T1313 BOOL  ; B机架#3门磁（公共）感应延时[0019.09]
T1314 BOOL  ; B机架#4门磁（公共）感应延时[0019.10]
T1315 BOOL  ; B机架#5门磁（公共）感应延时[0019.11]
T1316 BOOL  ; B机架#6门磁（公共）感应延时[0019.12]
T1317 BOOL  ; RK_07 #3托盘下料下降到位感应感应延时[0019.13]
T1318 BOOL  ; $?St$Bk?_#[5054] / RK_07 #3托盘下料位物料车到位感应#2感应延时[0019.14] / $?St$Bk?_#[5054]
T1319 BOOL  ; $?St$Bk?_#[5055] / RK_07 铝壳上料移载托盘到位保护感应感应延时[0019.15] / $?St$Bk?_#[5055]
T1322 BOOL  ; RK_02 电芯进料机械手#1压紧气缸压紧位感应延时
T1323 BOOL  ; RK_02 电芯进料机械手#2压紧气缸压紧位感应延时
T1326 BOOL  ; RK_03 电芯上料机械手#1压紧气缸压紧位感应延时
T1327 BOOL  ; RK_03 电芯上料机械手#2压紧气缸压紧位感应延时
T1373 BOOL  ; RK_05 #1入壳吸盘上#1伸缩气缸伸出位感应延时
T1374 BOOL  ; RK_05 #1入壳吸盘上#2伸缩气缸伸出位感应延时
T1375 BOOL  ; RK_05 #1入壳吸盘上#3伸缩气缸伸出位感应延时
T1376 BOOL  ; RK_05 #1入壳吸盘下#1伸缩气缸伸出位感应延时
T1377 BOOL  ; RK_05 #1入壳吸盘下#2伸缩气缸伸出位感应延时
T1378 BOOL  ; RK_05 #1入壳吸盘下#3伸缩气缸伸出位感应延时
T1391 BOOL  ; RK_05 #2入壳吸盘上#1伸缩气缸伸出位感应延时
T1392 BOOL  ; RK_05 #2入壳吸盘上#2伸缩气缸伸出位感应延时
T1393 BOOL  ; RK_05 #2入壳吸盘上#3伸缩气缸伸出位感应延时
T1394 BOOL  ; RK_05 #2入壳吸盘下#1伸缩气缸伸出位感应延时
T1395 BOOL  ; RK_05 #2入壳吸盘下#2伸缩气缸伸出位感应延时
T1396 BOOL  ; RK_05 #2入壳吸盘下#3伸缩气缸伸出位感应延时
T1500 BOOL  ; RK_02 电芯进料机械手夹爪气缸夹紧位报警延时
T1501 BOOL  ; RK_02 电芯进料机械手夹爪气缸张开位报警延时
T1502 BOOL  ; RK_02 电芯进料机械手#1压紧气缸松开位报警延时
T1503 BOOL  ; RK_02 电芯进料机械手#2压紧气缸松开位报警延时
T1504 BOOL  ; RK_03 电芯上料机械手夹爪气缸夹紧位报警延时
T1505 BOOL  ; RK_03 电芯上料机械手夹爪气缸张开位报警延时
T1506 BOOL  ; RK_03 电芯上料机械手#1压紧气缸松开位报警延时
T1507 BOOL  ; RK_03 电芯上料机械手#2压紧气缸松开位报警延时
T1508 BOOL  ; RK_03 电芯上料升降气缸下降位报警延时
T1509 BOOL  ; RK_03 电芯上料升降气缸上升位报警延时
T1510 BOOL  ; RK_04 电芯除尘伸缩气缸缩回位报警延时
T1511 BOOL  ; RK_04 电芯除尘伸缩气缸伸出位报警延时
T1512 BOOL  ; RK_05 #1入壳滚轮夹紧气缸夹紧位报警延时
T1513 BOOL  ; RK_05 #1入壳滚轮夹紧气缸松开位报警延时
T1514 BOOL  ; RK_05 #1入壳铝壳定位平台伸缩气缸缩回位报警延时
T1515 BOOL  ; RK_05 #1入壳铝壳定位平台伸缩气缸伸出位报警延时
T1516 BOOL  ; RK_05 #1入壳铝壳定位平台升降气缸上升位报警延时
T1517 BOOL  ; RK_05 #1入壳铝壳定位平台升降气缸下降位报警延时
T1518 BOOL  ; RK_05 #1入壳铝壳定位伸缩气缸缩回位报警延时
T1519 BOOL  ; RK_05 #1入壳铝壳定位伸缩气缸伸出位报警延时
T1520 BOOL  ; RK_05 #1入壳铝壳定位夹爪气缸夹紧位报警延时
T1521 BOOL  ; RK_05 #1入壳铝壳定位夹爪气缸张开位报警延时
T1522 BOOL  ; RK_05 #2入壳滚轮夹紧气缸夹紧位报警延时
T1523 BOOL  ; RK_05 #2入壳滚轮夹紧气缸松开位报警延时
T1524 BOOL  ; RK_05 #2入壳铝壳定位平台伸缩气缸缩回位报警延时
T1525 BOOL  ; RK_05 #2入壳铝壳定位平台伸缩气缸伸出位报警延时
T1526 BOOL  ; RK_05 #2入壳铝壳定位平台升降气缸上升位报警延时
T1527 BOOL  ; RK_05 #2入壳铝壳定位平台升降气缸下降位报警延时
T1528 BOOL  ; RK_05 #2入壳铝壳定位伸缩气缸缩回位报警延时
T1529 BOOL  ; RK_05 #2入壳铝壳定位伸缩气缸伸出位报警延时
T1530 BOOL  ; RK_05 #2入壳铝壳定位夹爪气缸夹紧位报警延时
T1531 BOOL  ; RK_05 #2入壳铝壳定位夹爪气缸张开位报警延时
T1532 BOOL  ; RK_01 U0_X 电芯来料Y轴报警信号报警延时
T1533 BOOL  ; RK_01 U0_X 电芯来料Y轴准备好了信号报警延时
T1534 BOOL  ; RK_02 U0_Y 电芯进料X轴报警信号报警延时
T1535 BOOL  ; RK_02 U0_Y 电芯进料X轴准备好了信号报警延时
T1536 BOOL  ; RK_02 U0_Z 电芯进料Z轴报警信号报警延时
T1537 BOOL  ; RK_02 U0_Z 电芯进料Z轴准备好了信号报警延时
T1538 BOOL  ; RK_03 U0_U 电芯上料X轴报警信号报警延时
T1539 BOOL  ; RK_03 U0_U 电芯上料X轴准备好了信号报警延时
T1540 BOOL  ; RK_05 U2_X #1入壳Y轴报警信号报警延时
T1541 BOOL  ; RK_05 U2_X #1入壳Y轴准备好了信号报警延时
T1542 BOOL  ; RK_05 U2_Y #2入壳Y轴报警信号报警延时
T1543 BOOL  ; RK_05 U2_Y #2入壳Y轴准备好了信号报警延时
T1544 BOOL  ; 0报警延时
T1545 BOOL  ; RK_05 #1入壳定位陶瓷棒上#1夹紧气缸伸出位报警延时
T1546 BOOL  ; RK_05 #1入壳定位陶瓷棒上#2夹紧气缸伸出位报警延时
T1547 BOOL  ; RK_05 #1入壳定位陶瓷棒下#1夹紧气缸伸出位报警延时
T1548 BOOL  ; RK_05 #1入壳定位陶瓷棒下#2夹紧气缸伸出位报警延时
T1549 BOOL  ; RK_05 #1入壳定位陶瓷棒上#1夹紧气缸缩回位报警延时
T1550 BOOL  ; RK_05 #1入壳定位陶瓷棒上#2夹紧气缸缩回位报警延时
T1551 BOOL  ; RK_05 #1入壳定位陶瓷棒下#1夹紧气缸缩回位报警延时
T1552 BOOL  ; RK_05 #1入壳定位陶瓷棒下#2夹紧气缸缩回位报警延时
T1553 BOOL  ; RK_05 #1入壳吸盘上#1伸缩气缸缩回位报警延时
T1554 BOOL  ; RK_05 #1入壳吸盘上#2伸缩气缸缩回位报警延时
T1555 BOOL  ; RK_05 #1入壳吸盘上#3伸缩气缸缩回位报警延时
T1556 BOOL  ; RK_05 #1入壳吸盘下#1伸缩气缸缩回位报警延时
T1557 BOOL  ; RK_05 #1入壳吸盘下#2伸缩气缸缩回位报警延时
T1558 BOOL  ; RK_05 #1入壳吸盘下#3伸缩气缸缩回位报警延时
T1559 BOOL  ; RK_05 #1入壳电芯#1定位夹爪气缸松开位报警延时
T1560 BOOL  ; RK_05 #1入壳电芯#2定位夹爪气缸松开位报警延时
T1561 BOOL  ; RK_05 #1入壳电芯#1定位夹爪气缸夹紧位报警延时
T1562 BOOL  ; RK_05 #1入壳电芯#2定位夹爪气缸夹紧位报警延时
T1563 BOOL  ; RK_05 #2入壳定位陶瓷棒上#1夹紧气缸伸出位报警延时
T1564 BOOL  ; RK_05 #2入壳定位陶瓷棒上#2夹紧气缸伸出位报警延时
T1565 BOOL  ; RK_05 #2入壳定位陶瓷棒下#1夹紧气缸伸出位报警延时
T1566 BOOL  ; RK_05 #2入壳定位陶瓷棒下#2夹紧气缸伸出位报警延时
T1567 BOOL  ; RK_05 #2入壳定位陶瓷棒上#1夹紧气缸缩回位报警延时
T1568 BOOL  ; RK_05 #2入壳定位陶瓷棒上#2夹紧气缸缩回位报警延时
T1569 BOOL  ; RK_05 #2入壳定位陶瓷棒下#1夹紧气缸缩回位报警延时
T1570 BOOL  ; RK_05 #2入壳定位陶瓷棒下#2夹紧气缸缩回位报警延时
T1571 BOOL  ; RK_05 #2入壳吸盘上#1伸缩气缸缩回位报警延时
T1572 BOOL  ; RK_05 #2入壳吸盘上#2伸缩气缸缩回位报警延时
T1573 BOOL  ; RK_05 #2入壳吸盘上#3伸缩气缸缩回位报警延时
T1574 BOOL  ; RK_05 #2入壳吸盘下#1伸缩气缸缩回位报警延时
T1575 BOOL  ; RK_05 #2入壳吸盘下#2伸缩气缸缩回位报警延时
T1576 BOOL  ; RK_05 #2入壳吸盘下#3伸缩气缸缩回位报警延时
T1577 BOOL  ; RK_05 #2入壳电芯#1定位夹爪气缸松开位报警延时
T1578 BOOL  ; RK_05 #2入壳电芯#2定位夹爪气缸松开位报警延时
T1579 BOOL  ; RK_05 #2入壳电芯#1定位夹爪气缸夹紧位报警延时
T1580 BOOL  ; RK_05 #2入壳电芯#2定位夹爪气缸夹紧位报警延时
T1581 BOOL  ; RK_01 电芯来料有料感应报警延时
T1582 BOOL  ; RK_02 电芯进料机械手夹爪柔性报警报警延时
T1583 BOOL  ; RK_03 电芯上料机械手夹爪柔性报警报警延时
T1584 BOOL  ; RK_04 电芯除尘有料感应报警延时
T1585 BOOL  ; RK_02 扫码NG拉带有料感应#1报警延时
T1586 BOOL  ; RK_02 扫码NG拉带有料感应#2报警延时
T1587 BOOL  ; RK_02 扫码NG拉带料满感应报警延时
T1588 BOOL  ; RK_05 #1入壳电芯有料感应报警延时
T1589 BOOL  ; RK_05 #1入壳铝壳有料感应报警延时
T1590 BOOL  ; RK_05 #2入壳电芯有料感应报警延时
T1591 BOOL  ; RK_05 #2入壳铝壳有料感应报警延时
T1592 BOOL  ; RK_05 #1入壳吸盘立真空报警延时
T1593 BOOL  ; RK_05 #2入壳吸盘立真空报警延时
T1594 BOOL  ; 前端设备对接输入信号（公共）报警延时
T1595 BOOL  ; 后端设备对接输入信号（公共）报警延时
T1597 BOOL  ; NC433模块DC5V电源信号（公共）报警延时
T1598 BOOL  ; DC24V伺服刹车电源信号（公共）报警延时
T1610 BOOL  ; 0报警延时
T1611 BOOL  ; 0报警延时
T1612 BOOL  ; 0报警延时
T1613 BOOL  ; 0报警延时
T1614 BOOL  ; 0报警延时
T1615 BOOL  ; 0报警延时
T1616 BOOL  ; 0报警延时
T1617 BOOL  ; 0报警延时
T1618 BOOL  ; 0报警延时
T1619 BOOL  ; 0报警延时
T1620 BOOL  ; 0报警延时
T1621 BOOL  ; 0报警延时
T1622 BOOL  ; 0报警延时
T1623 BOOL  ; 0报警延时
T1624 BOOL  ; 0报警延时
T1625 BOOL  ; 0报警延时
T1626 BOOL  ; 0报警延时
T1627 BOOL  ; 0报警延时
T1628 BOOL  ; RK_11 电池除尘旋转伸缩气缸到位报警延时
T1629 BOOL  ; RK_11 电池除尘旋转伸缩气缸原位报警延时
T1630 BOOL  ; RK_11 电池除尘伸缩气缸伸出位报警延时
T1631 BOOL  ; RK_11 电池除尘伸缩气缸缩回位报警延时
T1632 BOOL  ; RK_11 电池除尘夹爪气缸夹紧位报警延时
T1633 BOOL  ; RK_11 电池除尘夹爪气缸张开位报警延时
T1634 BOOL  ; RK_12 预焊上料机械手夹爪气缸夹紧位报警延时
T1635 BOOL  ; RK_12 预焊上料机械手夹爪气缸张开位报警延时
T1636 BOOL  ; RK_12 预焊下料机械手夹爪气缸夹紧位报警延时
T1637 BOOL  ; RK_12 预焊下料机械手夹爪气缸张开位报警延时
T1638 BOOL  ; RK_13 #1移载升降气缸上升位报警延时
T1639 BOOL  ; RK_13 #1移载升降气缸下降位报警延时
T1640 BOOL  ; RK_13 #1移载定位#1伸缩气缸缩回位报警延时
T1641 BOOL  ; RK_13 #1移载定位#1伸缩气缸伸出位报警延时
T1642 BOOL  ; RK_13 #1移载定位#2伸缩气缸缩回位报警延时
T1643 BOOL  ; RK_13 #1移载定位#2伸缩气缸伸出位报警延时
T1644 BOOL  ; RK_13 #1移载导向#1伸缩气缸伸出位报警延时
T1645 BOOL  ; RK_13 #1移载导向#1伸缩气缸缩回位报警延时
T1646 BOOL  ; RK_13 #1移载导向#2伸缩气缸伸出位报警延时
T1647 BOOL  ; RK_13 #1移载导向#2伸缩气缸缩回位报警延时
T1648 BOOL  ; RK_13 #1移载左右定位伸缩气缸伸出位报警延时
T1649 BOOL  ; RK_13 #1移载左右定位伸缩气缸缩回位报警延时
T1650 BOOL  ; RK_13 #2移载升降气缸上升位报警延时
T1651 BOOL  ; RK_13 #2移载升降气缸下降位报警延时
T1652 BOOL  ; RK_13 #2移载定位#1伸缩气缸缩回位报警延时
T1653 BOOL  ; RK_13 #2移载定位#1伸缩气缸伸出位报警延时
T1654 BOOL  ; RK_13 #2移载定位#2伸缩气缸缩回位报警延时
T1655 BOOL  ; RK_13 #2移载定位#2伸缩气缸伸出位报警延时
T1656 BOOL  ; RK_13 #2移载导向#1伸缩气缸伸出位报警延时
T1657 BOOL  ; RK_13 #2移载导向#1伸缩气缸缩回位报警延时
T1658 BOOL  ; RK_13 #2移载导向#2伸缩气缸伸出位报警延时
T1659 BOOL  ; RK_13 #2移载导向#2伸缩气缸缩回位报警延时
T1660 BOOL  ; RK_13 #2移载左右定位伸缩气缸伸出位报警延时
T1661 BOOL  ; RK_13 #2移载左右定位伸缩气缸缩回位报警延时
T1662 BOOL  ; RK_14 #1压装升降气缸下降位报警延时
T1663 BOOL  ; RK_14 #1压装升降气缸上升位报警延时
T1664 BOOL  ; RK_14 #1压装#1吸盘升降气缸下降位报警延时
T1665 BOOL  ; RK_14 #1压装#1吸盘升降气缸上升位报警延时
T1666 BOOL  ; RK_14 #1压装#2吸盘升降气缸下降位报警延时
T1667 BOOL  ; RK_14 #1压装#2吸盘升降气缸上升位报警延时
T1668 BOOL  ; RK_14 #2压装升降气缸下降位报警延时
T1669 BOOL  ; RK_14 #2压装升降气缸上升位报警延时
T1670 BOOL  ; RK_14 #2压装#1吸盘升降气缸下降位报警延时
T1671 BOOL  ; RK_14 #2压装#1吸盘升降气缸上升位报警延时
T1672 BOOL  ; RK_14 #2压装#2吸盘升降气缸下降位报警延时
T1673 BOOL  ; RK_14 #2压装#2吸盘升降气缸上升位报警延时
T1674 BOOL  ; RK_15 轮廓检测#1伸缩气缸伸出位报警延时
T1675 BOOL  ; RK_15 轮廓检测#1伸缩气缸缩回位报警延时
T1676 BOOL  ; RK_15 轮廓检测#2伸缩气缸伸出位报警延时
T1677 BOOL  ; RK_15 轮廓检测#2伸缩气缸缩回位报警延时
T1678 BOOL  ; RK_12 轮廓检测NG拨料气缸伸出位报警延时
T1679 BOOL  ; RK_12 轮廓检测NG拨料气缸缩回位报警延时
T1680 BOOL  ; RK_11 电池除尘有料感应报警延时
T1681 BOOL  ; RK_12 预焊上料机械手夹爪柔性报警报警延时
T1682 BOOL  ; RK_12 预焊下料机械手夹爪柔性报警报警延时
T1683 BOOL  ; RK_16 激光焊接完成信号报警延时
T1684 BOOL  ; RK_16 激光焊机故障信号报警延时
T1685 BOOL  ; RK_13 #1移载电池顶盖超高检测报警延时
T1686 BOOL  ; RK_16 激光焊机急停信号报警延时
T1687 BOOL  ; RK_13 #2移载电池顶盖超高检测报警延时
T1688 BOOL  ; RK_13 #1移载有料感应报警延时
T1689 BOOL  ; RK_13 #2移载有料感应报警延时
T1690 BOOL  ; RK_14 #1压装吸盘立真空报警延时
T1691 BOOL  ; RK_14 #2压装吸盘立真空报警延时
T1692 BOOL  ; RK_12 U4_X 预焊上下料X轴报警信号报警延时
T1693 BOOL  ; RK_12 U4_X 预焊上下料X轴准备好了信号报警延时
T1694 BOOL  ; RK_12 U4_Y 预焊上料Z轴报警信号报警延时
T1695 BOOL  ; RK_12 U4_Y 预焊上料Z轴准备好了信号报警延时
T1696 BOOL  ; RK_12 U4_Z 预焊下料Z轴报警信号报警延时
T1697 BOOL  ; RK_12 U4_Z 预焊下料Z轴准备好了信号报警延时
T1698 BOOL  ; RK_13 U4_U #1移载Y轴报警信号报警延时
T1699 BOOL  ; RK_13 U4_U #1移载Y轴准备好了信号报警延时
T1700 BOOL  ; RK_13 U6_X #2移载Y轴报警信号报警延时
T1701 BOOL  ; RK_13 U6_X #2移载Y轴准备好了信号报警延时
T1702 BOOL  ; RK_16 U6_Y 激光焊接X轴报警信号报警延时
T1703 BOOL  ; RK_16 U6_Y 激光焊接X轴准备好了信号报警延时
T1704 BOOL  ; RK_16 U6_Z 激光焊接Z轴报警信号报警延时
T1705 BOOL  ; RK_16 U6_Z 激光焊接Z轴准备好了信号报警延时
T1706 BOOL  ; 0报警延时
T1707 BOOL  ; 0报警延时
T1708 BOOL  ; 0报警延时
T1709 BOOL  ; RK_12 轮廓检测NG料槽#1有料感应报警延时
T1710 BOOL  ; RK_12 轮廓检测NG料槽#1料满感应报警延时
T1711 BOOL  ; RK_12 轮廓检测NG料槽#2有料感应报警延时
T1712 BOOL  ; RK_12 轮廓检测NG料槽#2料满感应报警延时
T1713 BOOL  ; RK_12 OK出料拉带放料位有料感应#1报警延时
T1714 BOOL  ; RK_12 OK出料拉带放料位有料感应#2报警延时
T1715 BOOL  ; RK_12 OK出料拉带出料位有料感应报警延时
T1716 BOOL  ; 0报警延时
T1717 BOOL  ; 0报警延时
T1718 BOOL  ; 0报警延时
T1719 BOOL  ; 0报警延时
T1720 BOOL  ; 0报警延时
T1721 BOOL  ; 0报警延时
T1722 BOOL  ; 0报警延时
T1723 BOOL  ; 0报警延时
T1724 BOOL  ; RK_06 铝壳上料升降气缸下降位报警延时
T1725 BOOL  ; RK_06 铝壳上料升降气缸上升位报警延时
T1726 BOOL  ; RK_06 电池下料升降气缸下降位报警延时
T1727 BOOL  ; RK_06 电池下料升降气缸上升位报警延时
T1728 BOOL  ; RK_06 铝壳上料夹爪气缸夹紧位报警延时
T1729 BOOL  ; RK_06 铝壳上料夹爪气缸张开位报警延时
T1730 BOOL  ; RK_06 电池下料夹爪气缸夹紧位报警延时
T1731 BOOL  ; RK_06 电池下料夹爪气缸张开位报警延时
T1732 BOOL  ; RK_07 #1铝壳上料车定位升降气缸上升位报警延时
T1733 BOOL  ; RK_07 #1铝壳上料车定位升降气缸下降位报警延时
T1734 BOOL  ; RK_07 #2铝壳上料车定位升降气缸上升位报警延时
T1735 BOOL  ; RK_07 #2铝壳上料车定位升降气缸下降位报警延时
T1736 BOOL  ; RK_07 #3托盘下料车定位升降气缸上升位报警延时
T1737 BOOL  ; RK_07 #3托盘下料车定位升降气缸下降位报警延时
T1738 BOOL  ; RK_07 铝壳进料机械手升降气缸下降位报警延时
T1739 BOOL  ; RK_07 铝壳进料机械手升降气缸上升位报警延时
T1740 BOOL  ; RK_08 铝壳除尘旋转伸缩气缸原位报警延时
T1741 BOOL  ; RK_08 铝壳除尘旋转伸缩气缸到位报警延时
T1742 BOOL  ; RK_08 铝壳除尘伸缩气缸伸出位报警延时
T1743 BOOL  ; RK_08 铝壳除尘伸缩气缸缩回位报警延时
T1744 BOOL  ; RK_08 铝壳除尘夹爪气缸夹紧位报警延时
T1745 BOOL  ; RK_08 铝壳除尘夹爪气缸张开位报警延时
T1746 BOOL  ; RK_09 #1Hipot测试旋转伸缩气缸到位报警延时
T1747 BOOL  ; RK_09 #1Hipot测试旋转伸缩气缸原位报警延时
T1748 BOOL  ; RK_09 #1Hipot测试平台伸缩气缸缩回位报警延时
T1749 BOOL  ; RK_09 #1Hipot测试平台伸缩气缸伸出位报警延时
T1750 BOOL  ; RK_09 #1Hipot测试伸缩气缸伸出位报警延时
T1751 BOOL  ; RK_09 #1Hipot测试伸缩气缸缩回位报警延时
T1752 BOOL  ; RK_09 #2Hipot测试旋转伸缩气缸到位报警延时
T1753 BOOL  ; RK_09 #2Hipot测试旋转伸缩气缸原位报警延时
T1754 BOOL  ; RK_09 #2Hipot测试平台伸缩气缸缩回位报警延时
T1755 BOOL  ; RK_09 #2Hipot测试平台伸缩气缸伸出位报警延时
T1756 BOOL  ; RK_09 #2Hipot测试伸缩气缸伸出位报警延时
T1757 BOOL  ; RK_09 #2Hipot测试伸缩气缸缩回位报警延时
T1758 BOOL  ; RK_10 电池除尘上料机械手升降气缸下降位报警延时
T1759 BOOL  ; RK_10 电池除尘上料机械手升降气缸上升位报警延时
T1760 BOOL  ; RK_10 电池除尘上料机械手夹爪气缸夹紧位报警延时
T1761 BOOL  ; RK_10 电池除尘上料机械手夹爪气缸张开位报警延时
T1762 BOOL  ; RK_06 U8_X 电池上下料X轴报警信号报警延时
T1763 BOOL  ; RK_06 U8_X 电池上下料X轴准备好了信号报警延时
T1764 BOOL  ; RK_07 U8_Y 铝壳进料X轴报警信号报警延时
T1765 BOOL  ; RK_07 U8_Y 铝壳进料X轴准备好了信号报警延时
T1766 BOOL  ; RK_07 U8_Z 铝壳上料移载Y轴报警信号报警延时
T1767 BOOL  ; RK_07 U8_Z 铝壳上料移载Y轴准备好了信号报警延时
T1768 BOOL  ; RK_10 U8_U 电池除尘上料X轴报警信号报警延时
T1769 BOOL  ; RK_10 U8_U 电池除尘上料X轴准备好了信号报警延时
T1770 BOOL  ; RK_09 Hipot测试完成信号报警延时
T1771 BOOL  ; RK_07 #1铝壳上料启动按钮报警延时
T1772 BOOL  ; RK_07 #2铝壳上料启动按钮报警延时
T1773 BOOL  ; RK_07 #3托盘下料启动按钮报警延时
T1774 BOOL  ; RK_07 铝壳上料移载吸盘立真空报警延时
T1775 BOOL  ; RK_07 铝壳进料吸盘立真空报警延时
T1776 BOOL  ; RK_07 #1铝壳上料托盘到位感应报警延时
T1777 BOOL  ; RK_07 #1铝壳上料位物料车到位感应报警延时
T1778 BOOL  ; RK_07 #1铝壳上料初始位（#1）报警延时
T1779 BOOL  ; RK_07 #1铝壳上料一个托盘位（#2）报警延时
T1780 BOOL  ; RK_07 #1铝壳上料高限位（#3）报警延时
T1781 BOOL  ; RK_07 #2铝壳上料托盘到位感应报警延时
T1782 BOOL  ; RK_07 #2铝壳上料位物料车到位感应报警延时
T1783 BOOL  ; RK_07 #2铝壳上料初始位（#1）报警延时
T1784 BOOL  ; RK_07 #2铝壳上料一个托盘位（#2）报警延时
T1785 BOOL  ; RK_07 #2铝壳上料高限位（#3）报警延时
T1786 BOOL  ; RK_07 #3托盘下料上升到位感应报警延时
T1787 BOOL  ; RK_07 #3托盘下料位物料车到位感应报警延时
T1788 BOOL  ; RK_07 #3托盘下料初始位（#1）报警延时
T1789 BOOL  ; RK_07 #3托盘下料一个托盘位（#2）报警延时
T1790 BOOL  ; RK_07 #3托盘下料高限位（#3）报警延时
T1791 BOOL  ; RK_07 铝壳上料移载托盘到位感应报警延时
T1792 BOOL  ; RK_08 铝壳除尘有料感应报警延时
T1793 BOOL  ; RK_09 #1Hipot测试有料感应报警延时
T1794 BOOL  ; RK_09 #2Hipot测试有料感应报警延时
T1795 BOOL  ; RK_10 Hipot检测NG拉带有料感应#1报警延时
T1796 BOOL  ; RK_10 Hipot检测NG拉带有料感应#2报警延时
T1797 BOOL  ; RK_10 Hipot检测NG拉带料满感应报警延时
T1798 BOOL  ; RK_06 铝壳上料夹爪柔性报警报警延时
T1799 BOOL  ; RK_06 电池下料夹爪柔性报警报警延时
T1800 BOOL  ; RK_07 铝壳进料机械手柔性报警报警延时
T1801 BOOL  ; RK_10 电池除尘上料机械手夹爪柔性报警报警延时
T1806 BOOL  ; 机台进气压力（正压）（公共）报警延时
T1807 BOOL  ; 机台进气压力（负压）（公共）报警延时
T1817 BOOL  ; RK_07 #3托盘下料下降到位感应报警延时
T1819 BOOL  ; $?St$Bk?_#[5056] / RK_07 铝壳上料移载托盘到位保护感应报警延时 / $?St$Bk?_#[5056]
T1822 BOOL  ; RK_02 电芯进料机械手#1压紧气缸压紧位报警延时
T1823 BOOL  ; RK_02 电芯进料机械手#2压紧气缸压紧位报警延时
T1826 BOOL  ; RK_03 电芯上料机械手#1压紧气缸压紧位报警延时
T1827 BOOL  ; RK_03 电芯上料机械手#2压紧气缸压紧位报警延时
T1836 BOOL  ; RK_05 #1入壳压力高报警延时
T1837 BOOL  ; RK_05 #2入壳压力高报警延时
T1852 BOOL  ; RK_01 U0_X 电芯来料Y轴无原点信号报警延时
T1853 BOOL  ; RK_02 U0_Y 电芯进料X轴无原点信号报警延时
T1854 BOOL  ; RK_02 U0_Z 电芯进料Z轴无原点信号报警延时
T1855 BOOL  ; RK_03 U0_U 电芯上料X轴无原点信号报警延时
T1856 BOOL  ; RK_05 U2_X #1入壳Y轴无原点信号报警延时
T1857 BOOL  ; RK_05 U2_Y #2入壳Y轴无原点信号报警延时
T1858 BOOL  ; RK_12 U4_X 预焊上下料X轴无原点信号报警延时
T1859 BOOL  ; RK_12 U4_Y 预焊上料Z轴无原点信号报警延时
T1860 BOOL  ; RK_12 U4_Z 预焊下料Z轴无原点信号报警延时
T1861 BOOL  ; RK_13 U4_U #1移载Y轴无原点信号报警延时
T1862 BOOL  ; RK_13 U6_X #2移载Y轴无原点信号报警延时
T1863 BOOL  ; RK_16 U6_Y 激光焊接X轴无原点信号报警延时
T1864 BOOL  ; RK_16 U6_Z 激光焊接Z轴无原点信号报警延时
T1865 BOOL  ; RK_06 U8_X 电池上下料X轴无原点信号报警延时
T1866 BOOL  ; RK_07 U8_Y 铝壳进料X轴无原点信号报警延时
T1867 BOOL  ; RK_07 U8_Z 铝壳上料移载Y轴无原点信号报警延时
T1868 BOOL  ; RK_10 U8_U 电池除尘上料X轴无原点信号报警延时
T1869 BOOL  ; 扫码阻挡#1伸出输出报警
T1870 BOOL  ; 扫码阻挡#1缩回输出报警
T1871 BOOL  ; 扫码阻挡#2伸出输出报警
T1872 BOOL  ; 扫码阻挡#2缩回输出报警
T1873 BOOL  ; RK_05 #1入壳吸盘上#1伸缩气缸伸出位报警延时
T1874 BOOL  ; RK_05 #1入壳吸盘上#2伸缩气缸伸出位报警延时
T1875 BOOL  ; RK_05 #1入壳吸盘上#3伸缩气缸伸出位报警延时
T1876 BOOL  ; RK_05 #1入壳吸盘下#1伸缩气缸伸出位报警延时
T1877 BOOL  ; RK_05 #1入壳吸盘下#2伸缩气缸伸出位报警延时
T1878 BOOL  ; RK_05 #1入壳吸盘下#3伸缩气缸伸出位报警延时
T1891 BOOL  ; RK_05 #2入壳吸盘上#1伸缩气缸伸出位报警延时
T1892 BOOL  ; RK_05 #2入壳吸盘上#2伸缩气缸伸出位报警延时
T1893 BOOL  ; RK_05 #2入壳吸盘上#3伸缩气缸伸出位报警延时
T1894 BOOL  ; RK_05 #2入壳吸盘下#1伸缩气缸伸出位报警延时
T1895 BOOL  ; RK_05 #2入壳吸盘下#2伸缩气缸伸出位报警延时
T1896 BOOL  ; RK_05 #2入壳吸盘下#3伸缩气缸伸出位报警延时
T1902 BOOL  ; RK_07 铝壳上料移载吸盘破真空报警延时
T1903 BOOL  ; RK_07 铝壳进料吸盘破真空报警延时
T1912 BOOL  ; RK_05 #1入壳吸盘破真空报警延时
T1913 BOOL  ; RK_05 #2入壳吸盘破真空报警延时
T1914 BOOL  ; RK_14 #1压装吸盘破真空报警延时
T1915 BOOL  ; RK_14 #2压装吸盘破真空报警延时
T1932 BOOL  ; RK_01 电芯来料机构复位超时报警延时
T1933 BOOL  ; RK_02 电芯进料机构复位超时报警延时
T1934 BOOL  ; RK_03 电芯上料机构复位超时报警延时
T1935 BOOL  ; RK_04 电芯除尘机构复位超时报警延时
T1936 BOOL  ; RK_05 #1入壳机构复位超时报警延时
T1937 BOOL  ; RK_05 #2入壳机构复位超时报警延时
T1938 BOOL  ; RK_06 电池上下料机构复位超时报警延时
T1939 BOOL  ; RK_07 铝壳进料机构复位超时报警延时
T1940 BOOL  ; RK_07 铝壳上料移载机构复位超时报警延时
T1941 BOOL  ; RK_07 #1铝壳上料升降机构复位超时报警延时
T1942 BOOL  ; RK_07 #2铝壳上料升降机构复位超时报警延时
T1943 BOOL  ; RK_07 铝壳托盘下料升降机构复位超时报警延时
T1944 BOOL  ; RK_08 铝壳除尘机构复位超时报警延时
T1945 BOOL  ; RK_09 #1Hipot检测机构复位超时报警延时
T1946 BOOL  ; RK_09 #2Hipot检测机构复位超时报警延时
T1947 BOOL  ; RK_10 电池除尘上料机构复位超时报警延时
T1948 BOOL  ; RK_11 电池除尘机构复位超时报警延时
T1949 BOOL  ; RK_12 预焊上下料机构复位超时报警延时
T1950 BOOL  ; RK_13 #1移载机构复位超时报警延时
T1951 BOOL  ; RK_13 #2移载机构复位超时报警延时
T1952 BOOL  ; RK_14 #1压装机构复位超时报警延时
T1953 BOOL  ; RK_14 #2压装机构复位超时报警延时
T1954 BOOL  ; RK_15 轮廓检测机构复位超时报警延时
T1955 BOOL  ; RK_16 焊接机构复位超时报警延时
T1962 BOOL  ; 整机复位超时报警延时
T1963 BOOL  ; 激光焊接超时报警延时
T1964 BOOL  ; RK_01 电芯来料机构有料记忆报警延时
T1965 BOOL  ; RK_02 扫码NG拉带放料位有料记忆报警延时
T1966 BOOL  ; RK_04 电芯除尘机构有料记忆报警延时
T1967 BOOL  ; RK_05 #1入壳机构有电池记忆报警延时
T1968 BOOL  ; RK_05 #1入壳机构有电芯记忆报警延时
T1969 BOOL  ; RK_05 #1入壳机构有铝壳记忆报警延时
T1970 BOOL  ; RK_05 #2入壳机构有电池记忆报警延时
T1971 BOOL  ; RK_05 #2入壳机构有电芯记忆报警延时
T1972 BOOL  ; RK_05 #2入壳机构有铝壳记忆报警延时
T1973 BOOL  ; RK_11 电池除尘机构有料记忆报警延时
T1974 BOOL  ; RK_08 铝壳除尘机构有料记忆报警延时
T1975 BOOL  ; RK_09 #1Hipot检测机构有料记忆报警延时
T1976 BOOL  ; RK_09 #2Hipot检测机构有料记忆报警延时
T1977 BOOL  ; RK_10 Hipot检测NG拉带放料位有料记忆报警延时
T1978 BOOL  ; RK_12 轮廓检测NG槽#1有料记忆报警延时
T1979 BOOL  ; RK_12 轮廓检测NG槽#2有料记忆报警延时
T1980 BOOL  ; RK_13 #1移载有料记忆报警延时
T1981 BOOL  ; RK_13 #2移载有料记忆报警延时
T1982 BOOL  ; RK_12 出料拉带放料位有料记忆报警延时
T1983 BOOL  ; RK_07 铝壳上料移载机构有托盘记忆报警延时
T1984 BOOL  ; RK_07 铝壳上料移载机构托盘有料记忆报警延时
T1992 BOOL  ; $?St$Bk?_#[5057] / 电芯进料X轴允许去放料位安全设定值过小 / 报警延时$?St$Bk?_#[5057]
T1993 BOOL  ; $?St$Bk?_#[5058] / 电芯上料X轴允许去取料位安全设定值过小 / 报警延时$?St$Bk?_#[5058]
T1994 BOOL  ; 电池除尘上料X轴允许去电池除尘放料位安全设定值过小报警延时
T1995 BOOL  ; $?St$Bk?_#[5059] / 预焊上下料X轴允许去电池除尘取料位安全设定值过小 / 报警延时$?St$Bk?_#[5059]
T1996 BOOL  ; RK_02 电芯进料机构MES入站就绪通知&确认超时报警延时
T1997 BOOL  ; RK_11 电池除尘上料机构MES出站就绪通知&确认超时报警延时
T1998 BOOL  ; RK_12 电池上下料机构MES出站就绪通知&确认超时报警延时
T1999 BOOL  ; 整机工艺参数变更通知&确认超时报警延时
T2500 BOOL  ; RK_01 电芯来料机构开始运行条件延时
T2509 BOOL  ; RK_01 电芯来料机构复位完成延时
T2510 BOOL  ; RK_02 电芯进料机构开始运行条件延时
T2519 BOOL  ; RK_02 电芯进料机构复位完成延时
T2520 BOOL  ; RK_03 电芯上料机构开始运行条件延时
T2529 BOOL  ; RK_03 电芯上料机构复位完成延时
T2530 BOOL  ; RK_04 电芯除尘机构开始运行条件延时
T2538 BOOL  ; 电芯除尘机构吹气延时
T2539 BOOL  ; RK_04 电芯除尘机构复位完成延时
T2540 BOOL  ; RK_05 #1入壳机构开始运行条件1延时（铝壳定位）
T2541 BOOL  ; RK_05 #1入壳机构开始运行条件2延时（电芯定位&入壳）
T2549 BOOL  ; RK_05 #1入壳机构复位完成延时
T2550 BOOL  ; RK_05 #2入壳机构开始运行条件1延时（铝壳定位）
T2551 BOOL  ; RK_05 #2入壳机构开始运行条件2延时（电芯定位&入壳）
T2559 BOOL  ; RK_05 #2入壳机构复位完成延时
T2560 BOOL  ; RK_06 电池上下料机构开始运行条件1延时（铝壳取料）
T2561 BOOL  ; RK_06 电池上下料机构开始运行条件2延时（铝壳下料）
T2562 BOOL  ; RK_06 电池上下料机构开始运行条件3延时（电池取料）
T2563 BOOL  ; RK_06 电池上下料机构开始运行条件4延时（电池下料）
T2569 BOOL  ; RK_06 电池上下料机构复位完成延时
T2570 BOOL  ; RK_07 铝壳进料机构开始运行条件延时
T2579 BOOL  ; RK_07 铝壳进料机构复位完成延时
T2580 BOOL  ; RK_07 铝壳上料移载机构开始运行条件1延时（铝壳上料）
T2581 BOOL  ; RK_07 铝壳上料移载机构开始运行条件2延时（铝壳取料）
T2582 BOOL  ; RK_07 铝壳上料移载机构开始运行条件3延时（铝壳托盘卸载）
T2589 BOOL  ; RK_07 铝壳上料移载机构复位完成延时
T2595 BOOL  ; #1铝壳上料电机初次上料反转到安全位延时
T2596 BOOL  ; #1铝壳上料车定位升降气缸下降延时
T2605 BOOL  ; #2铝壳上料电机初次上料反转到安全位延时
T2606 BOOL  ; #2铝壳上料车定位升降气缸下降延时
T2615 BOOL  ; #3铝壳下料电机初次下料反转到安全位延时
T2620 BOOL  ; RK_08 铝壳除尘机构开始运行条件延时
T2628 BOOL  ; 铝壳除尘机构吹气延时
T2629 BOOL  ; RK_08 铝壳除尘机构复位完成延时
T2630 BOOL  ; RK_09 #1Hipot检测机构开始运行条件延时
T2635 BOOL  ; RK_09 #1Hipot检测机构测试触发延时
T2636 BOOL  ; RK_09 #1Hipot检测机构测试完成放电延时
T2637 BOOL  ; RK_09 Hipot测试完成读结果延时
T2639 BOOL  ; RK_09 #1Hipot检测机构复位完成延时
T2640 BOOL  ; RK_09 #2Hipot检测机构开始运行条件延时
T2645 BOOL  ; RK_09 #2Hipot检测机构测试触发延时
T2646 BOOL  ; RK_09 #2Hipot检测机构测试完成放电延时
T2649 BOOL  ; RK_09 #2Hipot检测机构复位完成延时
T2650 BOOL  ; RK_10 电池除尘上料机构开始运行条件延时
T2659 BOOL  ; RK_10 电池除尘上料机构复位完成延时
T2660 BOOL  ; RK_11 电池除尘机构开始运行条件延时
T2668 BOOL  ; 电池除尘机构吹气延时
T2669 BOOL  ; RK_11 电池除尘机构复位完成延时
T2670 BOOL  ; RK_12 预焊上下料机构开始运行条件1延时（预焊电池取料）
T2671 BOOL  ; RK_12 预焊上下料机构开始运行条件2延时（预焊电池放料）
T2672 BOOL  ; RK_12 预焊上下料机构开始运行条件3延时（OK/NG电池取料）
T2673 BOOL  ; RK_12 预焊上下料机构开始运行条件4延时（OK/NG电池放料）
T2679 BOOL  ; RK_12 预焊上下料机构复位完成延时
T2680 BOOL  ; RK_13 #1移载机构开始运行条件延时
T2689 BOOL  ; RK_13 #1移载机构复位完成延时
T2690 BOOL  ; RK_13 #2移载机构开始运行条件延时
T2699 BOOL  ; RK_13 #2移载机构复位完成延时
T2700 BOOL  ; RK_14 #1压装机构开始运行条件延时
T2709 BOOL  ; RK_14 #1压装机构复位完成延时
T2710 BOOL  ; RK_14 #2压装机构开始运行条件延时
T2719 BOOL  ; RK_14 #2压装机构复位完成延时
T2720 BOOL  ; RK_15 轮廓检测机构开始运行条件延时
T2724 BOOL  ; RK_15 轮廓检测机构测量数据初始化延时
T2725 BOOL  ; RK_15 轮廓检测机构#1点测量读数据延时
T2726 BOOL  ; RK_15 轮廓检测机构#2点测量读数据延时
T2727 BOOL  ; RK_15 轮廓检测机构#3点测量读数据延时
T2728 BOOL  ; RK_15 轮廓检测机构#4点测量读数据延时
T2729 BOOL  ; RK_15 轮廓检测机构复位完成延时
T2730 BOOL  ; RK_16 焊接机构开始运行条件延时
T2735 BOOL  ; RK_16 焊接机构激光焊接延时触发
T2736 BOOL  ; RK_16 焊接机构激光焊接触发延时
T2739 BOOL  ; RK_16 焊接机构复位完成延时
T2800 BOOL  ; 电芯进料扫码数据初始化延时
T2801 BOOL  ; 进料扫码延时
T2802 BOOL  ; 接收数据清零延时发送无协议通讯TXD
T2803 BOOL  ; 扫码结果判定延时
T2804 BOOL  ; 扫码发送超时
T2822 BOOL  ; Hipot检测仪参数写入标志延时
T2840 BOOL  ; RK_15 轮廓检测机构测量程序切换解析延时
T2841 BOOL  ; RK_15 轮廓检测机构测量数据读取解析延时
T2843 BOOL  ; RK_15 轮廓检测机构测量数据读取触发延时
T2860 BOOL  ; RK_07 U8_Y 铝壳进料X轴#1取料位感应延时
T2861 BOOL  ; RK_07 U8_Y 铝壳进料X轴#2取料位感应延时
T2862 BOOL  ; RK_07 U8_Y 铝壳进料X轴#3取料位感应延时
T2863 BOOL  ; RK_07 U8_Y 铝壳进料X轴#4取料位感应延时
T2864 BOOL  ; RK_07 U8_Y 铝壳进料X轴#5取料位感应延时
T2880 BOOL  ; RK_07 U8_Z 铝壳上料移载Y轴#1铝壳取料位感应延时
T2881 BOOL  ; RK_07 U8_Z 铝壳上料移载Y轴#2铝壳取料位感应延时
T2882 BOOL  ; RK_07 U8_Z 铝壳上料移载Y轴#3铝壳取料位感应延时
T2900 BOOL  ; RK_13 #1移载左右定位伸缩气缸缩回[A]延迟
T2901 BOOL  ; RK_13 #2移载左右定位伸缩气缸缩回[A]延迟
T3000 BOOL  ; #1铝壳上料机构手动上料超时
T3001 BOOL  ; #2铝壳上料机构手动上料超时
T3002 BOOL  ; #3铝壳托盘下料机构手动下料超时
W0.00 BOOL  ; 启动按钮（SW）
W0.01 BOOL  ; 停止按钮(SW)
W0.02 BOOL  ; 复位按钮（SW）
W0.04 BOOL  ; 整机复位按钮（SW）
W0.05 BOOL  ; 清料停止按钮（SW）
W0.06 BOOL  ; 整机记忆清除（SW）
W0.07 BOOL  ; 门磁屏蔽（SW）
W0.08 BOOL  ; 蜂鸣器屏蔽（SW）
W0.14 BOOL  ; 铝壳进料X轴自动生成位置按钮（SW）
W0.15 BOOL  ; 铝壳上料移载Y轴自动生成位置按钮（SW）
W150.00 BOOL  ; 数据保存按钮（SW）
W150.01 BOOL  ; 数据调出按钮（SW）
W151.00 BOOL  ; 参数保存成功
W151.01 BOOL  ; 参数调出成功
W152.01 BOOL  ; #1配方使用标志
W152.02 BOOL  ; #2配方使用标志
W152.03 BOOL  ; #3配方使用标志
W152.04 BOOL  ; #4配方使用标志
W152.05 BOOL  ; #5配方使用标志
W152.06 BOOL  ; #6配方使用标志
W152.07 BOOL  ; #7配方使用标志
W152.08 BOOL  ; #8配方使用标志
W152.09 BOOL  ; #9配方使用标志
W1.00 BOOL  ; 手动模式
W1.01 BOOL  ; 自动模式
W200.00 BOOL  ; RK_01 U0_X 电芯来料Y轴回原点完成标志
W200.01 BOOL  ; RK_01 U0_X 电芯来料Y轴回原点忙标志
W200.02 BOOL  ; RK_01 U0_X 电芯来料Y轴上料位完成标志
W200.03 BOOL  ; RK_01 U0_X 电芯来料Y轴上料位忙标志
W200.04 BOOL  ; RK_01 U0_X 电芯来料Y轴下料位完成标志
W200.05 BOOL  ; RK_01 U0_X 电芯来料Y轴下料位忙标志
W201.15 BOOL  ; RK_01 U0_X 电芯来料Y轴轴忙标志
W204.00 BOOL  ; RK_01 电芯来料机构单步标志
W205.00 BOOL  ; RK_02 U0_Y 电芯进料X轴回原点完成标志
W205.01 BOOL  ; RK_02 U0_Y 电芯进料X轴回原点忙标志
W205.02 BOOL  ; RK_02 U0_Y 电芯进料X轴取料位完成标志
W205.03 BOOL  ; $?St$Bk?_#[5060] / RK_02 U0_Y 电芯进料X轴取料位忙标志 / $?St$Bk?_#[5060]
W205.04 BOOL  ; RK_02 U0_Y 电芯进料X轴扫码OK放料位完成标志
W205.05 BOOL  ; RK_02 U0_Y 电芯进料X轴扫码OK放料位忙标志
W205.06 BOOL  ; RK_02 U0_Y 电芯进料X轴扫码NG放料位完成标志
W205.07 BOOL  ; $?St$Bk?_#[5061] / RK_02 U0_Y 电芯进料X轴扫码NG放料位忙标志 / $?St$Bk?_#[5061]
W205.08 BOOL  ; RK_02 U0_Z 电芯进料Z轴回原点完成标志
W205.09 BOOL  ; RK_02 U0_Z 电芯进料Z轴回原点忙标志
W205.10 BOOL  ; RK_02 U0_Z 电芯进料Z轴待料位（扫码）完成标志
W205.11 BOOL  ; RK_02 U0_Z 电芯进料Z轴待料位（扫码）忙标志
W205.12 BOOL  ; RK_02 U0_Z 电芯进料Z轴取料位完成标志
W205.13 BOOL  ; RK_02 U0_Z 电芯进料Z轴取料位忙标志
W205.14 BOOL  ; RK_02 U0_Z 电芯进料Z轴扫码OK放料位完成标志
W205.15 BOOL  ; RK_02 U0_Z 电芯进料Z轴扫码OK放料位忙标志
W206.00 BOOL  ; RK_02 U0_Z 电芯进料Z轴扫码NG放料位完成标志
W206.01 BOOL  ; RK_02 U0_Z 电芯进料Z轴扫码NG放料位忙标志
W206.02 BOOL  ; RK_02 U0_Z 电芯进料Z轴扫码位完成标志
W206.03 BOOL  ; RK_02 U0_Z 电芯进料Z轴扫码位忙标志
W206.10 BOOL  ; RK_02 U0_Y 电芯进料X轴运行中电芯进料Z轴不在待料位（扫码）停轴标志
W206.11 BOOL  ; RK_02 U0_Z 电芯进料Z轴柔性报警后轴回初始位标志
W206.14 BOOL  ; RK_02 U0_Z 电芯进料Z轴轴忙标志
W206.15 BOOL  ; RK_02 U0_Y 电芯进料X轴轴忙标志
W209.00 BOOL  ; RK_02  电芯进料机构单步标志
W209.01 BOOL  ; 电芯进料X轴允许去放料位安全标志
W209.02 BOOL  ; 电芯进料X轴有放OK料需求标志
W209.03 BOOL  ; 电芯进料X轴有放NG料需求标志
W209.13 BOOL  ; 电芯上料X轴允许运行标志
W209.14 BOOL  ; 电芯进料X轴允许运行标志
W209.15 BOOL  ; 电芯进/上料伺服距离过小标志
W20.00 BOOL  ; RK_02 电芯进料机构夹爪有料标志
W20.01 BOOL  ; RK_04 电芯除尘机构有料标志
W20.02 BOOL  ; RK_03 电芯上料机构夹爪有料标志
W20.03 BOOL  ; RK_05 #1入壳机构有电芯标志
W20.04 BOOL  ; RK_05 #2入壳机构有电芯标志
W210.00 BOOL  ; RK_03 U0_U 电芯上料X轴回原点完成标志
W210.01 BOOL  ; RK_03 U0_U 电芯上料X轴回原点忙标志
W210.02 BOOL  ; RK_03 U0_U 电芯上料X轴待料位完成标志
W210.03 BOOL  ; RK_03 U0_U 电芯上料X轴待料位忙标志
W210.04 BOOL  ; RK_03 U0_U 电芯上料X轴取料位完成标志
W210.05 BOOL  ; RK_03 U0_U 电芯上料X轴取料位忙标志
W210.06 BOOL  ; RK_03 U0_U 电芯上料X轴#1入壳放料位完成标志
W210.07 BOOL  ; RK_03 U0_U 电芯上料X轴#1入壳放料位忙标志
W210.08 BOOL  ; RK_03 U0_U 电芯上料X轴#2入壳放料位完成标志
W210.09 BOOL  ; RK_03 U0_U 电芯上料X轴#2入壳放料位忙标志
W211.10 BOOL  ; RK_03 U0_U 电芯上料X轴运行中电芯上料升降气缸不在上升位停止伺服标志
W211.15 BOOL  ; RK_03 U0_U 电芯上料X轴轴忙标志
W214.00 BOOL  ; RK_03  电芯上料机构单步标志
W214.01 BOOL  ; 电芯上料X轴允许去取料位安全标志
W214.02 BOOL  ; 电芯上料X轴有取料需求标志
W214.03 BOOL  ; 电芯上料X轴去#1入壳放料位条件
W214.04 BOOL  ; 电芯上料X轴去#2入壳放料位条件
W219.00 BOOL  ; RK_04  电芯除尘机构单步标志
W21.00 BOOL  ; RK_07 铝壳进料机构夹爪有料标志
W21.01 BOOL  ; RK_08 铝壳除尘机构有料标志
W21.02 BOOL  ; RK_06 电池上下料机构上料夹爪有料标志
W21.03 BOOL  ; RK_05 #1入壳机构有铝壳标志
W21.04 BOOL  ; RK_05 #2入壳机构有铝壳标志
W220.00 BOOL  ; RK_05 U2_X #1入壳Y轴回原点完成标志
W220.01 BOOL  ; RK_05 U2_X #1入壳Y轴回原点忙标志
W220.02 BOOL  ; RK_05 U2_X #1入壳Y轴待料位完成标志
W220.03 BOOL  ; RK_05 U2_X #1入壳Y轴待料位忙标志
W220.04 BOOL  ; RK_05 U2_X #1入壳Y轴滚轮压紧位完成标志
W220.05 BOOL  ; RK_05 U2_X #1入壳Y轴滚轮压紧位忙标志
W220.06 BOOL  ; RK_05 U2_X #1入壳Y轴滚轮松开位完成标志
W220.07 BOOL  ; RK_05 U2_X #1入壳Y轴滚轮松开位忙标志
W220.08 BOOL  ; RK_05 U2_X #1入壳Y轴入壳位完成标志
W220.09 BOOL  ; RK_05 U2_X #1入壳Y轴入壳位忙标志
W220.10 BOOL  ; RK_05 U2_X #1入壳Y轴电芯定位夹爪松开位完成标志
W220.11 BOOL  ; RK_05 U2_X #1入壳Y轴电芯定位夹爪松开位忙标志
W221.10 BOOL  ; RK_05 #1入壳压力高报警标志
W221.15 BOOL  ; RK_05 U2_X #1入壳Y轴轴忙标志
W222.00 BOOL  ; RK_05 #1入壳机构入壳条件
W222.01 BOOL  ; RK_05 #1入壳机构入壳位到待料位条件
W224.00 BOOL  ; RK_05 #1入壳机构单步标志
W225.00 BOOL  ; RK_05 U2_Y #2入壳Y轴回原点完成标志
W225.01 BOOL  ; RK_05 U2_Y #2入壳Y轴回原点忙标志
W225.02 BOOL  ; RK_05 U2_Y #2入壳Y轴待料位完成标志
W225.03 BOOL  ; RK_05 U2_Y #2入壳Y轴待料位忙标志
W225.04 BOOL  ; RK_05 U2_Y #2入壳Y轴滚轮压紧位完成标志
W225.05 BOOL  ; RK_05 U2_Y #2入壳Y轴滚轮压紧位忙标志
W225.06 BOOL  ; RK_05 U2_Y #2入壳Y轴滚轮松开位完成标志
W225.07 BOOL  ; RK_05 U2_Y #2入壳Y轴滚轮松开位忙标志
W225.08 BOOL  ; RK_05 U2_Y #2入壳Y轴入壳位完成标志
W225.09 BOOL  ; RK_05 U2_Y #2入壳Y轴入壳位忙标志
W225.10 BOOL  ; RK_05 U2_Y #2入壳Y轴电芯定位夹爪松开位完成标志
W225.11 BOOL  ; RK_05 U2_Y #2入壳Y轴电芯定位夹爪松开位忙标志
W226.10 BOOL  ; RK_05 #2入壳压力高报警标志
W226.15 BOOL  ; RK_05 U2_Y #2入壳Y轴轴忙标志
W227.00 BOOL  ; RK_05 #2入壳机构入壳条件
W227.01 BOOL  ; RK_05 #2入壳机构入壳位到待料位条件
W229.00 BOOL  ; RK_05 #2入壳机构单步标志
W22.00 BOOL  ; 清料中铝壳进料机构运行允许标志
W230.00 BOOL  ; RK_06 U8_X 电池上下料X轴回原点完成标志
W230.01 BOOL  ; RK_06 U8_X 电池上下料X轴回原点忙标志
W230.02 BOOL  ; RK_06 U8_X 电池上下料X轴铝壳除尘取料位完成标志
W230.03 BOOL  ; RK_06 U8_X 电池上下料X轴铝壳除尘取料位忙标志
W230.04 BOOL  ; RK_06 U8_X 电池上下料X轴#1入壳放料位完成标志
W230.05 BOOL  ; RK_06 U8_X 电池上下料X轴#1入壳放料位忙标志
W230.06 BOOL  ; RK_06 U8_X 电池上下料X轴#2入壳放料位完成标志
W230.07 BOOL  ; RK_06 U8_X 电池上下料X轴#2入壳放料位忙标志
W230.08 BOOL  ; RK_06 U8_X 电池上下料X轴#1入壳取料位完成标志
W230.09 BOOL  ; RK_06 U8_X 电池上下料X轴#1入壳取料位忙标志
W230.10 BOOL  ; RK_06 U8_X 电池上下料X轴#2入壳取料位完成标志
W230.11 BOOL  ; RK_06 U8_X 电池上下料X轴#2入壳取料位忙标志
W230.12 BOOL  ; RK_06 U8_X 电池上下料X轴#1Hipot检测放料位完成标志
W230.13 BOOL  ; RK_06 U8_X 电池上下料X轴#1Hipot检测放料位忙标志
W230.14 BOOL  ; RK_06 U8_X 电池上下料X轴#2Hipot检测放料位完成标志
W230.15 BOOL  ; RK_06 U8_X 电池上下料X轴#2Hipot检测放料位忙标志
W231.10 BOOL  ; RK_06 U8_X 电池上下料X轴运行中上料升降气缸不在上升位停止伺服标志
W231.11 BOOL  ; RK_06 U8_X 电池上下料X轴运行中下料升降气缸不在上升位停止伺服标志
W231.15 BOOL  ; RK_06 U8_X 电池上下料X轴轴忙标志
W233.00 BOOL  ; RK_06 #1入壳位有上铝壳需求标志
W233.01 BOOL  ; RK_06 #2入壳位有上铝壳需求标志
W233.02 BOOL  ; RK_06 #1入壳位有下电池需求标志
W233.03 BOOL  ; RK_06 #2入壳位有下电池需求标志
W233.04 BOOL  ; RK_09 #1Hipot检测位有放电池需求
W233.05 BOOL  ; RK_09 #2Hipot检测位有放电池需求
W233.06 BOOL  ; RK_09 #1入壳位有上铝壳需求优先标志
W233.07 BOOL  ; RK_09 #2入壳位有上铝壳需求优先标志
W234.00 BOOL  ; RK_06 电池上下料机构单步标志
W235.00 BOOL  ; RK_07 U8_Y 铝壳进料X轴回原点完成标志
W235.01 BOOL  ; RK_07 U8_Y 铝壳进料X轴回原点忙标志
W235.02 BOOL  ; RK_07 U8_Y 铝壳进料X轴等待位完成标志
W235.03 BOOL  ; RK_07 U8_Y 铝壳进料X轴等待位忙标志
W235.04 BOOL  ; RK_07 U8_Y 铝壳进料X轴取料位完成标志
W235.05 BOOL  ; RK_07 U8_Y 铝壳进料X轴取料位忙标志
W235.06 BOOL  ; RK_07 U8_Y 铝壳进料X轴放料位完成标志
W235.07 BOOL  ; RK_07 U8_Y 铝壳进料X轴放料位忙标志
W236.10 BOOL  ; RK_07 U8_Y 铝壳进料X轴运行中上料升降气缸不在上升位停止伺服标志
W236.15 BOOL  ; RK_07 U8_Y 铝壳进料X轴轴忙标志
W238.00 BOOL  ; RK_07 铝壳进料机构取料位序号递增标志
W239.00 BOOL  ; RK_07 铝壳进料机构单步标志
W240.00 BOOL  ; RK_07 U8_Z 铝壳上料移载Y轴回原点完成标志
W240.01 BOOL  ; RK_07 U8_Z 铝壳上料移载Y轴回原点忙标志
W240.02 BOOL  ; RK_07 U8_Z 铝壳上料移载Y轴#1铝壳上料位完成标志
W240.03 BOOL  ; RK_07 U8_Z 铝壳上料移载Y轴#1铝壳上料位忙标志
W240.04 BOOL  ; RK_07 U8_Z 铝壳上料移载Y轴#2铝壳上料位完成标志
W240.05 BOOL  ; RK_07 U8_Z 铝壳上料移载Y轴#2铝壳上料位忙标志
W240.06 BOOL  ; RK_07 U8_Z 铝壳上料移载Y轴#3铝壳托盘下料位完成标志
W240.07 BOOL  ; RK_07 U8_Z 铝壳上料移载Y轴#3铝壳托盘下料位忙标志
W240.08 BOOL  ; RK_07 U8_Z 铝壳上料移载Y轴铝壳取料位完成标志
W240.09 BOOL  ; RK_07 U8_Z 铝壳上料移载Y轴铝壳取料位忙标志
W241.10 BOOL  ; RK_07 U8_Z 铝壳上料移载Y轴运行中铝壳进料升降气缸&铝壳上下料工位异常停止伺服标志
W241.15 BOOL  ; RK_07 U8_Z 铝壳上料移载Y轴轴忙标志
W242.00 BOOL  ; 铝壳上料移载机构Y轴#1铝壳上料位优先标志
W242.01 BOOL  ; 铝壳上料移载机构Y轴#2铝壳上料位优先标志
W242.10 BOOL  ; RK_07 #1铝壳上料电机启动标志
W242.11 BOOL  ; RK_07 #2铝壳上料电机启动标志
W242.12 BOOL  ; RK_07 #3铝壳下料电机启动标志
W243.00 BOOL  ; RK_07 铝壳上料移载机构取料位序号递增标志
W244.00 BOOL  ; RK_07 铝壳上料移载机构单步标志
W264.00 BOOL  ; RK_08 铝壳除尘机构单步标志
W265.00 BOOL  ; RK_09 Hipot测试完成信号标志
W267.02 BOOL  ; Hipot检测仪参数写入标志
W268.00 BOOL  ; #1Hipot检测机构平台伸缩气缸允许伸出优先条件
W268.01 BOOL  ; #2Hipot检测机构平台伸缩气缸允许伸出优先条件
W269.00 BOOL  ; RK_09 #1Hipot检测机构单步标志
W274.00 BOOL  ; RK_09 #2Hipot检测机构单步标志
W275.00 BOOL  ; RK_10 U8_U 电池除尘上料X轴回原点完成标志
W275.01 BOOL  ; RK_10 U8_U 电池除尘上料X轴回原点忙标志
W275.02 BOOL  ; RK_10 U8_U 电池除尘上料X轴#1Hipot检测取料位完成标志
W275.03 BOOL  ; RK_10 U8_U 电池除尘上料X轴#1Hipot检测取料位忙标志
W275.04 BOOL  ; RK_10 U8_U 电池除尘上料X轴#2Hipot检测取料位完成标志
W275.05 BOOL  ; RK_10 U8_U 电池除尘上料X轴#2Hipot检测取料位忙标志
W275.06 BOOL  ; RK_10 U8_U 电池除尘上料X轴Hipot OK放料位完成标志
W275.07 BOOL  ; RK_10 U8_U 电池除尘上料X轴Hipot OK放料位忙标志
W275.08 BOOL  ; RK_10 U8_U 电池除尘上料X轴Hipot NG放料位完成标志
W275.09 BOOL  ; RK_10 U8_U 电池除尘上料X轴Hipot NG放料位忙标志
W276.10 BOOL  ; RK_10 U8_U 电池除尘上料X轴运行中上料升降气缸不在上升位停止伺服标志
W276.15 BOOL  ; RK_10 U8_U 电池除尘上料X轴轴忙标志
W279.00 BOOL  ; RK_10 电池除尘上料机构单步标志
W279.01 BOOL  ; 电池除尘上料X轴允许去电池除尘放料位安全标志
W279.02 BOOL  ; 电池除尘上料X轴有放OK料需求标志
W279.03 BOOL  ; 电池除尘上料X轴有放NG料需求标志
W279.04 BOOL  ; #1Hipot检测取料位有取电池需求
W279.05 BOOL  ; #2Hipot检测取料位有取电池需求
W279.13 BOOL  ; 预焊上下料X轴允许运行标志
W279.14 BOOL  ; 电池除尘上料X轴允许运行标志
W279.15 BOOL  ; 电池除尘上料/预焊上下料伺服距离过小标志
W284.00 BOOL  ; RK_11 电池除尘机构单步标志
W285.00 BOOL  ; RK_12 U4_X 预焊上下料X轴回原点完成标志
W285.01 BOOL  ; RK_12 U4_X 预焊上下料X轴回原点忙标志
W285.02 BOOL  ; RK_12 U4_X 预焊上下料X轴除尘取料位完成标志
W285.03 BOOL  ; RK_12 U4_X 预焊上下料X轴除尘取料位忙标志
W285.04 BOOL  ; RK_12 U4_X 预焊上下料X轴#1移载放料位完成标志
W285.05 BOOL  ; RK_12 U4_X 预焊上下料X轴#1移载放料位忙标志
W285.06 BOOL  ; RK_12 U4_X 预焊上下料X轴#2移载放料位完成标志
W285.07 BOOL  ; RK_12 U4_X 预焊上下料X轴#2移载放料位忙标志
W285.08 BOOL  ; RK_12 U4_X 预焊上下料X轴#1移载取料位完成标志
W285.09 BOOL  ; RK_12 U4_X 预焊上下料X轴#1移载取料位忙标志
W285.10 BOOL  ; RK_12 U4_X 预焊上下料X轴#2移载取料位完成标志
W285.11 BOOL  ; RK_12 U4_X 预焊上下料X轴#2移载取料位忙标志
W285.12 BOOL  ; RK_12 U4_X 预焊上下料X轴OK放料位完成标志
W285.13 BOOL  ; RK_12 U4_X 预焊上下料X轴OK放料位忙标志
W285.14 BOOL  ; RK_12 U4_X 预焊上下料X轴#1NG放料位完成标志
W285.15 BOOL  ; RK_12 U4_X 预焊上下料X轴#1NG放料位忙标志
W286.00 BOOL  ; RK_12 U4_X 预焊上下料X轴#2NG放料位完成标志
W286.01 BOOL  ; RK_12 U4_X 预焊上下料X轴#2NG放料位忙标志
W286.02 BOOL  ; RK_12 U4_Y 预焊上料Z轴回原点完成标志
W286.03 BOOL  ; RK_12 U4_Y 预焊上料Z轴回原点忙标志
W286.04 BOOL  ; RK_12 U4_Y 预焊上料Z轴待料位完成标志
W286.05 BOOL  ; RK_12 U4_Y 预焊上料Z轴待料位忙标志
W286.06 BOOL  ; RK_12 U4_Y 预焊上料Z轴除尘取料位完成标志
W286.07 BOOL  ; RK_12 U4_Y 预焊上料Z轴除尘取料位忙标志
W286.08 BOOL  ; RK_12 U4_Y 预焊上料Z轴#1移载放料位完成标志
W286.09 BOOL  ; RK_12 U4_Y 预焊上料Z轴#1移载放料位忙标志
W286.10 BOOL  ; RK_12 U4_Y 预焊上料Z轴#2移载放料位完成标志
W286.11 BOOL  ; RK_12 U4_Y 预焊上料Z轴#2移载放料位忙标志
W286.13 BOOL  ; RK_12 U4_Z 预焊下料Z轴轴忙标志
W286.14 BOOL  ; RK_12 U4_Y 预焊上料Z轴轴忙标志
W286.15 BOOL  ; RK_12 U4_X 预焊上下料X轴轴忙标志
W287.00 BOOL  ; RK_12 U4_Z 预焊下料Z轴回原点完成标志
W287.01 BOOL  ; RK_12 U4_Z 预焊下料Z轴回原点忙标志
W287.02 BOOL  ; RK_12 U4_Z 预焊下料Z轴待料位完成标志
W287.03 BOOL  ; RK_12 U4_Z 预焊下料Z轴待料位忙标志
W287.04 BOOL  ; RK_12 U4_Z 预焊下料Z轴#1移载取料位完成标志
W287.05 BOOL  ; RK_12 U4_Z 预焊下料Z轴#1移载取料位忙标志
W287.06 BOOL  ; RK_12 U4_Z 预焊下料Z轴#2移载取料位完成标志
W287.07 BOOL  ; RK_12 U4_Z 预焊下料Z轴#2移载取料位忙标志
W287.08 BOOL  ; RK_12 U4_Z 预焊下料Z轴OK放料位完成标志
W287.09 BOOL  ; RK_12 U4_Z 预焊下料Z轴OK放料位忙标志
W287.10 BOOL  ; RK_12 U4_Z 预焊下料Z轴#1NG放料位完成标志
W287.11 BOOL  ; RK_12 U4_Z 预焊下料Z轴#1NG放料位忙标志
W287.12 BOOL  ; RK_12 U4_Z 预焊下料Z轴#2NG放料位完成标志
W287.13 BOOL  ; RK_12 U4_Z 预焊下料Z轴#2NG放料位忙标志
W287.14 BOOL  ; RK_12 U4_X 预焊上下料X轴待料位完成标志
W287.15 BOOL  ; RK_12 U4_X 预焊上下料X轴待料位忙标志
W288.08 BOOL  ; RK_12 U4_Z 预焊上料Z轴柔性报警后轴回初始位标志
W288.09 BOOL  ; RK_12 U4_Z 预焊下料Z轴柔性报警后轴回初始位标志
W288.10 BOOL  ; RK_12 U4_X 预焊上下料X轴运行中预焊上料Z轴不在待料位停轴标志
W288.11 BOOL  ; RK_12 U4_X 预焊上下料X轴运行中预焊下料Z轴不在待料位停轴标志
W288.13 BOOL  ; RK_12 U4_Z 预焊下料Z轴轴忙标志
W288.14 BOOL  ; RK_12 U4_Z 预焊上料Z轴轴忙标志
W288.15 BOOL  ; RK_12 U4_X 预焊上下料X轴轴忙标志
W289.00 BOOL  ; RK_12 预焊上下料机构单步标志
W289.01 BOOL  ; 预焊上下料X轴允许去电池除尘取料位安全标志
W289.02 BOOL  ; 预焊上下料X轴有取料需求标志
W289.03 BOOL  ; #1移载有放电池需求标志
W289.04 BOOL  ; #2移载有放电池需求标志
W289.05 BOOL  ; #1移载有取电池需求标志
W289.06 BOOL  ; #2移载有取电池需求标志
W289.07 BOOL  ; #1轮廓NG槽有放NG电池需求标志
W289.08 BOOL  ; #2轮廓NG槽有放NG电池需求标志
W289.09 BOOL  ; 出料拉带有放OK电池需求标志
W289.10 BOOL  ; #1移载放电池需求优先标志
W289.11 BOOL  ; #2移载放电池需求优先标志
W289.12 BOOL  ; 轮廓NG槽放料前拨料气缸伸缩一次标志
W289.13 BOOL  ; #1移载有取电池标志
W289.14 BOOL  ; #2移载有取电池标志（预焊电池放料工况未运行）
W289.15 BOOL  ; #2移载有取电池标志
W290.00 BOOL  ; RK_13 U4_U #1移载Y轴回原点完成标志
W290.01 BOOL  ; RK_13 U4_U #1移载Y轴回原点忙标志
W290.02 BOOL  ; RK_13 U4_U #1移载Y轴取放料位完成标志
W290.03 BOOL  ; RK_13 U4_U #1移载Y轴取放料位忙标志
W290.04 BOOL  ; RK_13 U4_U #1移载Y轴压装位完成标志
W290.05 BOOL  ; RK_13 U4_U #1移载Y轴压装位忙标志
W290.06 BOOL  ; RK_13 U4_U #1移载Y轴#1轮廓检测位完成标志
W290.07 BOOL  ; RK_13 U4_U #1移载Y轴#1轮廓检测位忙标志
W290.08 BOOL  ; RK_13 U4_U #1移载Y轴#2轮廓检测位完成标志
W290.09 BOOL  ; RK_13 U4_U #1移载Y轴#2轮廓检测位忙标志
W290.10 BOOL  ; RK_13 U4_U #1移载Y轴激光焊接位完成标志
W290.11 BOOL  ; RK_13 U4_U #1移载Y轴激光焊接位忙标志
W291.15 BOOL  ; RK_13 U4_U #1移载Y轴轴忙标志
W294.00 BOOL  ; RK_13 #1移载机构单步标志
W295.00 BOOL  ; RK_13 U6_X #2移载Y轴回原点完成标志
W295.01 BOOL  ; RK_13 U6_X #2移载Y轴回原点忙标志
W295.02 BOOL  ; RK_13 U6_X #2移载Y轴取放料位完成标志
W295.03 BOOL  ; RK_13 U6_X #2移载Y轴取放料位忙标志
W295.04 BOOL  ; RK_13 U6_X #2移载Y轴压装位完成标志
W295.05 BOOL  ; RK_13 U6_X #2移载Y轴压装位忙标志
W295.06 BOOL  ; RK_13 U6_X #2移载Y轴#1轮廓检测位完成标志
W295.07 BOOL  ; RK_13 U6_X #2移载Y轴#1轮廓检测位忙标志
W295.08 BOOL  ; RK_13 U6_X #2移载Y轴#2轮廓检测位完成标志
W295.09 BOOL  ; RK_13 U6_X #2移载Y轴#2轮廓检测位忙标志
W295.10 BOOL  ; RK_13 U6_X #2移载Y轴激光焊接位完成标志
W295.11 BOOL  ; RK_13 U6_X #2移载Y轴激光焊接位忙标志
W296.15 BOOL  ; RK_13 U6_X #2移载Y轴轴忙标志
W299.00 BOOL  ; RK_13 #2移载机构单步标志
W2.00 BOOL  ; 良品数清零按钮（SW）
W2.01 BOOL  ; 不良品数清零按钮（SW）
W304.00 BOOL  ; RK_14 #1压装机构单步标志
W309.00 BOOL  ; RK_14 #2压装机构单步标志
W310.00 BOOL  ; #1移载轮廓检测位有轮廓检测需求
W310.01 BOOL  ; #2移载轮廓检测位有轮廓检测需求
W310.08 BOOL  ; RK_15 轮廓检测机构#1移载#1轮廓测量值读取标志
W310.09 BOOL  ; RK_15 轮廓检测机构#1移载#2轮廓测量值读取标志
W310.10 BOOL  ; RK_15 轮廓检测机构#1移载#3轮廓测量值读取标志
W310.11 BOOL  ; RK_15 轮廓检测机构#1移载#4轮廓测量值读取标志
W310.12 BOOL  ; RK_15 轮廓检测机构#2移载#1轮廓测量值读取标志
W310.13 BOOL  ; RK_15 轮廓检测机构#2移载#2轮廓测量值读取标志
W310.14 BOOL  ; RK_15 轮廓检测机构#2移载#3轮廓测量值读取标志
W310.15 BOOL  ; RK_15 轮廓检测机构#2移载#4轮廓测量值读取标志
W311.00 BOOL  ; RK_15 轮廓检测机构#1移载#1/4点测量程序触发
W311.01 BOOL  ; RK_15 轮廓检测机构#1移载#2/3点测量程序触发
W311.02 BOOL  ; RK_15 轮廓检测机构#2移载#1/4点测量程序触发
W311.03 BOOL  ; RK_15 轮廓检测机构#2移载#2/3点测量程序触发
W311.04 BOOL  ; RK_15 轮廓检测机构#1点测量数据读取触发
W311.05 BOOL  ; RK_15 轮廓检测机构#2点测量数据读取触发
W311.06 BOOL  ; RK_15 轮廓检测机构#3点测量数据读取触发
W311.07 BOOL  ; RK_15 轮廓检测机构#4点测量数据读取触发
W311.08 BOOL  ; RK_15 轮廓检测机构#1移载#1轮廓测量数据浮点数|字符显示标志（浮点数显示=0）
W311.09 BOOL  ; RK_15 轮廓检测机构#1移载#2轮廓测量数据浮点数|字符显示标志（浮点数显示=0）
W311.10 BOOL  ; RK_15 轮廓检测机构#1移载#3轮廓测量数据浮点数|字符显示标志（浮点数显示=0）
W311.11 BOOL  ; RK_15 轮廓检测机构#1移载#4轮廓测量数据浮点数|字符显示标志（浮点数显示=0）
W311.12 BOOL  ; RK_15 轮廓检测机构#2移载#1轮廓测量数据浮点数|字符显示标志（浮点数显示=0）
W311.13 BOOL  ; RK_15 轮廓检测机构#2移载#2轮廓测量数据浮点数|字符显示标志（浮点数显示=0）
W311.14 BOOL  ; RK_15 轮廓检测机构#2移载#3轮廓测量数据浮点数|字符显示标志（浮点数显示=0）
W311.15 BOOL  ; RK_15 轮廓检测机构#2移载#4轮廓测量数据浮点数|字符显示标志（浮点数显示=0）
W312.00 BOOL  ; RK_15 轮廓检测机构测量程序切换触发标志
W312.01 BOOL  ; RK_15 轮廓检测机构测量数据读取触发标志
W312.08 BOOL  ; RK_15 轮廓检测机构#1移载#1点测量OK标志
W312.09 BOOL  ; RK_15 轮廓检测机构#1移载#1点测量NG标志
W312.10 BOOL  ; RK_15 轮廓检测机构#1移载#2点测量OK标志
W312.11 BOOL  ; RK_15 轮廓检测机构#1移载#2点测量NG标志
W312.12 BOOL  ; RK_15 轮廓检测机构#1移载#3点测量OK标志
W312.13 BOOL  ; RK_15 轮廓检测机构#1移载#3点测量NG标志
W312.14 BOOL  ; RK_15 轮廓检测机构#1移载#4点测量OK标志
W312.15 BOOL  ; RK_15 轮廓检测机构#1移载#4点测量NG标志
W313.00 BOOL  ; RK_15 轮廓检测机构程序切换解析完成标志
W313.01 BOOL  ; RK_15 轮廓检测机构测量数据读取解析完成标志
W313.08 BOOL  ; RK_15 轮廓检测机构#2移载#1点测量OK标志
W313.09 BOOL  ; RK_15 轮廓检测机构#2移载#1点测量NG标志
W313.10 BOOL  ; RK_15 轮廓检测机构#2移载#2点测量OK标志
W313.11 BOOL  ; RK_15 轮廓检测机构#2移载#2点测量NG标志
W313.12 BOOL  ; RK_15 轮廓检测机构#2移载#3点测量OK标志
W313.13 BOOL  ; RK_15 轮廓检测机构#2移载#3点测量NG标志
W313.14 BOOL  ; RK_15 轮廓检测机构#2移载#4点测量OK标志
W313.15 BOOL  ; RK_15 轮廓检测机构#2移载#4点测量NG标志
W314.00 BOOL  ; RK_15 轮廓检测机构单步标志
W314.02 BOOL  ; RK_15 轮廓检测机构#1移载#1轮廓测量选择（手动）
W314.03 BOOL  ; RK_15 轮廓检测机构#1移载#2轮廓测量选择（手动）
W314.04 BOOL  ; RK_15 轮廓检测机构#1移载#3轮廓测量选择（手动）
W314.05 BOOL  ; RK_15 轮廓检测机构#1移载#4轮廓测量选择（手动）
W314.06 BOOL  ; RK_15 轮廓检测机构#2移载#1轮廓测量选择（手动）
W314.07 BOOL  ; RK_15 轮廓检测机构#2移载#2轮廓测量选择（手动）
W314.08 BOOL  ; RK_15 轮廓检测机构#2移载#3轮廓测量选择（手动）
W314.09 BOOL  ; RK_15 轮廓检测机构#2移载#4轮廓测量选择（手动）
W314.10 BOOL  ; RK_15 轮廓检测机构程序切换解析异常标志
W314.11 BOOL  ; RK_15 轮廓检测机构测量数据读取解析异常标志
W315.00 BOOL  ; RK_16 U6_Y 激光焊接X轴回原点完成标志
W315.01 BOOL  ; RK_16 U6_Y 激光焊接X轴回原点忙标志
W315.02 BOOL  ; RK_16 U6_Y 激光焊接X轴#1移载焊接位完成标志
W315.03 BOOL  ; RK_16 U6_Y 激光焊接X轴#1移载焊接位忙标志
W315.04 BOOL  ; RK_16 U6_Y 激光焊接X轴#2移载焊接位完成标志
W315.05 BOOL  ; RK_16 U6_Y 激光焊接X轴#2移载焊接位忙标志
W316.00 BOOL  ; RK_16 U6_Z 激光焊接Z轴回原点完成标志
W316.01 BOOL  ; RK_16 U6_Z 激光焊接Z轴回原点忙标志
W316.02 BOOL  ; RK_16 U6_Z 激光焊接Z轴待机位完成标志
W316.03 BOOL  ; RK_16 U6_Z 激光焊接Z轴待机位忙标志
W316.04 BOOL  ; RK_16 U6_Z 激光焊接Z轴#1移载焊接位完成标志
W316.05 BOOL  ; RK_16 U6_Z 激光焊接Z轴#1移载焊接位忙标志
W316.06 BOOL  ; RK_16 U6_Z 激光焊接Z轴#2移载焊接位完成标志
W316.07 BOOL  ; RK_16 U6_Z 激光焊接Z轴#2移载焊接位忙标志
W316.10 BOOL  ; RK_16 U6_Y 激光焊接X轴运行中激光焊接Z轴不在待料位停止伺服标志
W316.14 BOOL  ; RK_16 U6_Z 激光焊接Z轴轴忙标志
W316.15 BOOL  ; RK_16 U6_Y 激光焊接X轴轴忙标志
W318.00 BOOL  ; #1移载焊接位有焊接需求
W318.01 BOOL  ; #2移载焊接位有焊接需求
W319.00 BOOL  ; RK_16 焊接机构单步标志
W320.02 BOOL  ; RK_15 轮廓检测机构#1移载#1轮廓测量允许（手动）
W320.03 BOOL  ; RK_15 轮廓检测机构#1移载#2轮廓测量允许（手动）
W320.04 BOOL  ; RK_15 轮廓检测机构#1移载#3轮廓测量允许（手动）
W320.05 BOOL  ; RK_15 轮廓检测机构#1移载#4轮廓测量允许（手动）
W320.06 BOOL  ; RK_15 轮廓检测机构#2移载#1轮廓测量允许（手动）
W320.07 BOOL  ; RK_15 轮廓检测机构#2移载#2轮廓测量允许（手动）
W320.08 BOOL  ; RK_15 轮廓检测机构#2移载#3轮廓测量允许（手动）
W320.09 BOOL  ; RK_15 轮廓检测机构#2移载#4轮廓测量允许（手动）
W3.00 BOOL  ; 上游设备运行允许（SW）（屏蔽=1）
W3.01 BOOL  ; 下游设备放料允许（SW）（屏蔽=1）
W400.00 BOOL  ; RK_02 电芯进料机械手夹爪气缸夹紧位[alm]
W400.01 BOOL  ; RK_02 电芯进料机械手夹爪气缸张开位[alm]
W400.02 BOOL  ; RK_02 电芯进料机械手#1压紧气缸松开位[alm]
W400.03 BOOL  ; RK_02 电芯进料机械手#2压紧气缸松开位[alm]
W400.04 BOOL  ; RK_03 电芯上料机械手夹爪气缸夹紧位[alm]
W400.05 BOOL  ; RK_03 电芯上料机械手夹爪气缸张开位[alm]
W400.06 BOOL  ; RK_03 电芯上料机械手#1压紧气缸松开位[alm]
W400.07 BOOL  ; RK_03 电芯上料机械手#2压紧气缸松开位[alm]
W400.08 BOOL  ; RK_03 电芯上料升降气缸下降位[alm]
W400.09 BOOL  ; RK_03 电芯上料升降气缸上升位[alm]
W400.10 BOOL  ; RK_04 电芯除尘伸缩气缸缩回位[alm]
W400.11 BOOL  ; RK_04 电芯除尘伸缩气缸伸出位[alm]
W400.12 BOOL  ; RK_05 #1入壳滚轮夹紧气缸夹紧位[alm]
W400.13 BOOL  ; RK_05 #1入壳滚轮夹紧气缸松开位[alm]
W400.14 BOOL  ; RK_05 #1入壳铝壳定位平台伸缩气缸缩回位[alm]
W400.15 BOOL  ; RK_05 #1入壳铝壳定位平台伸缩气缸伸出位[alm]
W401.00 BOOL  ; RK_05 #1入壳铝壳定位平台升降气缸上升位[alm]
W401.01 BOOL  ; RK_05 #1入壳铝壳定位平台升降气缸下降位[alm]
W401.02 BOOL  ; RK_05 #1入壳铝壳定位伸缩气缸缩回位[alm]
W401.03 BOOL  ; RK_05 #1入壳铝壳定位伸缩气缸伸出位[alm]
W401.04 BOOL  ; RK_05 #1入壳铝壳定位夹爪气缸夹紧位[alm]
W401.05 BOOL  ; RK_05 #1入壳铝壳定位夹爪气缸张开位[alm]
W401.06 BOOL  ; RK_05 #2入壳滚轮夹紧气缸夹紧位[alm]
W401.07 BOOL  ; RK_05 #2入壳滚轮夹紧气缸松开位[alm]
W401.08 BOOL  ; RK_05 #2入壳铝壳定位平台伸缩气缸缩回位[alm]
W401.09 BOOL  ; RK_05 #2入壳铝壳定位平台伸缩气缸伸出位[alm]
W401.10 BOOL  ; RK_05 #2入壳铝壳定位平台升降气缸上升位[alm]
W401.11 BOOL  ; RK_05 #2入壳铝壳定位平台升降气缸下降位[alm]
W401.12 BOOL  ; RK_05 #2入壳铝壳定位伸缩气缸缩回位[alm]
W401.13 BOOL  ; RK_05 #2入壳铝壳定位伸缩气缸伸出位[alm]
W401.14 BOOL  ; RK_05 #2入壳铝壳定位夹爪气缸夹紧位[alm]
W401.15 BOOL  ; RK_05 #2入壳铝壳定位夹爪气缸张开位[alm]
W402.00 BOOL  ; RK_01 U0_X 电芯来料Y轴报警信号[alm]
W402.01 BOOL  ; RK_01 U0_X 电芯来料Y轴准备好了信号[alm]
W402.02 BOOL  ; RK_02 U0_Y 电芯进料X轴报警信号[alm]
W402.03 BOOL  ; RK_02 U0_Y 电芯进料X轴准备好了信号[alm]
W402.04 BOOL  ; RK_02 U0_Z 电芯进料Z轴报警信号[alm]
W402.05 BOOL  ; RK_02 U0_Z 电芯进料Z轴准备好了信号[alm]
W402.06 BOOL  ; RK_03 U0_U 电芯上料X轴报警信号[alm]
W402.07 BOOL  ; RK_03 U0_U 电芯上料X轴准备好了信号[alm]
W402.08 BOOL  ; RK_05 U2_X #1入壳Y轴报警信号[alm]
W402.09 BOOL  ; RK_05 U2_X #1入壳Y轴准备好了信号[alm]
W402.10 BOOL  ; RK_05 U2_Y #2入壳Y轴报警信号[alm]
W402.11 BOOL  ; RK_05 U2_Y #2入壳Y轴准备好了信号[alm]
W402.12 BOOL  ; 0[alm]
W402.13 BOOL  ; RK_05 #1入壳定位陶瓷棒上#1夹紧气缸伸出位[alm]
W402.14 BOOL  ; RK_05 #1入壳定位陶瓷棒上#2夹紧气缸伸出位[alm]
W402.15 BOOL  ; RK_05 #1入壳定位陶瓷棒下#1夹紧气缸伸出位[alm]
W403.00 BOOL  ; RK_05 #1入壳定位陶瓷棒下#2夹紧气缸伸出位[alm]
W403.01 BOOL  ; RK_05 #1入壳定位陶瓷棒上#1夹紧气缸缩回位[alm]
W403.02 BOOL  ; RK_05 #1入壳定位陶瓷棒上#2夹紧气缸缩回位[alm]
W403.03 BOOL  ; RK_05 #1入壳定位陶瓷棒下#1夹紧气缸缩回位[alm]
W403.04 BOOL  ; RK_05 #1入壳定位陶瓷棒下#2夹紧气缸缩回位[alm]
W403.05 BOOL  ; RK_05 #1入壳吸盘上#1伸缩气缸缩回位[alm]
W403.06 BOOL  ; RK_05 #1入壳吸盘上#2伸缩气缸缩回位[alm]
W403.07 BOOL  ; RK_05 #1入壳吸盘上#3伸缩气缸缩回位[alm]
W403.08 BOOL  ; RK_05 #1入壳吸盘下#1伸缩气缸缩回位[alm]
W403.09 BOOL  ; RK_05 #1入壳吸盘下#2伸缩气缸缩回位[alm]
W403.10 BOOL  ; RK_05 #1入壳吸盘下#3伸缩气缸缩回位[alm]
W403.11 BOOL  ; RK_05 #1入壳电芯#1定位夹爪气缸松开位[alm]
W403.12 BOOL  ; RK_05 #1入壳电芯#2定位夹爪气缸松开位[alm]
W403.13 BOOL  ; RK_05 #1入壳电芯#1定位夹爪气缸夹紧位[alm]
W403.14 BOOL  ; RK_05 #1入壳电芯#2定位夹爪气缸夹紧位[alm]
W403.15 BOOL  ; RK_05 #2入壳定位陶瓷棒上#1夹紧气缸伸出位[alm]
W404.00 BOOL  ; RK_05 #2入壳定位陶瓷棒上#2夹紧气缸伸出位[alm]
W404.01 BOOL  ; RK_05 #2入壳定位陶瓷棒下#1夹紧气缸伸出位[alm]
W404.02 BOOL  ; RK_05 #2入壳定位陶瓷棒下#2夹紧气缸伸出位[alm]
W404.03 BOOL  ; RK_05 #2入壳定位陶瓷棒上#1夹紧气缸缩回位[alm]
W404.04 BOOL  ; RK_05 #2入壳定位陶瓷棒上#2夹紧气缸缩回位[alm]
W404.05 BOOL  ; RK_05 #2入壳定位陶瓷棒下#1夹紧气缸缩回位[alm]
W404.06 BOOL  ; RK_05 #2入壳定位陶瓷棒下#2夹紧气缸缩回位[alm]
W404.07 BOOL  ; RK_05 #2入壳吸盘上#1伸缩气缸缩回位[alm]
W404.08 BOOL  ; RK_05 #2入壳吸盘上#2伸缩气缸缩回位[alm]
W404.09 BOOL  ; RK_05 #2入壳吸盘上#3伸缩气缸缩回位[alm]
W404.10 BOOL  ; RK_05 #2入壳吸盘下#1伸缩气缸缩回位[alm]
W404.11 BOOL  ; RK_05 #2入壳吸盘下#2伸缩气缸缩回位[alm]
W404.12 BOOL  ; RK_05 #2入壳吸盘下#3伸缩气缸缩回位[alm]
W404.13 BOOL  ; RK_05 #2入壳电芯#1定位夹爪气缸松开位[alm]
W404.14 BOOL  ; RK_05 #2入壳电芯#2定位夹爪气缸松开位[alm]
W404.15 BOOL  ; RK_05 #2入壳电芯#1定位夹爪气缸夹紧位[alm]
W405.00 BOOL  ; RK_05 #2入壳电芯#2定位夹爪气缸夹紧位[alm]
W405.01 BOOL  ; RK_01 电芯来料有料感应[alm]
W405.02 BOOL  ; RK_02 电芯进料机械手夹爪柔性报警[alm]
W405.03 BOOL  ; RK_03 电芯上料机械手夹爪柔性报警[alm]
W405.04 BOOL  ; RK_04 电芯除尘有料感应[alm]
W405.05 BOOL  ; RK_02 扫码NG拉带有料感应#1[alm]
W405.06 BOOL  ; RK_02 扫码NG拉带有料感应#2[alm]
W405.07 BOOL  ; RK_02 扫码NG拉带料满感应[alm]
W405.08 BOOL  ; RK_05 #1入壳电芯有料感应[alm]
W405.09 BOOL  ; RK_05 #1入壳铝壳有料感应[alm]
W405.10 BOOL  ; RK_05 #2入壳电芯有料感应[alm]
W405.11 BOOL  ; RK_05 #2入壳铝壳有料感应[alm]
W405.12 BOOL  ; RK_05 #1入壳吸盘立真空[alm]
W405.13 BOOL  ; RK_05 #2入壳吸盘立真空[alm]
W405.14 BOOL  ; 前端设备对接输入信号（公共）[alm]
W405.15 BOOL  ; 后端设备对接输入信号（公共）[alm]
W406.00 BOOL  ; 小屏插入信号（公共）[alm]
W406.01 BOOL  ; NC433模块DC5V电源信号（公共）[alm]
W406.02 BOOL  ; DC24V伺服刹车电源信号（公共）[alm]
W406.03 BOOL  ; 出料端急停（公共）[alm]
W406.04 BOOL  ; 小移动屏急停（公共）[alm]
W406.05 BOOL  ; A机架#1门磁（公共）[alm]
W406.06 BOOL  ; A机架#2门磁（公共）[alm]
W406.07 BOOL  ; A机架#3门磁（公共）[alm]
W406.08 BOOL  ; A机架#4门磁（公共）[alm]
W406.09 BOOL  ; A机架#5门磁（公共）[alm]
W406.10 BOOL  ; A机架#6门磁（公共）[alm]
W406.11 BOOL  ; A机架#7门磁（公共）[alm]
W406.12 BOOL  ; A机架#8门磁（公共）[alm]
W406.13 BOOL  ; A机架#9门磁（公共）[alm]
W406.14 BOOL  ; 0[alm]
W406.15 BOOL  ; 0[alm]
W407.00 BOOL  ; 0[alm]
W407.01 BOOL  ; 0[alm]
W407.02 BOOL  ; 0[alm]
W407.03 BOOL  ; 0[alm]
W407.04 BOOL  ; 0[alm]
W407.05 BOOL  ; 0[alm]
W407.06 BOOL  ; 0[alm]
W407.07 BOOL  ; 0[alm]
W407.08 BOOL  ; 0[alm]
W407.09 BOOL  ; 0[alm]
W407.10 BOOL  ; 0[alm]
W407.11 BOOL  ; 0[alm]
W407.12 BOOL  ; 0[alm]
W407.13 BOOL  ; 0[alm]
W407.14 BOOL  ; 0[alm]
W407.15 BOOL  ; 0[alm]
W408.00 BOOL  ; RK_11 电池除尘旋转伸缩气缸到位[alm]
W408.01 BOOL  ; RK_11 电池除尘旋转伸缩气缸原位[alm]
W408.02 BOOL  ; RK_11 电池除尘伸缩气缸伸出位[alm]
W408.03 BOOL  ; RK_11 电池除尘伸缩气缸缩回位[alm]
W408.04 BOOL  ; RK_11 电池除尘夹爪气缸夹紧位[alm]
W408.05 BOOL  ; RK_11 电池除尘夹爪气缸张开位[alm]
W408.06 BOOL  ; RK_12 预焊上料机械手夹爪气缸夹紧位[alm]
W408.07 BOOL  ; RK_12 预焊上料机械手夹爪气缸张开位[alm]
W408.08 BOOL  ; RK_12 预焊下料机械手夹爪气缸夹紧位[alm]
W408.09 BOOL  ; RK_12 预焊下料机械手夹爪气缸张开位[alm]
W408.10 BOOL  ; RK_13 #1移载升降气缸上升位[alm]
W408.11 BOOL  ; RK_13 #1移载升降气缸下降位[alm]
W408.12 BOOL  ; RK_13 #1移载定位#1伸缩气缸缩回位[alm]
W408.13 BOOL  ; RK_13 #1移载定位#1伸缩气缸伸出位[alm]
W408.14 BOOL  ; $?St$Bk?_#[5062] / RK_13 #1移载定位#2伸缩气缸缩回位[alm] / RK_13 #1移载定位#2伸缩气缸缩回位[alm] / $?St$Bk?_#[5062]
W408.15 BOOL  ; RK_13 #1移载定位#2伸缩气缸伸出位[alm]
W409.00 BOOL  ; RK_13 #1移载导向#1伸缩气缸伸出位[alm]
W409.01 BOOL  ; RK_13 #1移载导向#1伸缩气缸缩回位[alm]
W409.02 BOOL  ; RK_13 #1移载导向#2伸缩气缸伸出位[alm]
W409.03 BOOL  ; RK_13 #1移载导向#2伸缩气缸缩回位[alm]
W409.04 BOOL  ; RK_13 #1移载左右定位伸缩气缸伸出位[alm]
W409.05 BOOL  ; RK_13 #1移载左右定位伸缩气缸缩回位[alm]
W409.06 BOOL  ; RK_13 #2移载升降气缸上升位[alm]
W409.07 BOOL  ; RK_13 #2移载升降气缸下降位[alm]
W409.08 BOOL  ; RK_13 #2移载定位#1伸缩气缸缩回位[alm]
W409.09 BOOL  ; RK_13 #2移载定位#1伸缩气缸伸出位[alm]
W409.10 BOOL  ; RK_13 #2移载定位#2伸缩气缸缩回位[alm]
W409.11 BOOL  ; RK_13 #2移载定位#2伸缩气缸伸出位[alm]
W409.12 BOOL  ; RK_13 #2移载导向#1伸缩气缸伸出位[alm]
W409.13 BOOL  ; RK_13 #2移载导向#1伸缩气缸缩回位[alm]
W409.14 BOOL  ; RK_13 #2移载导向#2伸缩气缸伸出位[alm]
W409.15 BOOL  ; RK_13 #2移载导向#2伸缩气缸缩回位[alm]
W410.00 BOOL  ; RK_13 #2移载左右定位伸缩气缸伸出位[alm]
W410.01 BOOL  ; RK_13 #2移载左右定位伸缩气缸缩回位[alm]
W410.02 BOOL  ; RK_14 #1压装升降气缸下降位[alm]
W410.03 BOOL  ; RK_14 #1压装升降气缸上升位[alm]
W410.04 BOOL  ; RK_14 #1压装#1吸盘升降气缸下降位[alm]
W410.05 BOOL  ; RK_14 #1压装#1吸盘升降气缸上升位[alm]
W410.06 BOOL  ; RK_14 #1压装#2吸盘升降气缸下降位[alm]
W410.07 BOOL  ; RK_14 #1压装#2吸盘升降气缸上升位[alm]
W410.08 BOOL  ; RK_14 #2压装升降气缸下降位[alm]
W410.09 BOOL  ; RK_14 #2压装升降气缸上升位[alm]
W410.10 BOOL  ; RK_14 #2压装#1吸盘升降气缸下降位[alm]
W410.11 BOOL  ; RK_14 #2压装#1吸盘升降气缸上升位[alm]
W410.12 BOOL  ; RK_14 #2压装#2吸盘升降气缸下降位[alm]
W410.13 BOOL  ; RK_14 #2压装#2吸盘升降气缸上升位[alm]
W410.14 BOOL  ; RK_15 轮廓检测#1伸缩气缸伸出位[alm]
W410.15 BOOL  ; RK_15 轮廓检测#1伸缩气缸缩回位[alm]
W411.00 BOOL  ; RK_15 轮廓检测#2伸缩气缸伸出位[alm]
W411.01 BOOL  ; RK_15 轮廓检测#2伸缩气缸缩回位[alm]
W411.02 BOOL  ; RK_12 轮廓检测NG拨料气缸伸出位[alm]
W411.03 BOOL  ; RK_12 轮廓检测NG拨料气缸缩回位[alm]
W411.04 BOOL  ; RK_11 电池除尘有料感应[alm]
W411.05 BOOL  ; RK_12 预焊上料机械手夹爪柔性报警[alm]
W411.06 BOOL  ; RK_12 预焊下料机械手夹爪柔性报警[alm]
W411.07 BOOL  ; RK_16 激光焊接完成信号[alm]
W411.08 BOOL  ; RK_16 激光焊机故障信号[alm]
W411.09 BOOL  ; RK_13 #1移载电池顶盖超高检测[alm]
W411.10 BOOL  ; RK_16 激光焊机急停信号[alm]
W411.11 BOOL  ; RK_13 #2移载电池顶盖超高检测[alm]
W411.12 BOOL  ; RK_13 #1移载有料感应[alm]
W411.13 BOOL  ; RK_13 #2移载有料感应[alm]
W411.14 BOOL  ; RK_14 #1压装吸盘立真空[alm]
W411.15 BOOL  ; RK_14 #2压装吸盘立真空[alm]
W412.00 BOOL  ; RK_12 U4_X 预焊上下料X轴报警信号[alm]
W412.01 BOOL  ; RK_12 U4_X 预焊上下料X轴准备好了信号[alm]
W412.02 BOOL  ; RK_12 U4_Y 预焊上料Z轴报警信号[alm]
W412.03 BOOL  ; RK_12 U4_Y 预焊上料Z轴准备好了信号[alm]
W412.04 BOOL  ; RK_12 U4_Z 预焊下料Z轴报警信号[alm]
W412.05 BOOL  ; RK_12 U4_Z 预焊下料Z轴准备好了信号[alm]
W412.06 BOOL  ; RK_13 U4_U #1移载Y轴报警信号[alm]
W412.07 BOOL  ; RK_13 U4_U #1移载Y轴准备好了信号[alm]
W412.08 BOOL  ; RK_13 U6_X #2移载Y轴报警信号[alm]
W412.09 BOOL  ; RK_13 U6_X #2移载Y轴准备好了信号[alm]
W412.10 BOOL  ; RK_16 U6_Y 激光焊接X轴报警信号[alm]
W412.11 BOOL  ; RK_16 U6_Y 激光焊接X轴准备好了信号[alm]
W412.12 BOOL  ; RK_16 U6_Z 激光焊接Z轴报警信号[alm]
W412.13 BOOL  ; RK_16 U6_Z 激光焊接Z轴准备好了信号[alm]
W412.14 BOOL  ; 0[alm]
W412.15 BOOL  ; 0[alm]
W413.00 BOOL  ; 0[alm]
W413.01 BOOL  ; RK_12 轮廓检测NG料槽#1有料感应[alm]
W413.02 BOOL  ; RK_12 轮廓检测NG料槽#1料满感应[alm]
W413.03 BOOL  ; RK_12 轮廓检测NG料槽#2有料感应[alm]
W413.04 BOOL  ; RK_12 轮廓检测NG料槽#2料满感应[alm]
W413.05 BOOL  ; RK_12 OK出料拉带放料位有料感应#1[alm]
W413.06 BOOL  ; RK_12 OK出料拉带放料位有料感应#2[alm]
W413.07 BOOL  ; RK_12 OK出料拉带出料位有料感应[alm]
W413.08 BOOL  ; 0[alm]
W413.09 BOOL  ; 0[alm]
W413.10 BOOL  ; 0[alm]
W413.11 BOOL  ; 0[alm]
W413.12 BOOL  ; 0[alm]
W413.13 BOOL  ; 0[alm]
W413.14 BOOL  ; 0[alm]
W413.15 BOOL  ; 0[alm]
W414.00 BOOL  ; RK_06 铝壳上料升降气缸下降位[alm]
W414.01 BOOL  ; RK_06 铝壳上料升降气缸上升位[alm]
W414.02 BOOL  ; RK_06 电池下料升降气缸下降位[alm]
W414.03 BOOL  ; RK_06 电池下料升降气缸上升位[alm]
W414.04 BOOL  ; RK_06 铝壳上料夹爪气缸夹紧位[alm]
W414.05 BOOL  ; RK_06 铝壳上料夹爪气缸张开位[alm]
W414.06 BOOL  ; RK_06 电池下料夹爪气缸夹紧位[alm]
W414.07 BOOL  ; RK_06 电池下料夹爪气缸张开位[alm]
W414.08 BOOL  ; RK_07 #1铝壳上料车定位升降气缸上升位[alm]
W414.09 BOOL  ; RK_07 #1铝壳上料车定位升降气缸下降位[alm]
W414.10 BOOL  ; RK_07 #2铝壳上料车定位升降气缸上升位[alm]
W414.11 BOOL  ; RK_07 #2铝壳上料车定位升降气缸下降位[alm]
W414.12 BOOL  ; RK_07 #3托盘下料车定位升降气缸上升位[alm]
W414.13 BOOL  ; RK_07 #3托盘下料车定位升降气缸下降位[alm]
W414.14 BOOL  ; RK_07 铝壳进料机械手升降气缸下降位[alm]
W414.15 BOOL  ; RK_07 铝壳进料机械手升降气缸上升位[alm]
W415.00 BOOL  ; RK_08 铝壳除尘旋转伸缩气缸原位[alm]
W415.01 BOOL  ; RK_08 铝壳除尘旋转伸缩气缸到位[alm]
W415.02 BOOL  ; RK_08 铝壳除尘伸缩气缸伸出位[alm]
W415.03 BOOL  ; RK_08 铝壳除尘伸缩气缸缩回位[alm]
W415.04 BOOL  ; RK_08 铝壳除尘夹爪气缸夹紧位[alm]
W415.05 BOOL  ; RK_08 铝壳除尘夹爪气缸张开位[alm]
W415.06 BOOL  ; RK_09 #1Hipot测试旋转伸缩气缸到位[alm]
W415.07 BOOL  ; RK_09 #1Hipot测试旋转伸缩气缸原位[alm]
W415.08 BOOL  ; RK_09 #1Hipot测试平台伸缩气缸缩回位[alm]
W415.09 BOOL  ; RK_09 #1Hipot测试平台伸缩气缸伸出位[alm]
W415.10 BOOL  ; RK_09 #1Hipot测试伸缩气缸伸出位[alm]
W415.11 BOOL  ; RK_09 #1Hipot测试伸缩气缸缩回位[alm]
W415.12 BOOL  ; RK_09 #2Hipot测试旋转伸缩气缸到位[alm]
W415.13 BOOL  ; RK_09 #2Hipot测试旋转伸缩气缸原位[alm]
W415.14 BOOL  ; RK_09 #2Hipot测试平台伸缩气缸缩回位[alm]
W415.15 BOOL  ; RK_09 #2Hipot测试平台伸缩气缸伸出位[alm]
W416.00 BOOL  ; RK_09 #2Hipot测试伸缩气缸伸出位[alm]
W416.01 BOOL  ; RK_09 #2Hipot测试伸缩气缸缩回位[alm]
W416.02 BOOL  ; RK_10 电池除尘上料机械手升降气缸下降位[alm]
W416.03 BOOL  ; RK_10 电池除尘上料机械手升降气缸上升位[alm]
W416.04 BOOL  ; RK_10 电池除尘上料机械手夹爪气缸夹紧位[alm]
W416.05 BOOL  ; RK_10 电池除尘上料机械手夹爪气缸张开位[alm]
W416.06 BOOL  ; RK_06 U8_X 电池上下料X轴报警信号[alm]
W416.07 BOOL  ; RK_06 U8_X 电池上下料X轴准备好了信号[alm]
W416.08 BOOL  ; RK_07 U8_Y 铝壳进料X轴报警信号[alm]
W416.09 BOOL  ; RK_07 U8_Y 铝壳进料X轴准备好了信号[alm]
W416.10 BOOL  ; RK_07 U8_Z 铝壳上料移载Y轴报警信号[alm]
W416.11 BOOL  ; RK_07 U8_Z 铝壳上料移载Y轴准备好了信号[alm]
W416.12 BOOL  ; RK_10 U8_U 电池除尘上料X轴报警信号[alm]
W416.13 BOOL  ; RK_10 U8_U 电池除尘上料X轴准备好了信号[alm]
W416.14 BOOL  ; RK_09 Hipot测试完成信号[alm]
W416.15 BOOL  ; RK_07 #1铝壳上料启动按钮[alm]
W417.00 BOOL  ; RK_07 #2铝壳上料启动按钮[alm]
W417.01 BOOL  ; RK_07 #3托盘下料启动按钮[alm]
W417.02 BOOL  ; RK_07 铝壳上料移载吸盘立真空[alm]
W417.03 BOOL  ; RK_07 铝壳进料吸盘立真空[alm]
W417.04 BOOL  ; RK_07 #1铝壳上料托盘到位感应[alm]
W417.05 BOOL  ; RK_07 #1铝壳上料位物料车到位感应[alm]
W417.06 BOOL  ; RK_07 #1铝壳上料初始位（#1）[alm]
W417.07 BOOL  ; RK_07 #1铝壳上料一个托盘位（#2）[alm]
W417.08 BOOL  ; RK_07 #1铝壳上料高限位（#3）[alm]
W417.09 BOOL  ; RK_07 #2铝壳上料托盘到位感应[alm]
W417.10 BOOL  ; RK_07 #2铝壳上料位物料车到位感应[alm]
W417.11 BOOL  ; RK_07 #2铝壳上料初始位（#1）[alm]
W417.12 BOOL  ; RK_07 #2铝壳上料一个托盘位（#2）[alm]
W417.13 BOOL  ; RK_07 #2铝壳上料高限位（#3）[alm]
W417.14 BOOL  ; RK_07 #3托盘下料上升到位感应[alm]
W417.15 BOOL  ; RK_07 #3托盘下料位物料车到位感应[alm]
W418.00 BOOL  ; RK_07 #3托盘下料初始位（#1）[alm]
W418.01 BOOL  ; RK_07 #3托盘下料一个托盘位（#2）[alm]
W418.02 BOOL  ; RK_07 #3托盘下料高限位（#3）[alm]
W418.03 BOOL  ; RK_07 铝壳上料移载托盘到位感应[alm]
W418.04 BOOL  ; RK_08 铝壳除尘有料感应[alm]
W418.05 BOOL  ; RK_09 #1Hipot测试有料感应[alm]
W418.06 BOOL  ; RK_09 #2Hipot测试有料感应[alm]
W418.07 BOOL  ; RK_10 Hipot检测NG拉带有料感应#1[alm]
W418.08 BOOL  ; RK_10 Hipot检测NG拉带有料感应#2[alm]
W418.09 BOOL  ; RK_10 Hipot检测NG拉带料满感应[alm]
W418.10 BOOL  ; RK_06 铝壳上料夹爪柔性报警[alm]
W418.11 BOOL  ; RK_06 电池下料夹爪柔性报警[alm]
W418.12 BOOL  ; RK_07 铝壳进料机械手柔性报警[alm]
W418.13 BOOL  ; RK_10 电池除尘上料机械手夹爪柔性报警[alm]
W418.14 BOOL  ; 手/自动选择（公共）[alm]
W418.15 BOOL  ; 启动按钮_绿（公共）[alm]
W419.00 BOOL  ; 停止按钮_红（公共）[alm]
W419.01 BOOL  ; 复位按钮_黄（公共）[alm]
W419.02 BOOL  ; 机台进气压力（正压）（公共）[alm]
W419.03 BOOL  ; 机台进气压力（负压）（公共）[alm]
W419.04 BOOL  ; 主屏急停（公共）[alm]
W419.05 BOOL  ; 铝壳上料端急停（公共）[alm]
W419.06 BOOL  ; HipotNG端急停（公共）[alm]
W419.07 BOOL  ; B机架#1门磁（公共）[alm]
W419.08 BOOL  ; B机架#2门磁（公共）[alm]
W419.09 BOOL  ; B机架#3门磁（公共）[alm]
W419.10 BOOL  ; B机架#4门磁（公共）[alm]
W419.11 BOOL  ; B机架#5门磁（公共）[alm]
W419.12 BOOL  ; B机架#6门磁（公共）[alm]
W419.13 BOOL  ; RK_07 #3托盘下料下降到位感应[alm]
W419.15 BOOL  ; $?St$Bk?_#[5063] / RK_07 铝壳上料移载托盘到位保护感应[alm] / $?St$Bk?_#[5063]
W420.02 BOOL  ; RK_02 电芯进料机械手#1压紧气缸压紧位[alm]
W420.03 BOOL  ; RK_02 电芯进料机械手#2压紧气缸压紧位[alm]
W420.06 BOOL  ; RK_03 电芯上料机械手#1压紧气缸压紧位[alm]
W420.07 BOOL  ; RK_03 电芯上料机械手#2压紧气缸压紧位[alm]
W421.00 BOOL  ; RK_05 #1入壳压力高[alm]
W421.01 BOOL  ; RK_05 #2入壳压力高[alm]
W422.00 BOOL  ; RK_01 U0_X 电芯来料Y轴无原点信号[alm]
W422.01 BOOL  ; RK_02 U0_Y 电芯进料X轴无原点信号[alm]
W422.02 BOOL  ; RK_02 U0_Z 电芯进料Z轴无原点信号[alm]
W422.03 BOOL  ; RK_03 U0_U 电芯上料X轴无原点信号[alm]
W422.04 BOOL  ; RK_05 U2_X #1入壳Y轴无原点信号[alm]
W422.05 BOOL  ; RK_05 U2_Y #2入壳Y轴无原点信号[alm]
W422.06 BOOL  ; RK_12 U4_X 预焊上下料X轴无原点信号[alm]
W422.07 BOOL  ; RK_12 U4_Y 预焊上料Z轴无原点信号[alm]
W422.08 BOOL  ; RK_12 U4_Z 预焊下料Z轴无原点信号[alm]
W422.09 BOOL  ; RK_13 U4_U #1移载Y轴无原点信号[alm]
W422.10 BOOL  ; RK_13 U6_X #2移载Y轴无原点信号[alm]
W422.11 BOOL  ; RK_16 U6_Y 激光焊接X轴无原点信号[alm]
W422.12 BOOL  ; RK_16 U6_Z 激光焊接Z轴无原点信号[alm]
W422.13 BOOL  ; RK_06 U8_X 电池上下料X轴无原点信号[alm]
W422.14 BOOL  ; RK_07 U8_Y 铝壳进料X轴无原点信号[alm]
W422.15 BOOL  ; RK_07 U8_Z 铝壳上料移载Y轴无原点信号[alm]
W423.00 BOOL  ; RK_10 U8_U 电池除尘上料X轴无原点信号[alm]
W423.01 BOOL  ; 扫码阻挡#1伸出输出报警
W423.02 BOOL  ; 扫码阻挡#1缩回输出报警
W423.03 BOOL  ; 扫码阻挡#2伸出输出报警
W423.04 BOOL  ; 扫码阻挡#2缩回输出报警
W423.05 BOOL  ; RK_05 #1入壳吸盘上#1伸缩气缸伸出位[alm]
W423.06 BOOL  ; RK_05 #1入壳吸盘上#2伸缩气缸伸出位[alm]
W423.07 BOOL  ; RK_05 #1入壳吸盘上#3伸缩气缸伸出位[alm]
W423.08 BOOL  ; RK_05 #1入壳吸盘下#1伸缩气缸伸出位[alm]
W423.09 BOOL  ; RK_05 #1入壳吸盘下#2伸缩气缸伸出位[alm]
W423.10 BOOL  ; RK_05 #1入壳吸盘下#3伸缩气缸伸出位[alm]
W424.07 BOOL  ; RK_05 #2入壳吸盘上#1伸缩气缸伸出位[alm]
W424.08 BOOL  ; RK_05 #2入壳吸盘上#2伸缩气缸伸出位[alm]
W424.09 BOOL  ; RK_05 #2入壳吸盘上#3伸缩气缸伸出位[alm]
W424.10 BOOL  ; RK_05 #2入壳吸盘下#1伸缩气缸伸出位[alm]
W424.11 BOOL  ; RK_05 #2入壳吸盘下#2伸缩气缸伸出位[alm]
W424.12 BOOL  ; RK_05 #2入壳吸盘下#3伸缩气缸伸出位[alm]
W425.02 BOOL  ; RK_07 铝壳上料移载吸盘破真空[alm]
W425.03 BOOL  ; RK_07 铝壳进料吸盘破真空[alm]
W425.12 BOOL  ; RK_05 #1入壳吸盘破真空[alm]
W425.13 BOOL  ; RK_05 #2入壳吸盘破真空[alm]
W425.14 BOOL  ; RK_14 #1压装吸盘破真空[alm]
W425.15 BOOL  ; RK_14 #2压装吸盘破真空[alm]
W427.00 BOOL  ; RK_01 电芯来料机构复位超时[alm]
W427.01 BOOL  ; RK_02 电芯进料机构复位超时[alm]
W427.02 BOOL  ; RK_03 电芯上料机构复位超时复位超时[alm]
W427.03 BOOL  ; RK_04 电芯除尘机构复位超时复位超时[alm]
W427.04 BOOL  ; RK_05 #1入壳机构复位超时复位超时[alm]
W427.05 BOOL  ; RK_05 #2入壳机构复位超时复位超时[alm]
W427.06 BOOL  ; RK_06 电池上下料机构复位超时复位超时[alm]
W427.07 BOOL  ; RK_07 铝壳进料机构复位超时复位超时[alm]
W427.08 BOOL  ; RK_07 铝壳上料移载机构复位超时复位超时[alm]
W427.09 BOOL  ; RK_07 #1铝壳上料升降机构复位超时复位超时[alm]
W427.10 BOOL  ; RK_07 #2铝壳上料升降机构复位超时复位超时[alm]
W427.11 BOOL  ; RK_07 铝壳托盘下料升降机构复位超时复位超时[alm]
W427.12 BOOL  ; RK_08 铝壳除尘机构复位超时复位超时[alm]
W427.13 BOOL  ; RK_09 #1Hipot检测机构复位超时复位超时[alm]
W427.14 BOOL  ; RK_09 #2Hipot检测机构复位超时复位超时[alm]
W427.15 BOOL  ; RK_10 电池除尘上料机构复位超时复位超时[alm]
W428.00 BOOL  ; RK_11 电池除尘机构复位超时复位超时[alm]
W428.01 BOOL  ; RK_12 预焊上下料机构复位超时复位超时[alm]
W428.02 BOOL  ; RK_13 #1移载机构复位超时复位超时[alm]
W428.03 BOOL  ; RK_13 #2移载机构复位超时复位超时[alm]
W428.04 BOOL  ; RK_14 #1压装机构复位超时复位超时[alm]
W428.05 BOOL  ; RK_14 #2压装机构复位超时复位超时[alm]
W428.06 BOOL  ; RK_15 轮廓检测机构复位超时复位超时[alm]
W428.07 BOOL  ; RK_16 焊接机构复位超时复位超时[alm]
W428.14 BOOL  ; 整机复位超时[alm]
W428.15 BOOL  ; RK_16 激光焊接超时[alm]
W429.00 BOOL  ; RK_01 电芯来料机构有料记忆[alm]
W429.01 BOOL  ; RK_02 扫码NG拉带放料位有料记忆[alm]
W429.02 BOOL  ; RK_04 电芯除尘机构有料记忆[alm]
W429.03 BOOL  ; RK_05 #1入壳机构有电池记忆[alm]
W429.04 BOOL  ; RK_05 #1入壳机构有电芯记忆[alm]
W429.05 BOOL  ; RK_05 #1入壳机构有铝壳记忆[alm]
W429.06 BOOL  ; RK_05 #2入壳机构有电池记忆[alm]
W429.07 BOOL  ; RK_05 #2入壳机构有电芯记忆[alm]
W429.08 BOOL  ; RK_05 #2入壳机构有铝壳记忆[alm]
W429.09 BOOL  ; RK_11 电池除尘机构有料记忆[alm]
W429.10 BOOL  ; RK_08 铝壳除尘机构有料记忆[alm]
W429.11 BOOL  ; RK_09 #1Hipot检测机构有料记忆[alm]
W429.12 BOOL  ; RK_09 #2Hipot检测机构有料记忆[alm]
W429.13 BOOL  ; RK_10 Hipot检测NG拉带放料位有料记忆[alm]
W429.14 BOOL  ; RK_12 轮廓检测NG槽#1有料记忆异常,请检查[0013.01]
W429.15 BOOL  ; RK_12 轮廓检测NG槽#2有料记忆异常,请检查[0013.03]
W430.00 BOOL  ; RK_13 #1移载有料记忆异常,请检查[0011.12]
W430.01 BOOL  ; RK_13 #2移载有料记忆异常,请检查[0011.13]
W430.02 BOOL  ; RK_12 出料拉带放料位有料记忆[alm]
W430.03 BOOL  ; RK_07 铝壳上料移载机构有托盘记忆[alm]
W430.04 BOOL  ; RK_07 铝壳上料移载机构托盘有料记忆[alm]
W430.12 BOOL  ; $?St$Bk?_#[5064] / 电芯进料X轴允许去放料位安全设定值过小 / [alm]$?St$Bk?_#[5064]
W430.13 BOOL  ; $?St$Bk?_#[5065] / 电芯上料X轴允许去取料位安全设定值过小 / [alm]$?St$Bk?_#[5065]
W430.14 BOOL  ; 电池除尘上料X轴允许去电池除尘放料位安全设定值过小[alm]
W430.15 BOOL  ; $?St$Bk?_#[5066] / 预焊上下料X轴允许去电池除尘取料位安全设定值过小 / [alm]$?St$Bk?_#[5066]
W431.00 BOOL  ; RK_02 电芯进料机构MES入站就绪通知&确认超时[alm]
W431.01 BOOL  ; RK_11 电池除尘上料机构MES出站就绪通知&确认超时[alm]
W431.02 BOOL  ; RK_12 电池上下料机构MES出站就绪通知&确认超时[alm]
W431.03 BOOL  ; 整机工艺参数变更通知&确认超时[alm]
W432.00 BOOL  ; 电脑软件未启动[alm]
W432.01 BOOL  ; RK_01 扫码通讯异常[alm]
W432.02 BOOL  ; RK_09 Hipot检测通讯异常[alm]
W432.03 BOOL  ; RK_15 轮廓检测通讯异常[alm]
W432.04 BOOL  ; RK_05 #1入壳压力断线[alm]
W432.05 BOOL  ; RK_05 #2入壳压力断线[alm]
W438.00 BOOL  ; RK_02 U0_Y 电芯进料X轴运行中电芯进料Z轴不在待料位（扫码）[alm]
W438.02 BOOL  ; 电芯进/上料伺服距离过小[alm]
W438.03 BOOL  ; RK_03 U0_U 电芯上料X轴运行中电芯上料升降气缸不在上升位[alm]
W438.04 BOOL  ; RK_05 #1入壳压力高[alm]
W438.05 BOOL  ; RK_05 #2入壳压力高[alm]
W438.06 BOOL  ; RK_06 U8_X 电池上下料X轴运行中上料升降气缸不在上升位[alm]
W438.07 BOOL  ; RK_06 U8_X 电池上下料X轴运行中下料升降气缸不在上升位[alm]
W438.08 BOOL  ; RK_07 U8_Y 铝壳进料X轴运行中上料升降气缸不在上升位[alm]
W438.09 BOOL  ; RK_07 U8_Z 铝壳上料移载Y轴运行中铝壳进料升降气缸不在上升位&铝壳上下料电机不在安全位[alm]
W438.10 BOOL  ; RK_10 U8_U 电池除尘上料X轴运行中上料升降气缸不在上升位[alm]
W438.11 BOOL  ; 电池除尘上料/预焊上下料伺服距离过小[alm]
W438.14 BOOL  ; RK_12 U4_X 预焊上下料X轴运行中预焊上料Z轴不在待料位[alm]
W438.15 BOOL  ; RK_12 U4_X 预焊上下料X轴运行中预焊下料Z轴不在待料位[alm]
W439.00 BOOL  ; RK_16 U6_Y 激光焊接X轴运行中激光焊接Z轴不在待料位
W65.00 BOOL  ; RK_02 电芯进料机构扫码
W65.01 BOOL  ; RK_02 电芯进料机构扫码发送
W65.02 BOOL  ; RK_02 电芯进料机构扫码失败
W65.03 BOOL  ; RK_02 电芯进料机构扫码成功
W65.04 BOOL  ; RK_02 电芯进料机构扫码接收
W65.05 BOOL  ; RK_02 电芯进料机构重新扫码触发
W80.00 BOOL  ; #1铝壳上料机构手动上料超时
W80.01 BOOL  ; #2铝壳上料机构手动上料超时
W80.02 BOOL  ; #3铝壳托盘下料机构手动下料超时
W81.00 BOOL  ; RK_01 电芯来料机构不在初始位提示
W81.01 BOOL  ; RK_02 电芯进料机构不在初始位提示
W81.02 BOOL  ; RK_03 电芯上料机构不在初始位提示
W81.03 BOOL  ; RK_04 电芯除尘机构不在初始位提示
W81.04 BOOL  ; RK_05 #1入壳机构不在初始位提示
W81.05 BOOL  ; RK_05 #2入壳机构不在初始位提示
W81.06 BOOL  ; RK_06 电池上下料机构不在初始位提示
W81.07 BOOL  ; RK_07 铝壳进料机构不在初始位提示
W81.08 BOOL  ; RK_07 铝壳上料移载机构不在初始位提示
W81.09 BOOL  ; RK_08 铝壳除尘机构不在初始位提示
W81.10 BOOL  ; RK_09 #1Hipot检测机构不在初始位提示
W81.11 BOOL  ; RK_09 #2Hipot检测机构不在初始位提示
W81.12 BOOL  ; RK_10 电池除尘上料机构不在初始位提示
W81.13 BOOL  ; RK_11 电池除尘机构不在初始位提示
W81.14 BOOL  ; RK_12 预焊上下料机构不在初始位提示
W81.15 BOOL  ; RK_13 #1移载机构不在初始位提示
W82.00 BOOL  ; RK_13 #2移载机构不在初始位提示
W82.01 BOOL  ; RK_14 #1压装机构不在初始位提示
W82.02 BOOL  ; RK_14 #2压装机构不在初始位提示
W82.03 BOOL  ; RK_15 轮廓检测机构不在初始位提示
W82.04 BOOL  ; RK_16 焊接机构不在初始位提示
W83.00 BOOL  ; RK_07 #1铝壳上料托盘到位有感应异常提示[0017.04]
W83.01 BOOL  ; RK_07 #1铝壳上料托盘到位无感应异常提示[0017.04]
W84.00 BOOL  ; RK_07 #2铝壳上料托盘到位有感应异常提示[0017.09]
W84.01 BOOL  ; RK_07 #2铝壳上料托盘到位无感应异常提示[0017.09]
W85.00 BOOL  ; RK_07 #3托盘下料上升到位有感应异常提示[0017.14]
W85.01 BOOL  ; RK_07 #3托盘下料上升到位无感应异常提示[0017.14]
W85.02 BOOL  ; RK_07 #3托盘下料下降到位有感应异常提示[0019.13]
W85.03 BOOL  ; RK_07 #3托盘下料下降到位无感应异常提示[0019.13]
W86.00 BOOL  ; RK_07 铝壳上料移载托盘到位有感应异常提示[0018.03]
NC433_0_2000_Setting _NCx600_Setting
NC433_2_2020_Setting _NCx600_Setting
NC433_4_2040_Setting _NCx600_Setting
NC433_6_2060_Setting _NCx600_Setting
NC433_8_2080_Setting _NCx600_Setting
RK_01_U0_X_Home _NCx051A_Home_DINT
RK_01_U0_X_Pos1 _NCx011A_MoveAbsolute_DINT
RK_01_U0_X_Pos2 _NCx011A_MoveAbsolute_DINT
RK_02_U0_Y_Home _NCx051A_Home_DINT
RK_02_U0_Y_Pos1 _NCx011A_MoveAbsolute_DINT
RK_02_U0_Y_Pos2 _NCx011A_MoveAbsolute_DINT
RK_02_U0_Y_Pos3 _NCx011A_MoveAbsolute_DINT
RK_02_U0_Z_Home _NCx051A_Home_DINT
RK_02_U0_Z_Pos1 _NCx011A_MoveAbsolute_DINT
RK_02_U0_Z_Pos2 _NCx011A_MoveAbsolute_DINT
RK_02_U0_Z_Pos3 _NCx011A_MoveAbsolute_DINT
RK_02_U0_Z_Pos4 _NCx011A_MoveAbsolute_DINT
RK_02_U0_Z_Pos5 _NCx011A_MoveAbsolute_DINT
RK_03_U0_U_Home _NCx051A_Home_DINT
RK_03_U0_U_Pos1 _NCx011A_MoveAbsolute_DINT
RK_03_U0_U_Pos2 _NCx011A_MoveAbsolute_DINT
RK_03_U0_U_Pos3 _NCx011A_MoveAbsolute_DINT
RK_03_U0_U_Pos4 _NCx011A_MoveAbsolute_DINT
RK_05_U2_X_Home _NCx051A_Home_DINT
RK_05_U2_X_Pos1 _NCx011A_MoveAbsolute_DINT
RK_05_U2_X_Pos2 _NCx011A_MoveAbsolute_DINT
RK_05_U2_X_Pos3 _NCx011A_MoveAbsolute_DINT
RK_05_U2_X_Pos4 _NCx011A_MoveAbsolute_DINT
RK_05_U2_X_Pos5 _NCx011A_MoveAbsolute_DINT
RK_05_U2_Y_Home _NCx051A_Home_DINT
RK_05_U2_Y_Pos1 _NCx011A_MoveAbsolute_DINT
RK_05_U2_Y_Pos2 _NCx011A_MoveAbsolute_DINT
RK_05_U2_Y_Pos3 _NCx011A_MoveAbsolute_DINT
RK_05_U2_Y_Pos4 _NCx011A_MoveAbsolute_DINT
RK_05_U2_Y_Pos5 _NCx011A_MoveAbsolute_DINT
RK_06_U8_X_Home _NCx051A_Home_DINT
RK_06_U8_X_Pos1 _NCx011A_MoveAbsolute_DINT
RK_06_U8_X_Pos2 _NCx011A_MoveAbsolute_DINT
RK_06_U8_X_Pos3 _NCx011A_MoveAbsolute_DINT
RK_06_U8_X_Pos4 _NCx011A_MoveAbsolute_DINT
RK_06_U8_X_Pos5 _NCx011A_MoveAbsolute_DINT
RK_06_U8_X_Pos6 _NCx011A_MoveAbsolute_DINT
RK_06_U8_X_Pos7 _NCx011A_MoveAbsolute_DINT
RK_07_U8_Y_Home _NCx051A_Home_DINT
RK_07_U8_Y_Pos1 _NCx011A_MoveAbsolute_DINT
RK_07_U8_Y_Pos2 _NCx011A_MoveAbsolute_DINT
RK_07_U8_Y_Pos3 _NCx011A_MoveAbsolute_DINT
RK_07_U8_Z_Home _NCx051A_Home_DINT
RK_07_U8_Z_Pos1 _NCx011A_MoveAbsolute_DINT
RK_07_U8_Z_Pos2 _NCx011A_MoveAbsolute_DINT
RK_07_U8_Z_Pos3 _NCx011A_MoveAbsolute_DINT
RK_07_U8_Z_Pos4 _NCx011A_MoveAbsolute_DINT
RK_10_U8_U_Home _NCx051A_Home_DINT
RK_10_U8_U_Pos1 _NCx011A_MoveAbsolute_DINT
RK_10_U8_U_Pos2 _NCx011A_MoveAbsolute_DINT
RK_10_U8_U_Pos3 _NCx011A_MoveAbsolute_DINT
RK_10_U8_U_Pos4 _NCx011A_MoveAbsolute_DINT
RK_12_U4_X_Home _NCx051A_Home_DINT
RK_12_U4_X_Pos1 _NCx011A_MoveAbsolute_DINT
RK_12_U4_X_Pos2 _NCx011A_MoveAbsolute_DINT
RK_12_U4_X_Pos3 _NCx011A_MoveAbsolute_DINT
RK_12_U4_X_Pos4 _NCx011A_MoveAbsolute_DINT
RK_12_U4_X_Pos5 _NCx011A_MoveAbsolute_DINT
RK_12_U4_X_Pos6 _NCx011A_MoveAbsolute_DINT
RK_12_U4_X_Pos7 _NCx011A_MoveAbsolute_DINT
RK_12_U4_X_Pos8 _NCx011A_MoveAbsolute_DINT
RK_12_U4_X_Pos9 _NCx011A_MoveAbsolute_DINT
RK_12_U4_Y_Home _NCx051A_Home_DINT
RK_12_U4_Y_Pos1 _NCx011A_MoveAbsolute_DINT
RK_12_U4_Y_Pos2 _NCx011A_MoveAbsolute_DINT
RK_12_U4_Y_Pos3 _NCx011A_MoveAbsolute_DINT
RK_12_U4_Y_Pos4 _NCx011A_MoveAbsolute_DINT
RK_12_U4_Z_Home _NCx051A_Home_DINT
RK_12_U4_Z_Pos1 _NCx011A_MoveAbsolute_DINT
RK_12_U4_Z_Pos2 _NCx011A_MoveAbsolute_DINT
RK_12_U4_Z_Pos3 _NCx011A_MoveAbsolute_DINT
RK_12_U4_Z_Pos4 _NCx011A_MoveAbsolute_DINT
RK_12_U4_Z_Pos5 _NCx011A_MoveAbsolute_DINT
RK_12_U4_Z_Pos6 _NCx011A_MoveAbsolute_DINT
RK_13_U4_U_Home _NCx051A_Home_DINT
RK_13_U4_U_Pos1 _NCx011A_MoveAbsolute_DINT
RK_13_U4_U_Pos2 _NCx011A_MoveAbsolute_DINT
RK_13_U4_U_Pos3 _NCx011A_MoveAbsolute_DINT
RK_13_U4_U_Pos4 _NCx011A_MoveAbsolute_DINT
RK_13_U4_U_Pos5 _NCx011A_MoveAbsolute_DINT
RK_13_U6_X_Home _NCx051A_Home_DINT
RK_13_U6_X_Pos1 _NCx011A_MoveAbsolute_DINT
RK_13_U6_X_Pos2 _NCx011A_MoveAbsolute_DINT
RK_13_U6_X_Pos3 _NCx011A_MoveAbsolute_DINT
RK_13_U6_X_Pos4 _NCx011A_MoveAbsolute_DINT
RK_13_U6_X_Pos5 _NCx011A_MoveAbsolute_DINT
RK_16_U6_Y_Home _NCx051A_Home_DINT
RK_16_U6_Y_Pos1 _NCx011A_MoveAbsolute_DINT
RK_16_U6_Y_Pos2 _NCx011A_MoveAbsolute_DINT
RK_16_U6_Z_Home _NCx051A_Home_DINT
RK_16_U6_Z_Pos1 _NCx011A_MoveAbsolute_DINT
RK_16_U6_Z_Pos2 _NCx011A_MoveAbsolute_DINT
RK_16_U6_Z_Pos3 _NCx011A_MoveAbsolute_DINT
RK_Pressure_1 入壳压力量程转换
RK_Pressure_2 入壳压力量程转换

## Program MAIN (cyclic task 0)
Local symbols
P_0_015 BOOL

### Section Main

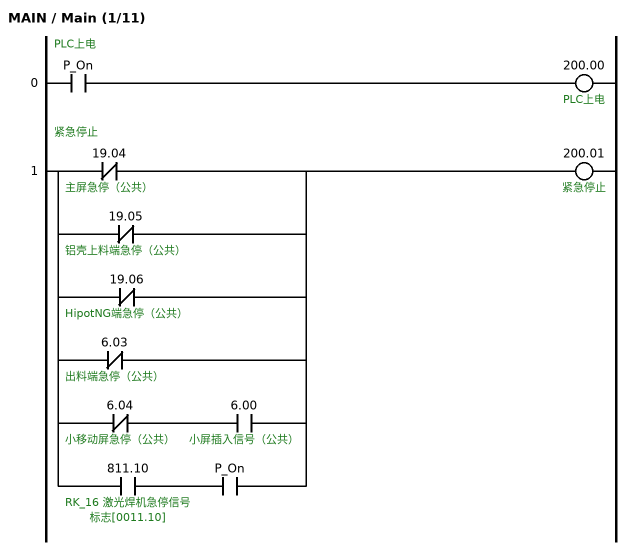
; rung 0: PLC上电
LD P_On
OUT 200.00  ; PLC上电
; rung 1: 紧急停止
LDNOT 19.04  ; 主屏急停（公共）
ORNOT 19.05  ; 铝壳上料端急停（公共）
ORNOT 19.06  ; HipotNG端急停（公共）
ORNOT 6.03  ; 出料端急停（公共）
LDNOT 6.04  ; 小移动屏急停（公共）
AND 6.00  ; 小屏插入信号（公共）
ORLD
LD 811.10  ; RK_16 激光焊机急停信号标志[0011.10]
AND P_On
ORLD
OUT 200.01  ; 紧急停止

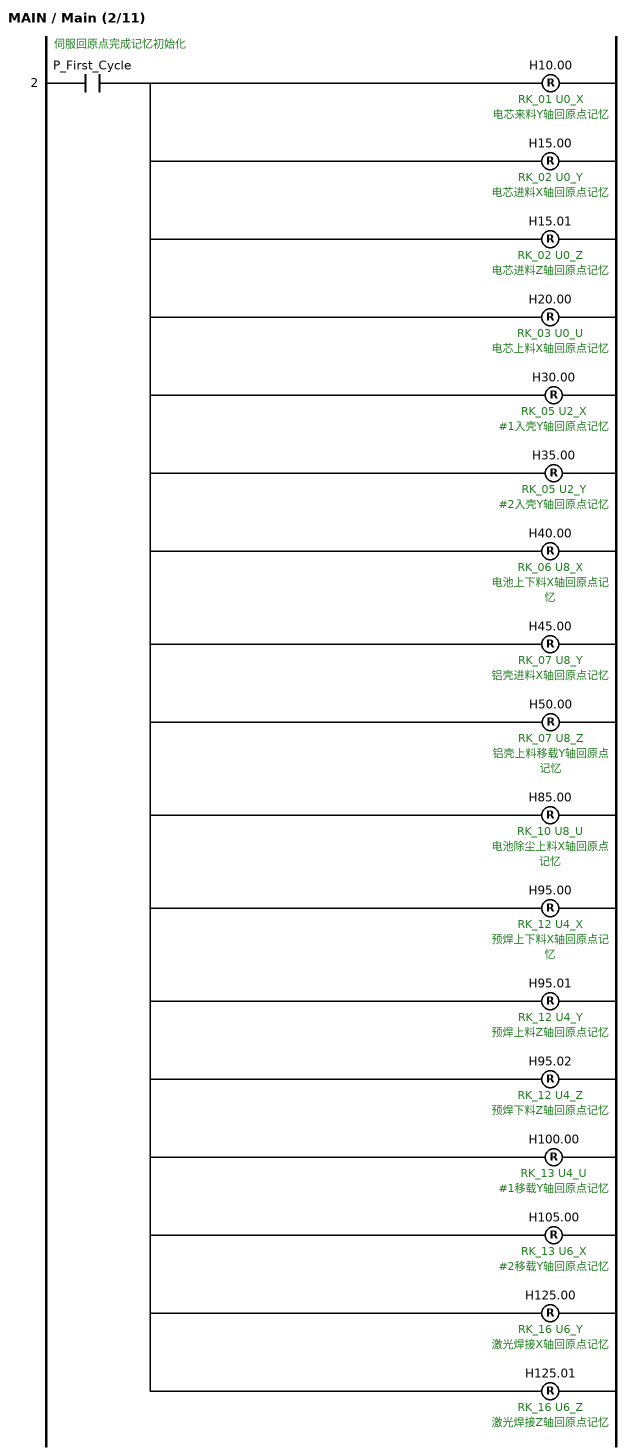
; rung 2: 伺服回原点完成记忆初始化
LD P_First_Cycle
RSET H10.00  ; RK_01 U0_X 电芯来料Y轴回原点记忆
RSET H15.00  ; RK_02 U0_Y 电芯进料X轴回原点记忆
RSET H15.01  ; RK_02 U0_Z 电芯进料Z轴回原点记忆
RSET H20.00  ; RK_03 U0_U 电芯上料X轴回原点记忆
RSET H30.00  ; RK_05 U2_X #1入壳Y轴回原点记忆
RSET H35.00  ; RK_05 U2_Y #2入壳Y轴回原点记忆
RSET H40.00  ; RK_06 U8_X 电池上下料X轴回原点记忆
RSET H45.00  ; RK_07 U8_Y 铝壳进料X轴回原点记忆
RSET H50.00  ; RK_07 U8_Z 铝壳上料移载Y轴回原点记忆
RSET H85.00  ; RK_10 U8_U 电池除尘上料X轴回原点记忆
RSET H95.00  ; RK_12 U4_X 预焊上下料X轴回原点记忆
RSET H95.01  ; RK_12 U4_Y 预焊上料Z轴回原点记忆
RSET H95.02  ; RK_12 U4_Z 预焊下料Z轴回原点记忆
RSET H100.00  ; RK_13 U4_U #1移载Y轴回原点记忆
RSET H105.00  ; RK_13 U6_X #2移载Y轴回原点记忆
RSET H125.00  ; RK_16 U6_Y 激光焊接X轴回原点记忆
RSET H125.01  ; RK_16 U6_Z 激光焊接Z轴回原点记忆

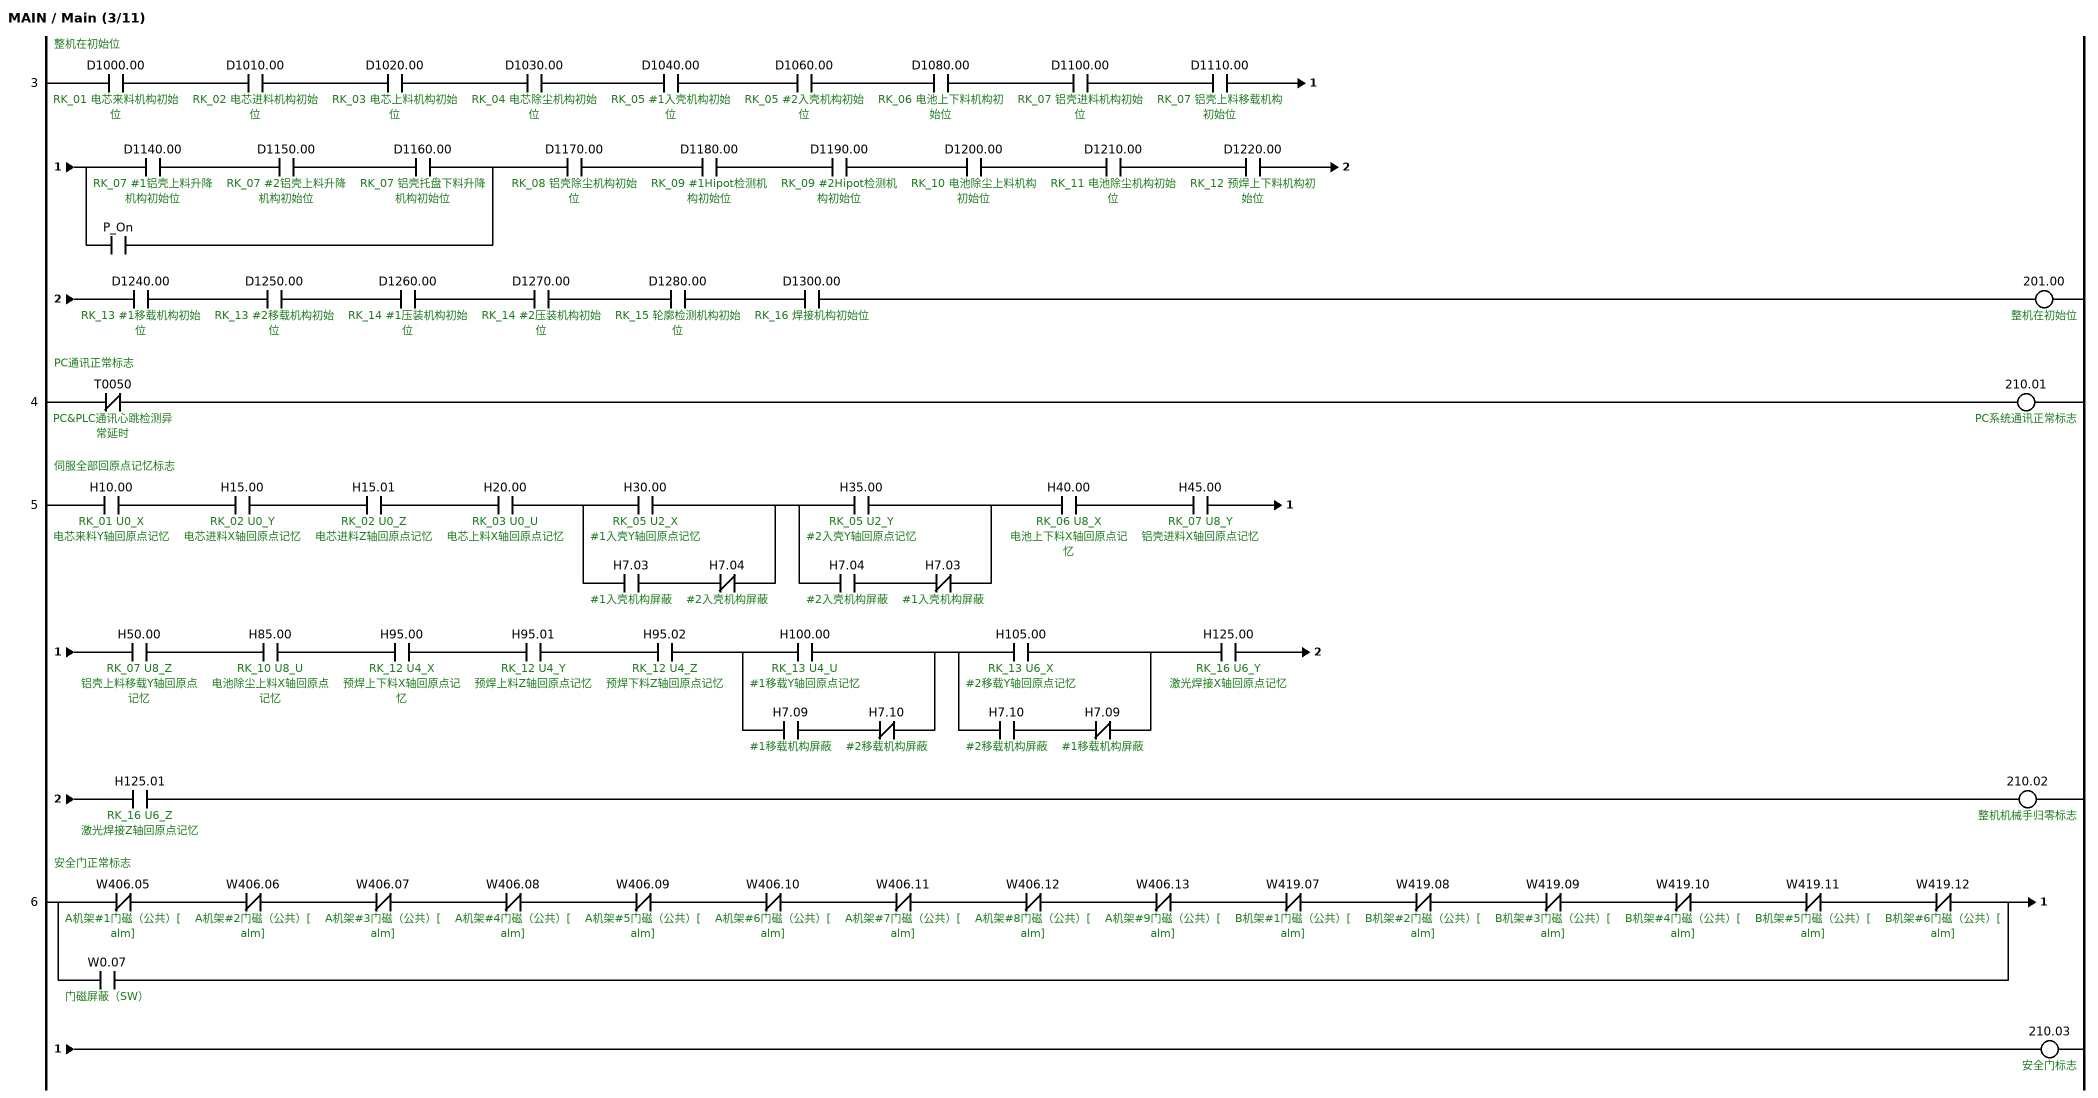
; rung 3: 整机在初始位
LD D1000.00  ; RK_01 电芯来料机构初始位
AND D1010.00  ; RK_02 电芯进料机构初始位
AND D1020.00  ; RK_03 电芯上料机构初始位
AND D1030.00  ; RK_04 电芯除尘机构初始位
AND D1040.00  ; RK_05 #1入壳机构初始位
AND D1060.00  ; RK_05 #2入壳机构初始位
AND D1080.00  ; RK_06 电池上下料机构初始位
AND D1100.00  ; RK_07 铝壳进料机构初始位
AND D1110.00  ; RK_07 铝壳上料移载机构初始位
LD D1140.00  ; RK_07 #1铝壳上料升降机构初始位
AND D1150.00  ; RK_07 #2铝壳上料升降机构初始位
AND D1160.00  ; RK_07 铝壳托盘下料升降机构初始位
OR P_On
ANDLD
AND D1170.00  ; RK_08 铝壳除尘机构初始位
AND D1180.00  ; RK_09 #1Hipot检测机构初始位
AND D1190.00  ; RK_09 #2Hipot检测机构初始位
AND D1200.00  ; RK_10 电池除尘上料机构初始位
AND D1210.00  ; RK_11 电池除尘机构初始位
AND D1220.00  ; RK_12 预焊上下料机构初始位
AND D1240.00  ; RK_13 #1移载机构初始位
AND D1250.00  ; RK_13 #2移载机构初始位
AND D1260.00  ; RK_14 #1压装机构初始位
AND D1270.00  ; RK_14 #2压装机构初始位
AND D1280.00  ; RK_15 轮廓检测机构初始位
AND D1300.00  ; RK_16 焊接机构初始位
OUT 201.00  ; 整机在初始位
; rung 4: PC通讯正常标志
LDNOT T0050  ; PC&PLC通讯心跳检测异常延时
OUT 210.01  ; PC系统通讯正常标志
; rung 5: 伺服全部回原点记忆标志
LD H10.00  ; RK_01 U0_X 电芯来料Y轴回原点记忆
AND H15.00  ; RK_02 U0_Y 电芯进料X轴回原点记忆
AND H15.01  ; RK_02 U0_Z 电芯进料Z轴回原点记忆
AND H20.00  ; RK_03 U0_U 电芯上料X轴回原点记忆
LD H30.00  ; RK_05 U2_X #1入壳Y轴回原点记忆
LD H7.03  ; #1入壳机构屏蔽
ANDNOT H7.04  ; #2入壳机构屏蔽
ORLD
ANDLD
LD H35.00  ; RK_05 U2_Y #2入壳Y轴回原点记忆
LD H7.04  ; #2入壳机构屏蔽
ANDNOT H7.03  ; #1入壳机构屏蔽
ORLD
ANDLD
AND H40.00  ; RK_06 U8_X 电池上下料X轴回原点记忆
AND H45.00  ; RK_07 U8_Y 铝壳进料X轴回原点记忆
AND H50.00  ; RK_07 U8_Z 铝壳上料移载Y轴回原点记忆
AND H85.00  ; RK_10 U8_U 电池除尘上料X轴回原点记忆
AND H95.00  ; RK_12 U4_X 预焊上下料X轴回原点记忆
AND H95.01  ; RK_12 U4_Y 预焊上料Z轴回原点记忆
AND H95.02  ; RK_12 U4_Z 预焊下料Z轴回原点记忆
LD H100.00  ; RK_13 U4_U #1移载Y轴回原点记忆
LD H7.09  ; #1移载机构屏蔽
ANDNOT H7.10  ; #2移载机构屏蔽
ORLD
ANDLD
LD H105.00  ; RK_13 U6_X #2移载Y轴回原点记忆
LD H7.10  ; #2移载机构屏蔽
ANDNOT H7.09  ; #1移载机构屏蔽
ORLD
ANDLD
AND H125.00  ; RK_16 U6_Y 激光焊接X轴回原点记忆
AND H125.01  ; RK_16 U6_Z 激光焊接Z轴回原点记忆
OUT 210.02  ; 整机机械手归零标志
; rung 6: 安全门正常标志
LDNOT W406.05  ; A机架#1门磁（公共）[alm]
ANDNOT W406.06  ; A机架#2门磁（公共）[alm]
ANDNOT W406.07  ; A机架#3门磁（公共）[alm]
ANDNOT W406.08  ; A机架#4门磁（公共）[alm]
ANDNOT W406.09  ; A机架#5门磁（公共）[alm]
ANDNOT W406.10  ; A机架#6门磁（公共）[alm]
ANDNOT W406.11  ; A机架#7门磁（公共）[alm]
ANDNOT W406.12  ; A机架#8门磁（公共）[alm]
ANDNOT W406.13  ; A机架#9门磁（公共）[alm]
ANDNOT W419.07  ; B机架#1门磁（公共）[alm]
ANDNOT W419.08  ; B机架#2门磁（公共）[alm]
ANDNOT W419.09  ; B机架#3门磁（公共）[alm]
ANDNOT W419.10  ; B机架#4门磁（公共）[alm]
ANDNOT W419.11  ; B机架#5门磁（公共）[alm]
ANDNOT W419.12  ; B机架#6门磁（公共）[alm]
OR W0.07  ; 门磁屏蔽（SW）
OUT 210.03  ; 安全门标志

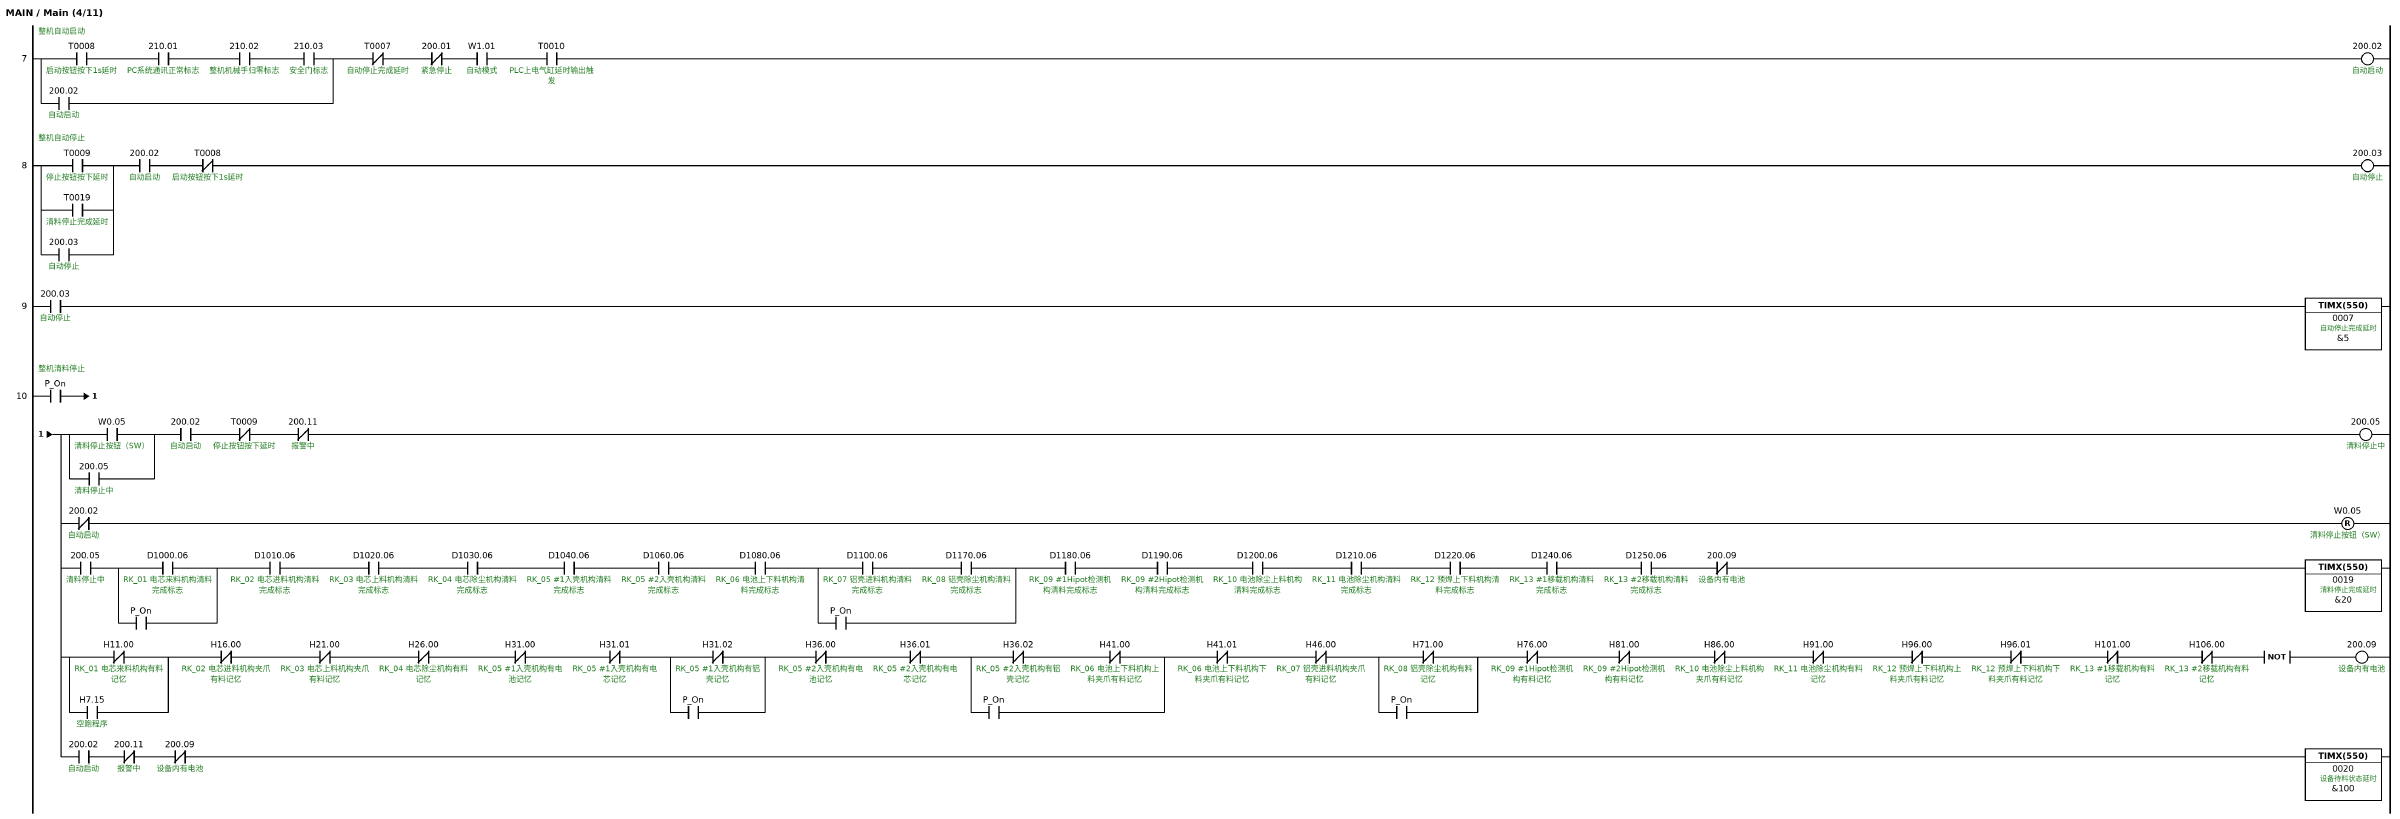
; rung 7: 整机自动启动
LD T0008  ; 启动按钮按下1s延时
AND 210.01  ; PC系统通讯正常标志
AND 210.02  ; 整机机械手归零标志
AND 210.03  ; 安全门标志
OR 200.02  ; 自动启动
ANDNOT T0007  ; 自动停止完成延时
ANDNOT 200.01  ; 紧急停止
AND W1.01  ; 自动模式
AND T0010  ; PLC上电气缸延时输出触发
OUT 200.02  ; 自动启动
; rung 8: 整机自动停止
LD T0009  ; 停止按钮按下延时
OR T0019  ; 清料停止完成延时
OR 200.03  ; 自动停止
AND 200.02  ; 自动启动
ANDNOT T0008  ; 启动按钮按下1s延时
OUT 200.03  ; 自动停止
; rung 9
LD 200.03  ; 自动停止
TIMX(550) 0007 &5  ; 自动停止完成延时
; rung 10: 整机清料停止
LD P_On
OUT TR0
LD W0.05  ; 清料停止按钮（SW）
OR 200.05  ; 清料停止中
ANDLD
AND 200.02  ; 自动启动
ANDNOT T0009  ; 停止按钮按下延时
ANDNOT 200.11  ; 报警中
OUT 200.05  ; 清料停止中
LD TR0
ANDNOT 200.02  ; 自动启动
RSET W0.05  ; 清料停止按钮（SW）
LD TR0
AND 200.05  ; 清料停止中
LD D1000.06  ; RK_01 电芯来料机构清料完成标志
OR P_On  // 待确认！！
ANDLD
AND D1010.06  ; RK_02 电芯进料机构清料完成标志
AND D1020.06  ; RK_03 电芯上料机构清料完成标志
AND D1030.06  ; RK_04 电芯除尘机构清料完成标志
AND D1040.06  ; RK_05 #1入壳机构清料完成标志
AND D1060.06  ; RK_05 #2入壳机构清料完成标志
AND D1080.06  ; RK_06 电池上下料机构清料完成标志
LD D1100.06  ; RK_07 铝壳进料机构清料完成标志
AND D1170.06  ; RK_08 铝壳除尘机构清料完成标志
OR P_On  // 待确认！！
ANDLD
AND D1180.06  ; RK_09 #1Hipot检测机构清料完成标志
AND D1190.06  ; RK_09 #2Hipot检测机构清料完成标志
AND D1200.06  ; RK_10 电池除尘上料机构清料完成标志
AND D1210.06  ; RK_11 电池除尘机构清料完成标志
AND D1220.06  ; RK_12 预焊上下料机构清料完成标志
AND D1240.06  ; RK_13 #1移载机构清料完成标志
AND D1250.06  ; RK_13 #2移载机构清料完成标志
ANDNOT 200.09  ; 设备内有电池
TIMX(550) 0019 &20  ; 清料停止完成延时
LD TR0
LDNOT H11.00  ; RK_01 电芯来料机构有料记忆
OR H7.15  ; 空跑程序
ANDLD
ANDNOT H16.00  ; RK_02 电芯进料机构夹爪有料记忆
ANDNOT H21.00  ; RK_03 电芯上料机构夹爪有料记忆
ANDNOT H26.00  ; RK_04 电芯除尘机构有料记忆
ANDNOT H31.00  ; RK_05 #1入壳机构有电池记忆
ANDNOT H31.01  ; RK_05 #1入壳机构有电芯记忆
LDNOT H31.02  ; RK_05 #1入壳机构有铝壳记忆
OR P_On  // 待确认！！
ANDLD
ANDNOT H36.00  ; RK_05 #2入壳机构有电池记忆
ANDNOT H36.01  ; RK_05 #2入壳机构有电芯记忆
LDNOT H36.02  ; RK_05 #2入壳机构有铝壳记忆
ANDNOT H41.00  ; RK_06 电池上下料机构上料夹爪有料记忆
OR P_On  // 待确认！！
ANDLD
ANDNOT H41.01  ; RK_06 电池上下料机构下料夹爪有料记忆
ANDNOT H46.00  ; RK_07 铝壳进料机构夹爪有料记忆
LDNOT H71.00  ; RK_08 铝壳除尘机构有料记忆
OR P_On  // 待确认！！
ANDLD
ANDNOT H76.00  ; RK_09 #1Hipot检测机构有料记忆
ANDNOT H81.00  ; RK_09 #2Hipot检测机构有料记忆
ANDNOT H86.00  ; RK_10 电池除尘上料机构夹爪有料记忆
ANDNOT H91.00  ; RK_11 电池除尘机构有料记忆
ANDNOT H96.00  ; RK_12 预焊上下料机构上料夹爪有料记忆
ANDNOT H96.01  ; RK_12 预焊上下料机构下料夹爪有料记忆
ANDNOT H101.00  ; RK_13 #1移载机构有料记忆
ANDNOT H106.00  ; RK_13 #2移载机构有料记忆
NOT(520)
OUT 200.09  ; 设备内有电池
LD TR0
AND 200.02  ; 自动启动
ANDNOT 200.11  ; 报警中
ANDNOT 200.09  ; 设备内有电池
TIMX(550) 0020 &100  ; 设备待料状态延时

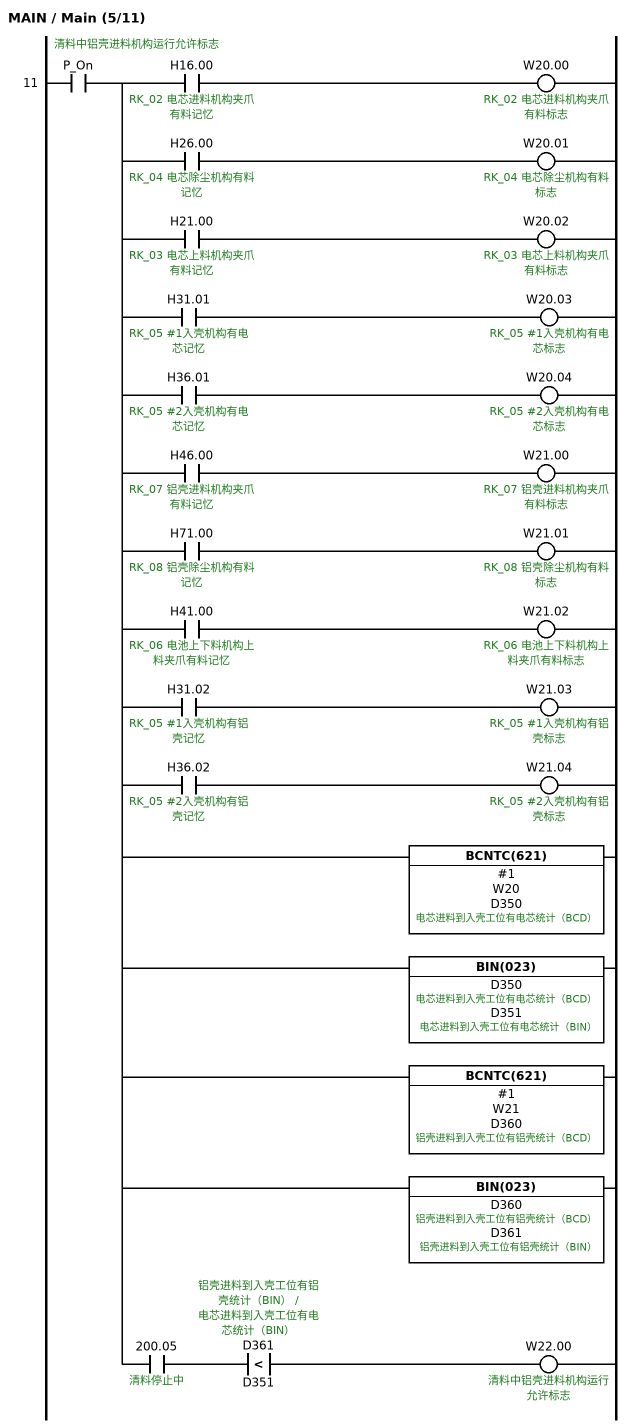
; rung 11: 清料中铝壳进料机构运行允许标志
LD P_On
OUT TR0
AND H16.00  ; RK_02 电芯进料机构夹爪有料记忆
OUT W20.00  ; RK_02 电芯进料机构夹爪有料标志
LD TR0
AND H26.00  ; RK_04 电芯除尘机构有料记忆
OUT W20.01  ; RK_04 电芯除尘机构有料标志
LD TR0
AND H21.00  ; RK_03 电芯上料机构夹爪有料记忆
OUT W20.02  ; RK_03 电芯上料机构夹爪有料标志
LD TR0
AND H31.01  ; RK_05 #1入壳机构有电芯记忆
OUT W20.03  ; RK_05 #1入壳机构有电芯标志
LD TR0
AND H36.01  ; RK_05 #2入壳机构有电芯记忆
OUT W20.04  ; RK_05 #2入壳机构有电芯标志
LD TR0
AND H46.00  ; RK_07 铝壳进料机构夹爪有料记忆
OUT W21.00  ; RK_07 铝壳进料机构夹爪有料标志
LD TR0
AND H71.00  ; RK_08 铝壳除尘机构有料记忆
OUT W21.01  ; RK_08 铝壳除尘机构有料标志
LD TR0
AND H41.00  ; RK_06 电池上下料机构上料夹爪有料记忆
OUT W21.02  ; RK_06 电池上下料机构上料夹爪有料标志
LD TR0
AND H31.02  ; RK_05 #1入壳机构有铝壳记忆
OUT W21.03  ; RK_05 #1入壳机构有铝壳标志
LD TR0
AND H36.02  ; RK_05 #2入壳机构有铝壳记忆
OUT W21.04  ; RK_05 #2入壳机构有铝壳标志
LD TR0
BCNTC(621) #1 W20 D350  ; 电芯进料到入壳工位有电芯统计（BCD）  // W20.05-20.15被占用，不能另作其它用途！！
BIN(023) D350 D351  ; 电芯进料到入壳工位有电芯统计（BCD）, 电芯进料到入壳工位有电芯统计（BIN）
BCNTC(621) #1 W21 D360  ; 铝壳进料到入壳工位有铝壳统计（BCD）  // W21.05-21.15被占用，不能另作其它用途！！
BIN(023) D360 D361  ; 铝壳进料到入壳工位有铝壳统计（BCD）, 铝壳进料到入壳工位有铝壳统计（BIN）
AND 200.05  ; 清料停止中
AND<(310) D361 D351  ; 铝壳进料到入壳工位有铝壳统计（BIN）, 电芯进料到入壳工位有电芯统计（BIN）
OUT W22.00  ; 清料中铝壳进料机构运行允许标志

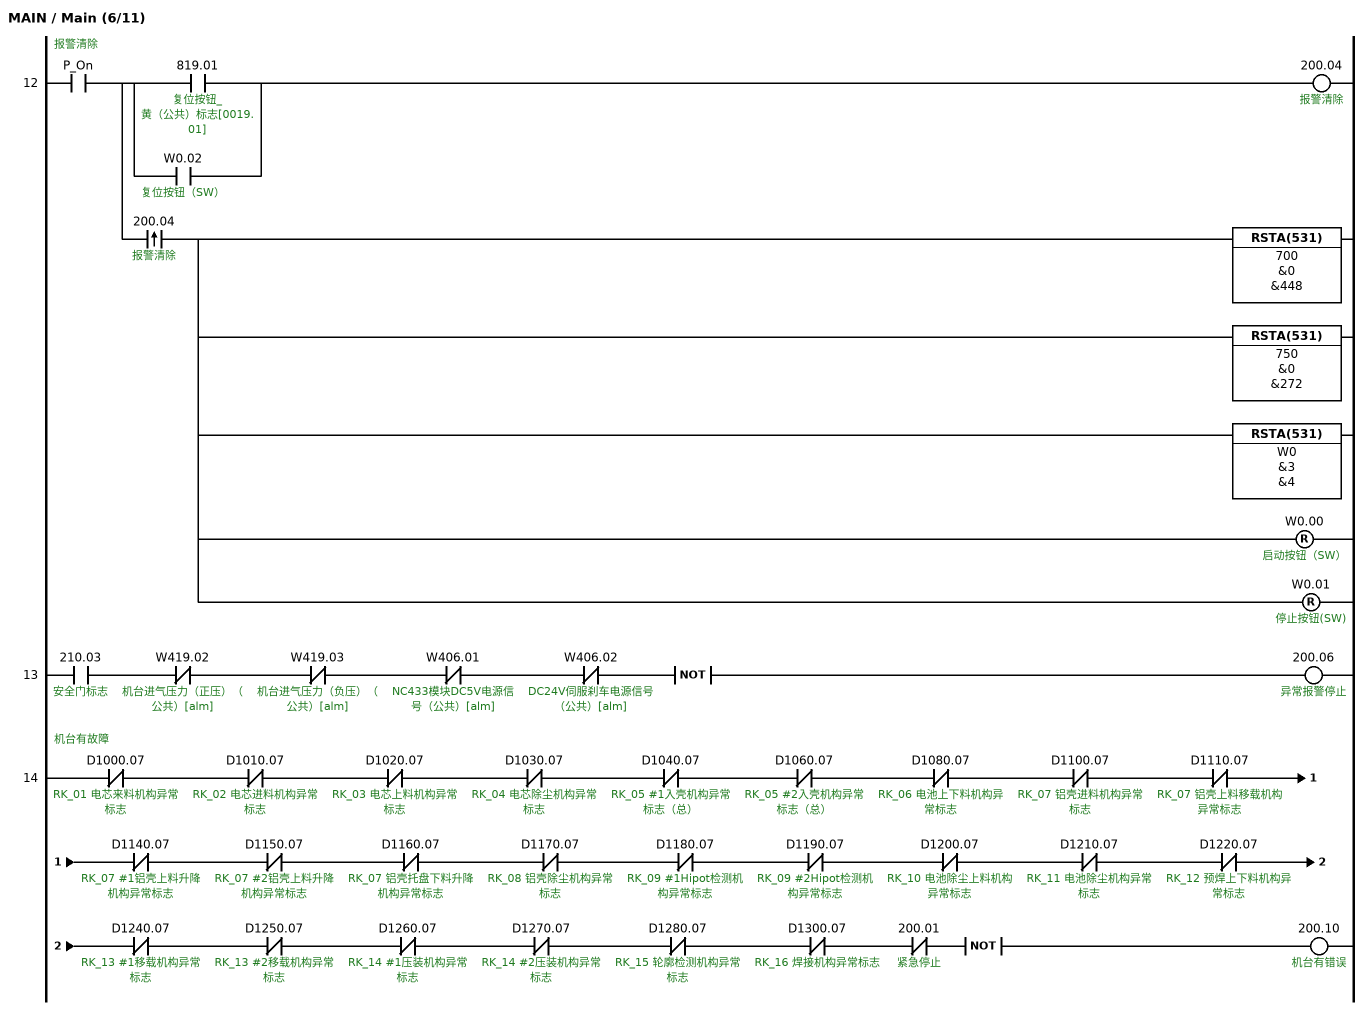
; rung 12: 报警清除
LD P_On
OUT TR0
LD 819.01  ; 复位按钮_黄（公共）标志[0019.01]
OR W0.02  ; 复位按钮（SW）
ANDLD
OUT 200.04  ; 报警清除
LD TR0
@AND 200.04  ; 报警清除
RSTA(531) 700 &0 &448
RSTA(531) 750 &0 &272
RSTA(531) W0 &3 &4
RSET W0.00  ; 启动按钮（SW）
RSET W0.01  ; 停止按钮(SW)
; rung 13
LD 210.03  ; 安全门标志
ANDNOT W419.02  ; 机台进气压力（正压）（公共）[alm]
ANDNOT W419.03  ; 机台进气压力（负压）（公共）[alm]
ANDNOT W406.01  ; NC433模块DC5V电源信号（公共）[alm]
ANDNOT W406.02  ; DC24V伺服刹车电源信号（公共）[alm]
NOT(520)
OUT 200.06  ; 异常报警停止
; rung 14: 机台有故障
LDNOT D1000.07  ; RK_01 电芯来料机构异常标志
ANDNOT D1010.07  ; RK_02 电芯进料机构异常标志
ANDNOT D1020.07  ; RK_03 电芯上料机构异常标志
ANDNOT D1030.07  ; RK_04 电芯除尘机构异常标志
ANDNOT D1040.07  ; RK_05 #1入壳机构异常标志（总）
ANDNOT D1060.07  ; RK_05 #2入壳机构异常标志（总）
ANDNOT D1080.07  ; RK_06 电池上下料机构异常标志
ANDNOT D1100.07  ; RK_07 铝壳进料机构异常标志
ANDNOT D1110.07  ; RK_07 铝壳上料移载机构异常标志
ANDNOT D1140.07  ; RK_07 #1铝壳上料升降机构异常标志
ANDNOT D1150.07  ; RK_07 #2铝壳上料升降机构异常标志
ANDNOT D1160.07  ; RK_07 铝壳托盘下料升降机构异常标志
ANDNOT D1170.07  ; RK_08 铝壳除尘机构异常标志
ANDNOT D1180.07  ; RK_09 #1Hipot检测机构异常标志
ANDNOT D1190.07  ; RK_09 #2Hipot检测机构异常标志
ANDNOT D1200.07  ; RK_10 电池除尘上料机构异常标志
ANDNOT D1210.07  ; RK_11 电池除尘机构异常标志
ANDNOT D1220.07  ; RK_12 预焊上下料机构异常标志
ANDNOT D1240.07  ; RK_13 #1移载机构异常标志
ANDNOT D1250.07  ; RK_13 #2移载机构异常标志
ANDNOT D1260.07  ; RK_14 #1压装机构异常标志
ANDNOT D1270.07  ; RK_14 #2压装机构异常标志
ANDNOT D1280.07  ; RK_15 轮廓检测机构异常标志
ANDNOT D1300.07  ; RK_16 焊接机构异常标志
ANDNOT 200.01  ; 紧急停止
NOT(520)
OUT 200.10  ; 机台有错误

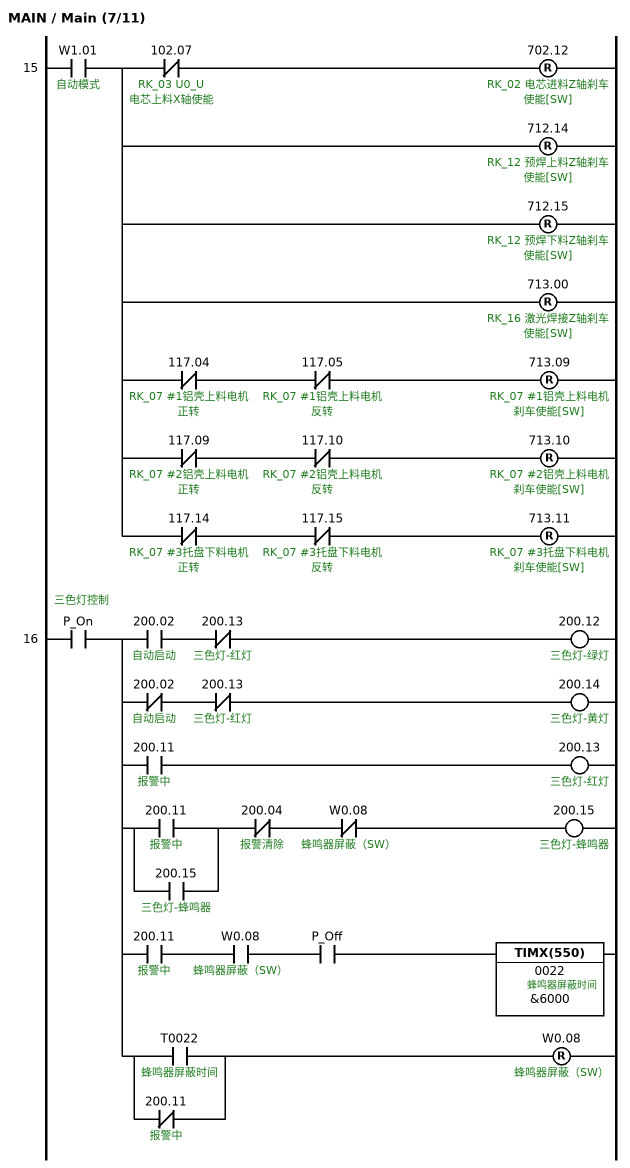
; rung 15
LD W1.01  ; 自动模式
OUT TR0
ANDNOT 102.07  ; RK_03 U0_U 电芯上料X轴使能
RSET 702.12  ; RK_02 电芯进料Z轴刹车使能[SW]
LD TR0
RSET 712.14  ; RK_12 预焊上料Z轴刹车使能[SW]
RSET 712.15  ; RK_12 预焊下料Z轴刹车使能[SW]
RSET 713.00  ; RK_16 激光焊接Z轴刹车使能[SW]
ANDNOT 117.04  ; RK_07 #1铝壳上料电机正转
ANDNOT 117.05  ; RK_07 #1铝壳上料电机反转
RSET 713.09  ; RK_07 #1铝壳上料电机刹车使能[SW]
LD TR0
ANDNOT 117.09  ; RK_07 #2铝壳上料电机正转
ANDNOT 117.10  ; RK_07 #2铝壳上料电机反转
RSET 713.10  ; RK_07 #2铝壳上料电机刹车使能[SW]
LD TR0
ANDNOT 117.14  ; RK_07 #3托盘下料电机正转
ANDNOT 117.15  ; RK_07 #3托盘下料电机反转
RSET 713.11  ; RK_07 #3托盘下料电机刹车使能[SW]
; rung 16: 三色灯控制
LD P_On
OUT TR0
AND 200.02  ; 自动启动
ANDNOT 200.13  ; 三色灯-红灯
OUT 200.12  ; 三色灯-绿灯
LD TR0
ANDNOT 200.02  ; 自动启动
ANDNOT 200.13  ; 三色灯-红灯
OUT 200.14  ; 三色灯-黄灯
LD TR0
AND 200.11  ; 报警中
OUT 200.13  ; 三色灯-红灯
LD TR0
LD 200.11  ; 报警中
OR 200.15  ; 三色灯-蜂鸣器
ANDLD
ANDNOT 200.04  ; 报警清除
ANDNOT W0.08  ; 蜂鸣器屏蔽（SW）
OUT 200.15  ; 三色灯-蜂鸣器
LD TR0
AND 200.11  ; 报警中
AND W0.08  ; 蜂鸣器屏蔽（SW）
AND P_Off
TIMX(550) 0022 &6000  ; 蜂鸣器屏蔽时间
LD TR0
LD T0022  ; 蜂鸣器屏蔽时间
ORNOT 200.11  ; 报警中
ANDLD
RSET W0.08  ; 蜂鸣器屏蔽（SW）

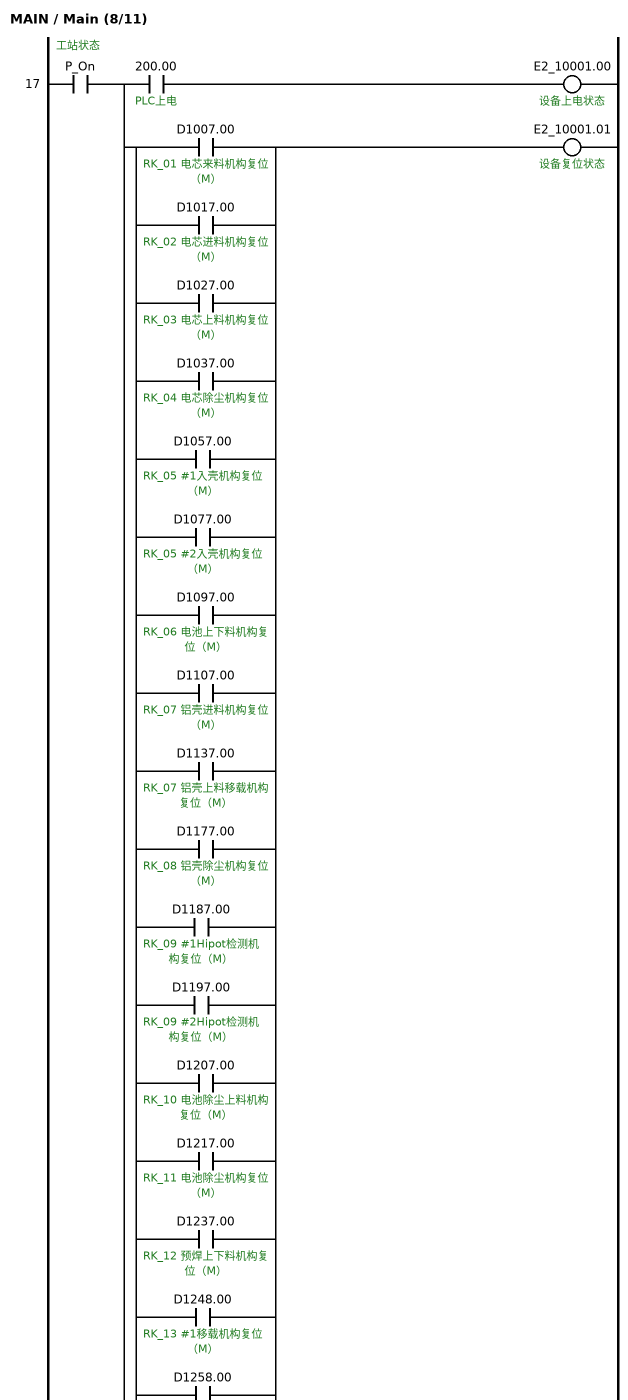

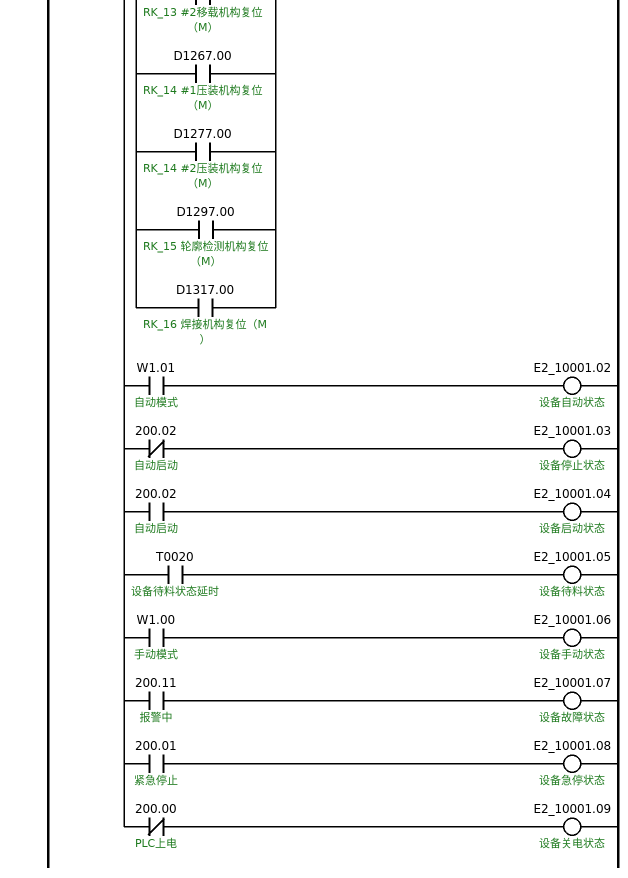
; rung 17: 工站状态
LD P_On
OUT TR0
AND 200.00  ; PLC上电
OUT E2_10001.00  ; 设备上电状态
LD TR0
LD D1007.00  ; RK_01 电芯来料机构复位（M）
OR D1017.00  ; RK_02 电芯进料机构复位（M）
OR D1027.00  ; RK_03 电芯上料机构复位（M）
OR D1037.00  ; RK_04 电芯除尘机构复位（M）
OR D1057.00  ; RK_05 #1入壳机构复位（M）
OR D1077.00  ; RK_05 #2入壳机构复位（M）
OR D1097.00  ; RK_06 电池上下料机构复位（M）
OR D1107.00  ; RK_07 铝壳进料机构复位（M）
OR D1137.00  ; RK_07 铝壳上料移载机构复位（M）
OR D1177.00  ; RK_08 铝壳除尘机构复位（M）
OR D1187.00  ; RK_09 #1Hipot检测机构复位（M）
OR D1197.00  ; RK_09 #2Hipot检测机构复位（M）
OR D1207.00  ; RK_10 电池除尘上料机构复位（M）
OR D1217.00  ; RK_11 电池除尘机构复位（M）
OR D1237.00  ; RK_12 预焊上下料机构复位（M）
OR D1248.00  ; RK_13 #1移载机构复位（M）
OR D1258.00  ; RK_13 #2移载机构复位（M）
OR D1267.00  ; RK_14 #1压装机构复位（M）
OR D1277.00  ; RK_14 #2压装机构复位（M）
OR D1297.00  ; RK_15 轮廓检测机构复位（M）
OR D1317.00  ; RK_16 焊接机构复位（M）
ANDLD
OUT E2_10001.01  ; 设备复位状态
LD TR0
AND W1.01  ; 自动模式
OUT E2_10001.02  ; 设备自动状态
LD TR0
ANDNOT 200.02  ; 自动启动
OUT E2_10001.03  ; 设备停止状态
LD TR0
AND 200.02  ; 自动启动
OUT E2_10001.04  ; 设备启动状态
LD TR0
AND T0020  ; 设备待料状态延时
OUT E2_10001.05  ; 设备待料状态
LD TR0
AND W1.00  ; 手动模式
OUT E2_10001.06  ; 设备手动状态
LD TR0
AND 200.11  ; 报警中
OUT E2_10001.07  ; 设备故障状态
LD TR0
AND 200.01  ; 紧急停止
OUT E2_10001.08  ; 设备急停状态
LD TR0
ANDNOT 200.00  ; PLC上电
OUT E2_10001.09  ; 设备关电状态

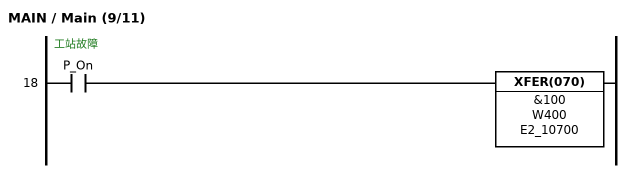
; rung 18: 工站故障
LD P_On
XFER(070) &100 W400 E2_10700

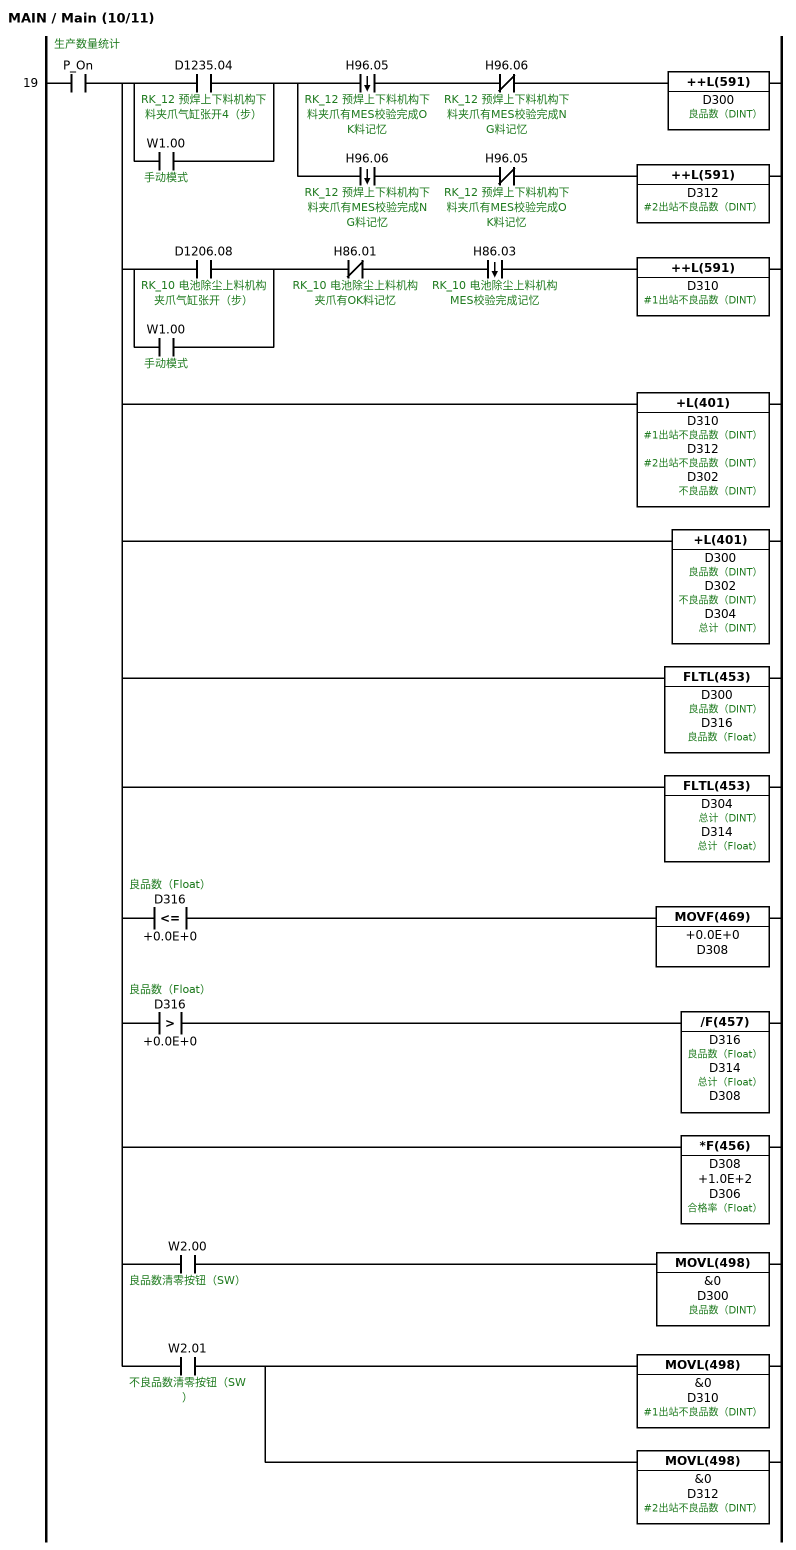
; rung 19: 生产数量统计
LD P_On
OUT TR0
LD D1235.04  ; RK_12 预焊上下料机构下料夹爪气缸张开4（步）
OR W1.00  ; 手动模式
ANDLD
OUT TR1
%AND H96.05  ; RK_12 预焊上下料机构下料夹爪有MES校验完成OK料记忆
ANDNOT H96.06  ; RK_12 预焊上下料机构下料夹爪有MES校验完成NG料记忆
++L(591) D300  ; 良品数（DINT）
LD TR1
%AND H96.06  ; RK_12 预焊上下料机构下料夹爪有MES校验完成NG料记忆
ANDNOT H96.05  ; RK_12 预焊上下料机构下料夹爪有MES校验完成OK料记忆
++L(591) D312  ; #2出站不良品数（DINT）
LD TR0
LD D1206.08  ; RK_10 电池除尘上料机构夹爪气缸张开（步）
OR W1.00  ; 手动模式
ANDLD
ANDNOT H86.01  ; RK_10 电池除尘上料机构夹爪有OK料记忆
%AND H86.03  ; RK_10 电池除尘上料机构MES校验完成记忆
++L(591) D310  ; #1出站不良品数（DINT）
LD TR0
+L(401) D310 D312 D302  ; #1出站不良品数（DINT）, #2出站不良品数（DINT）, 不良品数（DINT）
+L(401) D300 D302 D304  ; 良品数（DINT）, 不良品数（DINT）, 总计（DINT）
FLTL(453) D300 D316  ; 良品数（DINT）, 良品数（Float）
FLTL(453) D304 D314  ; 总计（DINT）, 总计（Float）
AND<=F(332) D316 +0.0E+0  ; 良品数（Float）
MOVF(469) +0.0E+0 D308
LD TR0
AND>F(333) D316 +0.0E+0  ; 良品数（Float）
/F(457) D316 D314 D308  ; 良品数（Float）, 总计（Float）
LD TR0
*F(456) D308 +1.0E+2 D306  ; 合格率（Float）
AND W2.00  ; 良品数清零按钮（SW）
MOVL(498) &0 D300  ; 良品数（DINT）
LD TR0
AND W2.01  ; 不良品数清零按钮（SW）
MOVL(498) &0 D310  ; #1出站不良品数（DINT）
MOVL(498) &0 D312  ; #2出站不良品数（DINT）

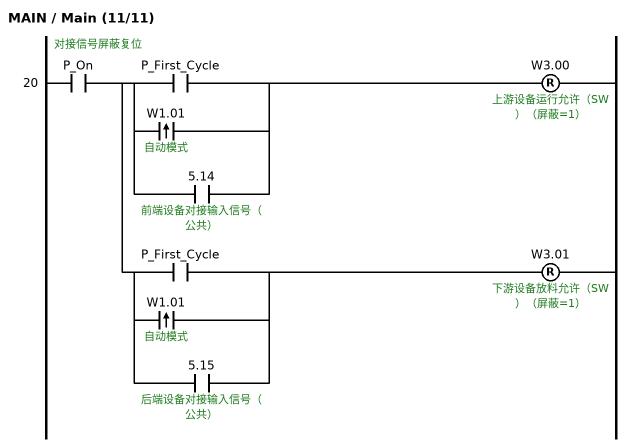
; rung 20: 对接信号屏蔽复位
LD P_On
OUT TR0
LD P_First_Cycle
@OR W1.01  ; 自动模式
OR 5.14  ; 前端设备对接输入信号（公共）
ANDLD
RSET W3.00  ; 上游设备运行允许（SW）（屏蔽=1）
LD TR0
LD P_First_Cycle
@OR W1.01  ; 自动模式
OR 5.15  ; 后端设备对接输入信号（公共）
ANDLD
RSET W3.01  ; 下游设备放料允许（SW）（屏蔽=1）

### Section 入料扫码RS232_Port0

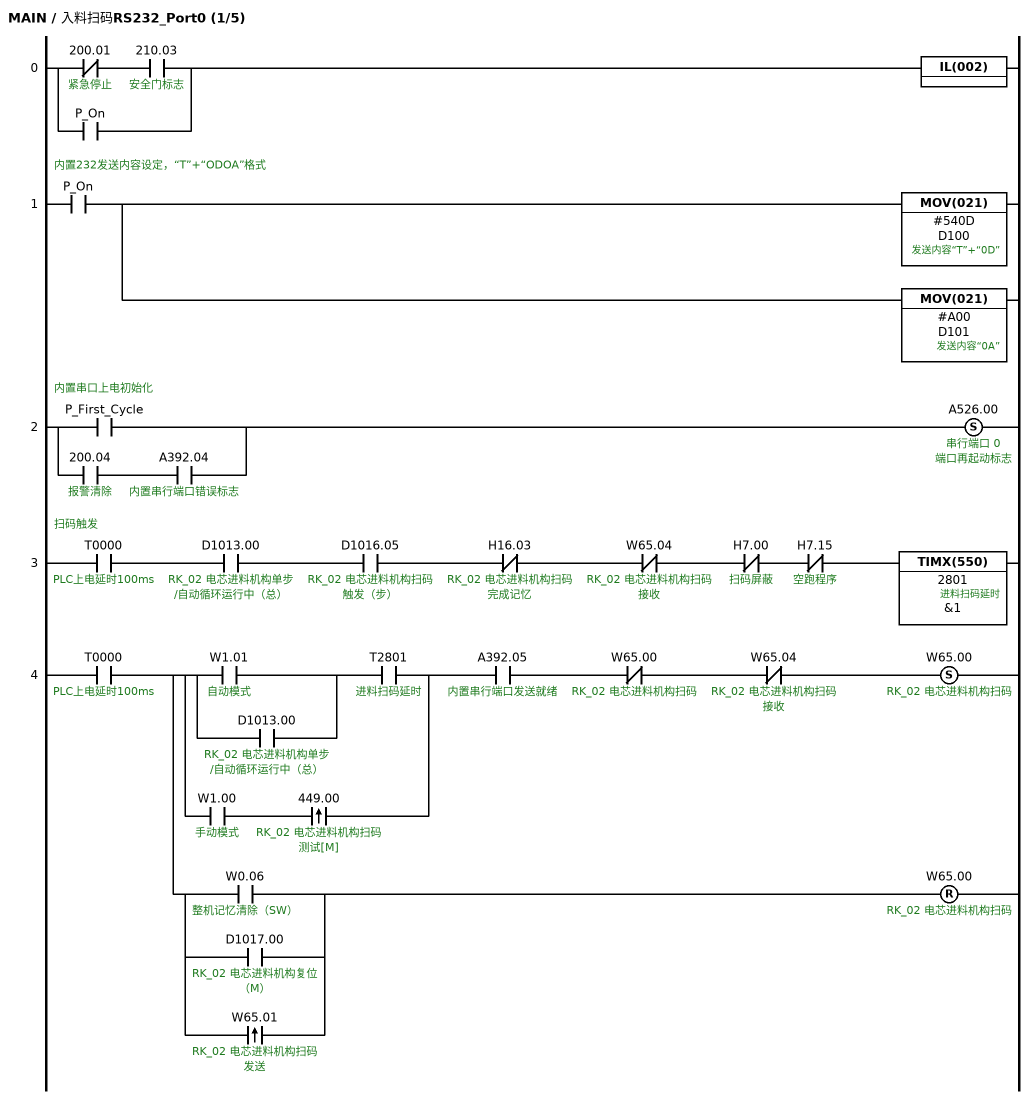
; rung 0
LDNOT 200.01  ; 紧急停止
AND 210.03  ; 安全门标志
OR P_On
IL(002)
; rung 1: 内置232发送内容设定，“T”+“ODOA”格式
LD P_On
MOV(021) #540D D100  ; 发送内容“T”+“0D”
MOV(021) #A00 D101  ; 发送内容“0A”
; rung 2: 内置串口上电初始化
LD P_First_Cycle
LD 200.04  ; 报警清除
AND A392.04  ; 内置串行端口错误标志
ORLD
SET A526.00  ; 串行端口 0 端口再起动标志
; rung 3: 扫码触发
LD T0000  ; PLC上电延时100ms
AND D1013.00  ; RK_02 电芯进料机构单步/自动循环运行中（总）
AND D1016.05  ; RK_02 电芯进料机构扫码触发（步）
ANDNOT H16.03  ; RK_02 电芯进料机构扫码完成记忆
ANDNOT W65.04  ; RK_02 电芯进料机构扫码接收
ANDNOT H7.00  ; 扫码屏蔽
ANDNOT H7.15  ; 空跑程序
TIMX(550) 2801 &1  ; 进料扫码延时
; rung 4
LD T0000  ; PLC上电延时100ms
OUT TR0
LD W1.01  ; 自动模式
OR D1013.00  ; RK_02 电芯进料机构单步/自动循环运行中（总）
AND T2801  ; 进料扫码延时
LD W1.00  ; 手动模式
@AND 449.00  ; RK_02 电芯进料机构扫码测试[M]
ORLD
ANDLD
AND A392.05  ; 内置串行端口发送就绪
ANDNOT W65.00  ; RK_02 电芯进料机构扫码
ANDNOT W65.04  ; RK_02 电芯进料机构扫码接收
SET W65.00  ; RK_02 电芯进料机构扫码
LD TR0
LD W0.06  ; 整机记忆清除（SW）
OR D1017.00  ; RK_02 电芯进料机构复位（M）
@OR W65.01  ; RK_02 电芯进料机构扫码发送
ANDLD
RSET W65.00  ; RK_02 电芯进料机构扫码

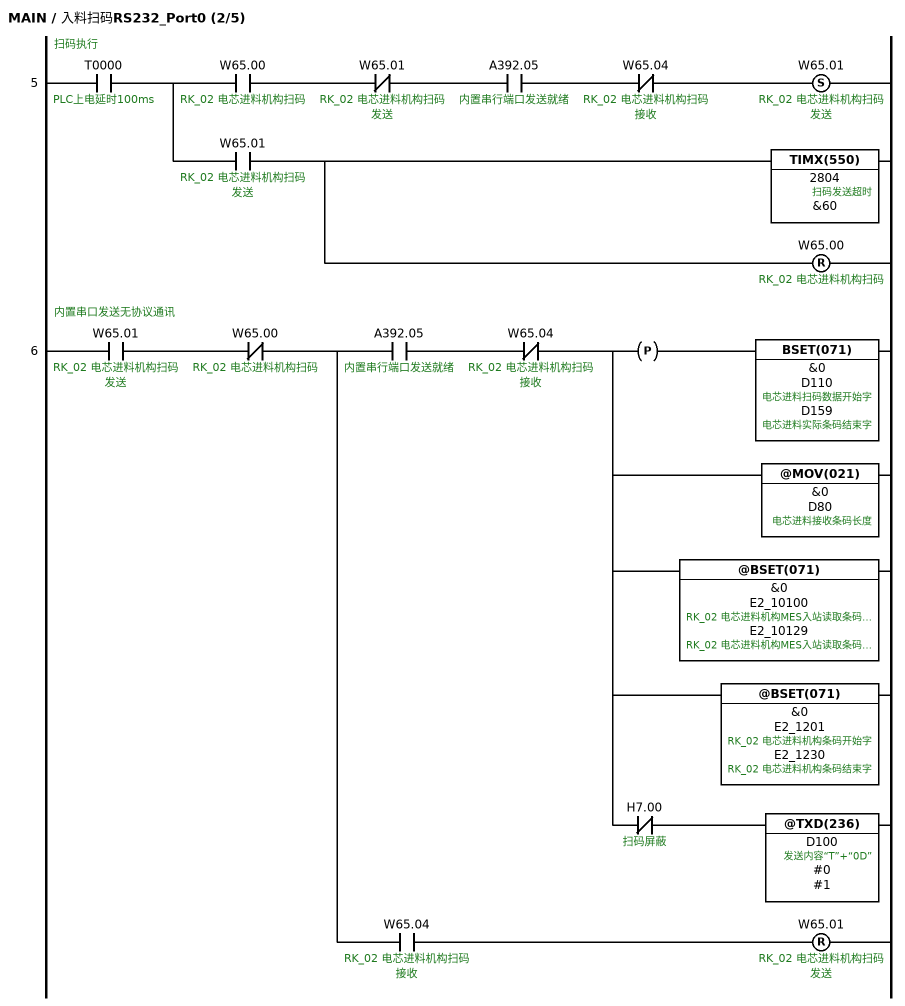
; rung 5: 扫码执行
LD T0000  ; PLC上电延时100ms
OUT TR0
AND W65.00  ; RK_02 电芯进料机构扫码
ANDNOT W65.01  ; RK_02 电芯进料机构扫码发送
AND A392.05  ; 内置串行端口发送就绪
ANDNOT W65.04  ; RK_02 电芯进料机构扫码接收
SET W65.01  ; RK_02 电芯进料机构扫码发送
LD TR0
AND W65.01  ; RK_02 电芯进料机构扫码发送
TIMX(550) 2804 &60  ; 扫码发送超时
RSET W65.00  ; RK_02 电芯进料机构扫码
; rung 6: 内置串口发送无协议通讯
LD W65.01  ; RK_02 电芯进料机构扫码发送
ANDNOT W65.00  ; RK_02 电芯进料机构扫码
OUT TR0
AND A392.05  ; 内置串行端口发送就绪
ANDNOT W65.04  ; RK_02 电芯进料机构扫码接收
OUT TR1
UP(521)
BSET(071) &0 D110 D159  ; 电芯进料扫码数据开始字, 电芯进料实际条码结束字
LD TR1
@MOV(021) &0 D80  ; 电芯进料接收条码长度
@BSET(071) &0 E2_10100 E2_10129  ; RK_02 电芯进料机构MES入站读取条码开始字, RK_02 电芯进料机构MES入站读取条码结束字
@BSET(071) &0 E2_1201 E2_1230  ; RK_02 电芯进料机构条码开始字, RK_02 电芯进料机构条码结束字
ANDNOT H7.00  ; 扫码屏蔽
@TXD(236) D100 #0 #1  ; 发送内容“T”+“0D”
LD TR0
AND W65.04  ; RK_02 电芯进料机构扫码接收
RSET W65.01  ; RK_02 电芯进料机构扫码发送

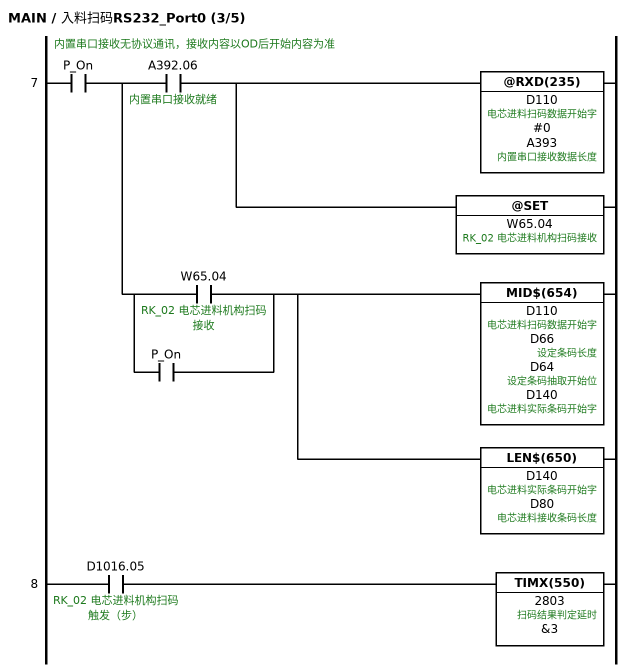
; rung 7: 内置串口接收无协议通讯，接收内容以OD后开始内容为准
LD P_On
OUT TR0
AND A392.06  ; 内置串口接收就绪
@RXD(235) D110 #0 A393  ; 电芯进料扫码数据开始字, 内置串口接收数据长度
@SET W65.04  ; RK_02 电芯进料机构扫码接收
LD TR0
LD W65.04  ; RK_02 电芯进料机构扫码接收
OR P_On
ANDLD
MID$(654) D110 D66 D64 D140  ; 电芯进料扫码数据开始字, 设定条码长度, 设定条码抽取开始位, 电芯进料实际条码开始字
LEN$(650) D140 D80  ; 电芯进料实际条码开始字, 电芯进料接收条码长度
; rung 8
LD D1016.05  ; RK_02 电芯进料机构扫码触发（步）
TIMX(550) 2803 &3  ; 扫码结果判定延时

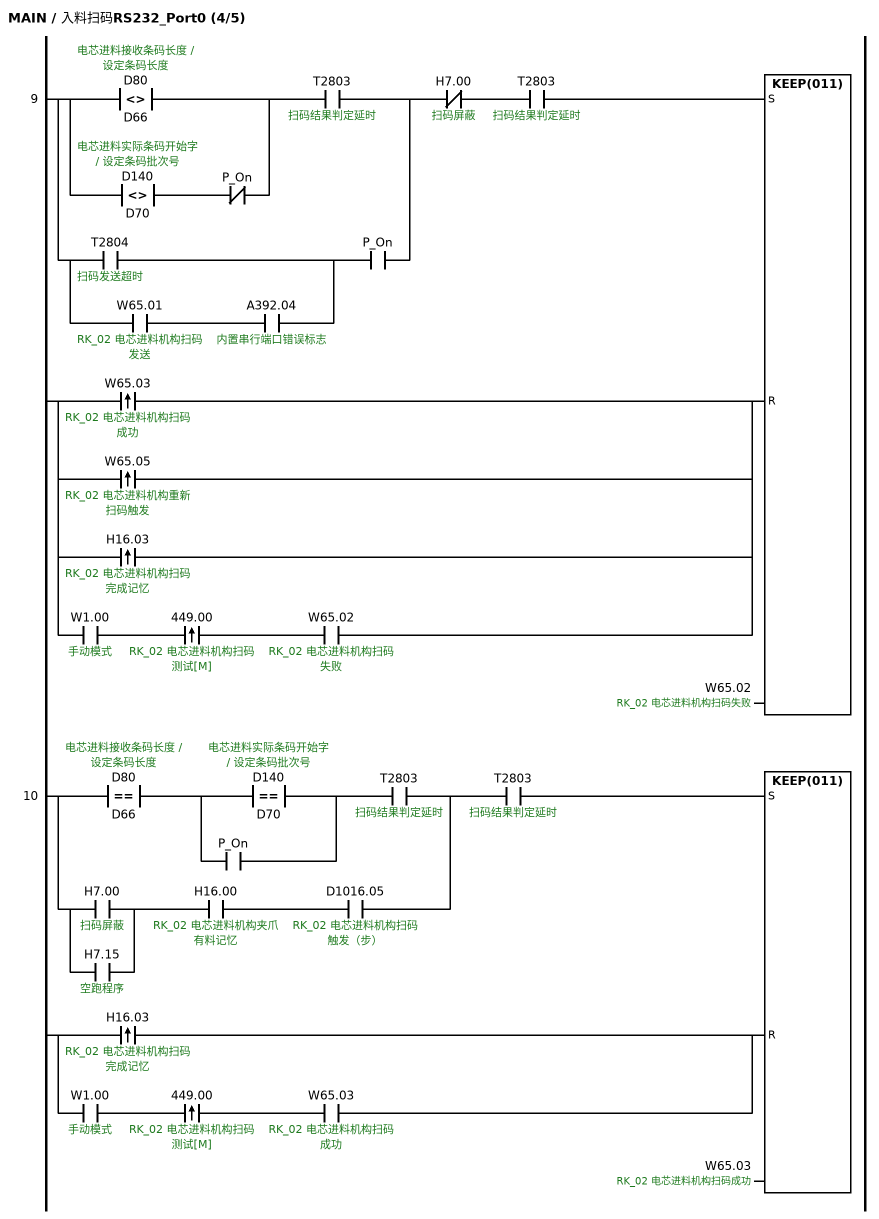
; rung 9
LD<>(305) D80 D66  ; 电芯进料接收条码长度, 设定条码长度
LD<>$(671) D140 D70  ; 电芯进料实际条码开始字, 设定条码批次号
ANDNOT P_On
ORLD
AND T2803  ; 扫码结果判定延时
LD T2804  ; 扫码发送超时
LD W65.01  ; RK_02 电芯进料机构扫码发送
AND A392.04  ; 内置串行端口错误标志
ORLD
AND P_On
ORLD
ANDNOT H7.00  ; 扫码屏蔽
AND T2803  ; 扫码结果判定延时
@LD W65.03  ; RK_02 电芯进料机构扫码成功
@OR W65.05  ; RK_02 电芯进料机构重新扫码触发
@OR H16.03  ; RK_02 电芯进料机构扫码完成记忆
LD W1.00  ; 手动模式
@AND 449.00  ; RK_02 电芯进料机构扫码测试[M]
AND W65.02  ; RK_02 电芯进料机构扫码失败
ORLD
KEEP(011) W65.02  ; RK_02 电芯进料机构扫码失败
; rung 10
LD=(300) D80 D66  ; 电芯进料接收条码长度, 设定条码长度
LD=$(670) D140 D70  ; 电芯进料实际条码开始字, 设定条码批次号
OR P_On
ANDLD
AND T2803  ; 扫码结果判定延时
LD H7.00  ; 扫码屏蔽
OR H7.15  ; 空跑程序
AND H16.00  ; RK_02 电芯进料机构夹爪有料记忆
AND D1016.05  ; RK_02 电芯进料机构扫码触发（步）
ORLD
AND T2803  ; 扫码结果判定延时
@LD H16.03  ; RK_02 电芯进料机构扫码完成记忆
LD W1.00  ; 手动模式
@AND 449.00  ; RK_02 电芯进料机构扫码测试[M]
AND W65.03  ; RK_02 电芯进料机构扫码成功
ORLD
KEEP(011) W65.03  ; RK_02 电芯进料机构扫码成功

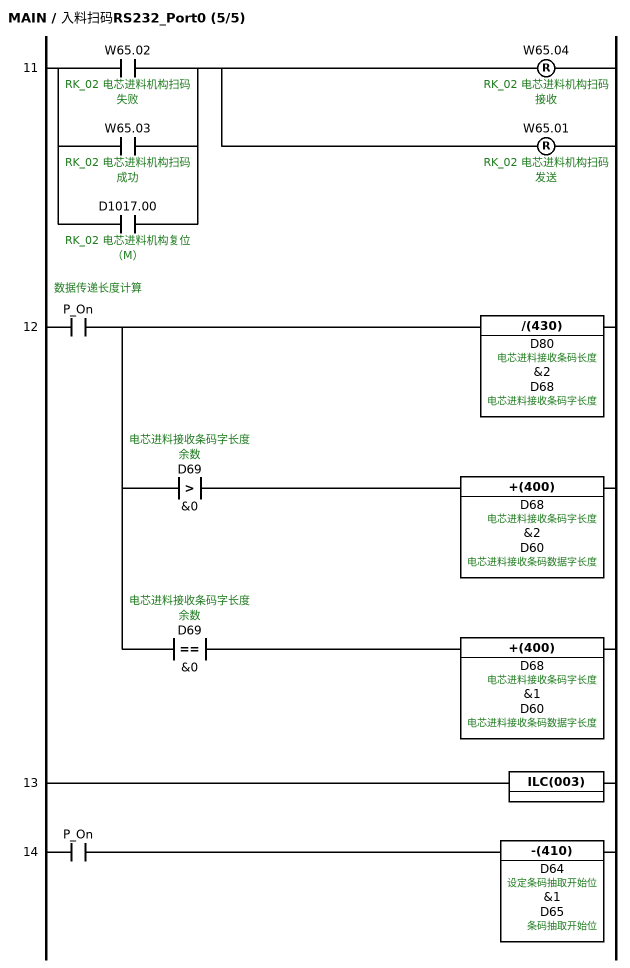
; rung 11
LD W65.02  ; RK_02 电芯进料机构扫码失败
OR W65.03  ; RK_02 电芯进料机构扫码成功
OR D1017.00  ; RK_02 电芯进料机构复位（M）
RSET W65.04  ; RK_02 电芯进料机构扫码接收
RSET W65.01  ; RK_02 电芯进料机构扫码发送
; rung 12: 数据传递长度计算
LD P_On
OUT TR0
/(430) D80 &2 D68  ; 电芯进料接收条码长度, 电芯进料接收条码字长度
AND>(320) D69 &0  ; 电芯进料接收条码字长度余数
+(400) D68 &2 D60  ; 电芯进料接收条码字长度, 电芯进料接收条码数据字长度
LD TR0
AND=(300) D69 &0  ; 电芯进料接收条码字长度余数
+(400) D68 &1 D60  ; 电芯进料接收条码字长度, 电芯进料接收条码数据字长度
; rung 13
ILC(003)
; rung 14
LD P_On
-(410) D64 &1 D65  ; 设定条码抽取开始位, 条码抽取开始位

### Section 轮廓仪SCU21_1550_Port1

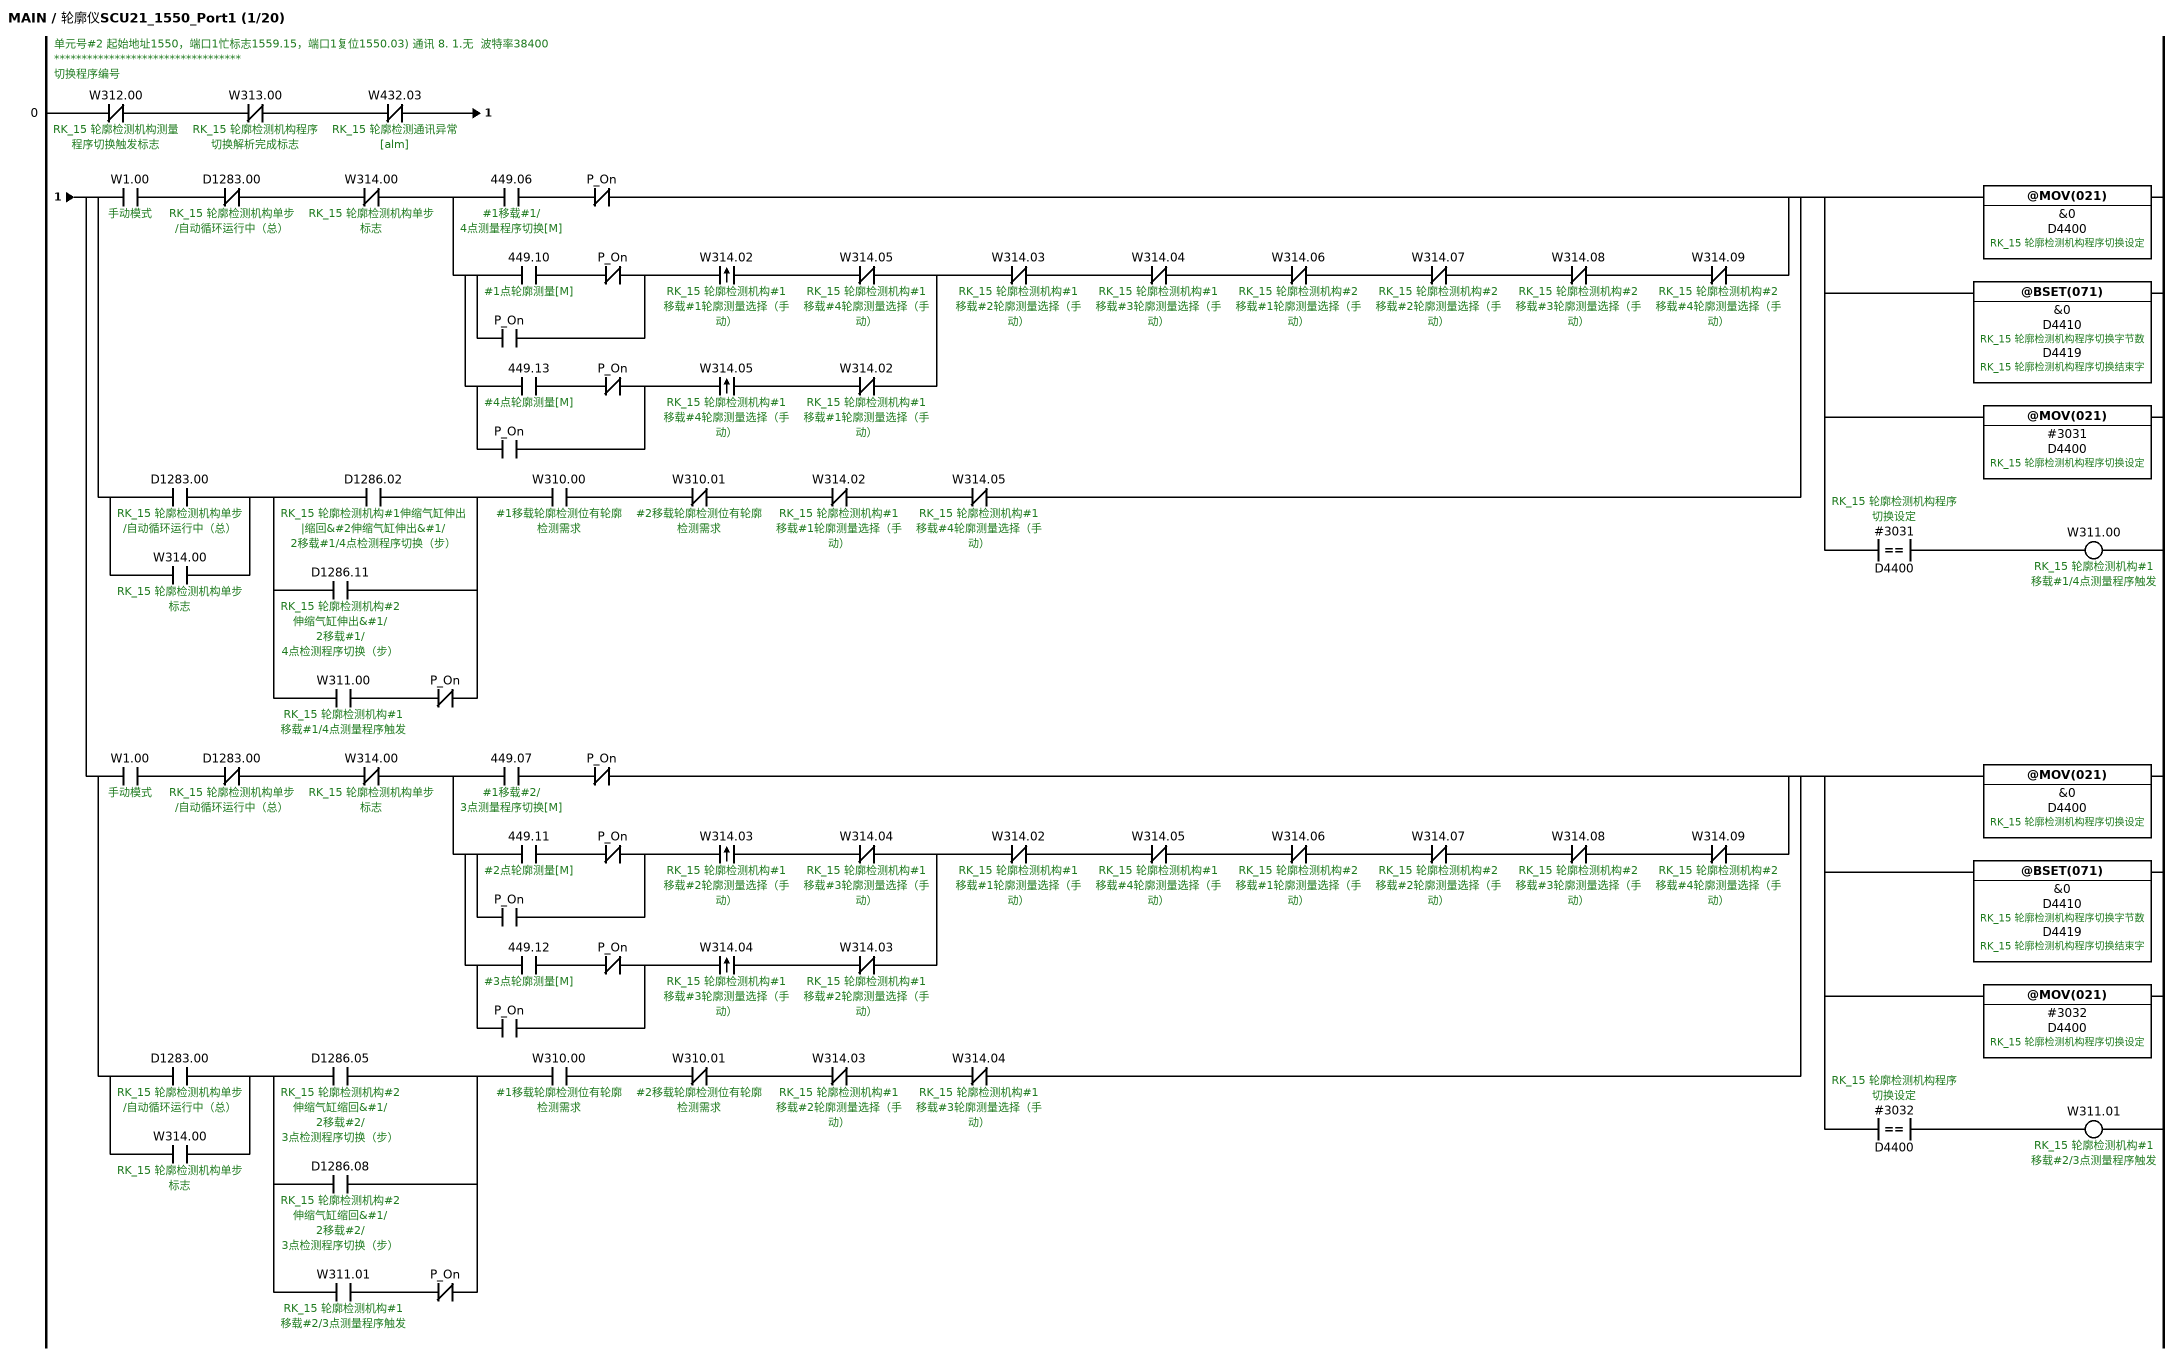
; rung 0: 单元号#2 起始地址1550，端口1忙标志1559.15，端口1复位1550.03) 通讯 8. 1.无  波特率38400 / ********************************** / 切换程序编号
LDNOT W312.00  ; RK_15 轮廓检测机构测量程序切换触发标志
ANDNOT W313.00  ; RK_15 轮廓检测机构程序切换解析完成标志
ANDNOT W432.03  ; RK_15 轮廓检测通讯异常[alm]
OUT TR0
LD W1.00  ; 手动模式
ANDNOT D1283.00  ; RK_15 轮廓检测机构单步/自动循环运行中（总）
ANDNOT W314.00  ; RK_15 轮廓检测机构单步标志
LD 449.06  ; #1移载#1/4点测量程序切换[M]
ANDNOT P_On
LD 449.10  ; #1点轮廓测量[M]
ANDNOT P_On
OR P_On
@AND W314.02  ; RK_15 轮廓检测机构#1移载#1轮廓测量选择（手动）  // HMI按钮操作模式为“切换开关”
ANDNOT W314.05  ; RK_15 轮廓检测机构#1移载#4轮廓测量选择（手动）
LD 449.13  ; #4点轮廓测量[M]
ANDNOT P_On
OR P_On
@AND W314.05  ; RK_15 轮廓检测机构#1移载#4轮廓测量选择（手动）  // HMI按钮操作模式为“切换开关”
ANDNOT W314.02  ; RK_15 轮廓检测机构#1移载#1轮廓测量选择（手动）
ORLD
ANDNOT W314.03  ; RK_15 轮廓检测机构#1移载#2轮廓测量选择（手动）
ANDNOT W314.04  ; RK_15 轮廓检测机构#1移载#3轮廓测量选择（手动）
ANDNOT W314.06  ; RK_15 轮廓检测机构#2移载#1轮廓测量选择（手动）
ANDNOT W314.07  ; RK_15 轮廓检测机构#2移载#2轮廓测量选择（手动）
ANDNOT W314.08  ; RK_15 轮廓检测机构#2移载#3轮廓测量选择（手动）
ANDNOT W314.09  ; RK_15 轮廓检测机构#2移载#4轮廓测量选择（手动）
ORLD
ANDLD
LD D1283.00  ; RK_15 轮廓检测机构单步/自动循环运行中（总）
OR W314.00  ; RK_15 轮廓检测机构单步标志
LD D1286.02  ; RK_15 轮廓检测机构#1伸缩气缸伸出|缩回&#2伸缩气缸伸出&#1/2移载#1/4点检测程序切换（步）
OR D1286.11  ; RK_15 轮廓检测机构#2伸缩气缸伸出&#1/2移载#1/4点检测程序切换（步）
LD W311.00  ; RK_15 轮廓检测机构#1移载#1/4点测量程序触发
ANDNOT P_On
ORLD
ANDLD
AND W310.00  ; #1移载轮廓检测位有轮廓检测需求
ANDNOT W310.01  ; #2移载轮廓检测位有轮廓检测需求
ANDNOT W314.02  ; RK_15 轮廓检测机构#1移载#1轮廓测量选择（手动）
ANDNOT W314.05  ; RK_15 轮廓检测机构#1移载#4轮廓测量选择（手动）
ORLD
ANDLD
@MOV(021) &0 D4400  ; RK_15 轮廓检测机构程序切换设定
@BSET(071) &0 D4410 D4419  ; RK_15 轮廓检测机构程序切换字节数, RK_15 轮廓检测机构程序切换结束字
@MOV(021) #3031 D4400  ; RK_15 轮廓检测机构程序切换设定  // #1移载#1/4点测量程序
AND=(300) #3031 D4400  ; RK_15 轮廓检测机构程序切换设定
OUT W311.00  ; RK_15 轮廓检测机构#1移载#1/4点测量程序触发
LD TR0
LD W1.00  ; 手动模式
ANDNOT D1283.00  ; RK_15 轮廓检测机构单步/自动循环运行中（总）
ANDNOT W314.00  ; RK_15 轮廓检测机构单步标志
LD 449.07  ; #1移载#2/3点测量程序切换[M]
ANDNOT P_On
LD 449.11  ; #2点轮廓测量[M]
ANDNOT P_On
OR P_On
@AND W314.03  ; RK_15 轮廓检测机构#1移载#2轮廓测量选择（手动）  // HMI按钮操作模式为“切换开关”
ANDNOT W314.04  ; RK_15 轮廓检测机构#1移载#3轮廓测量选择（手动）
LD 449.12  ; #3点轮廓测量[M]
ANDNOT P_On
OR P_On
@AND W314.04  ; RK_15 轮廓检测机构#1移载#3轮廓测量选择（手动）  // HMI按钮操作模式为“切换开关”
ANDNOT W314.03  ; RK_15 轮廓检测机构#1移载#2轮廓测量选择（手动）
ORLD
ANDNOT W314.02  ; RK_15 轮廓检测机构#1移载#1轮廓测量选择（手动）
ANDNOT W314.05  ; RK_15 轮廓检测机构#1移载#4轮廓测量选择（手动）
ANDNOT W314.06  ; RK_15 轮廓检测机构#2移载#1轮廓测量选择（手动）
ANDNOT W314.07  ; RK_15 轮廓检测机构#2移载#2轮廓测量选择（手动）
ANDNOT W314.08  ; RK_15 轮廓检测机构#2移载#3轮廓测量选择（手动）
ANDNOT W314.09  ; RK_15 轮廓检测机构#2移载#4轮廓测量选择（手动）
ORLD
ANDLD
LD D1283.00  ; RK_15 轮廓检测机构单步/自动循环运行中（总）
OR W314.00  ; RK_15 轮廓检测机构单步标志
LD D1286.05  ; RK_15 轮廓检测机构#2伸缩气缸缩回&#1/2移载#2/3点检测程序切换（步）
OR D1286.08  ; RK_15 轮廓检测机构#2伸缩气缸缩回&#1/2移载#2/3点检测程序切换（步）
LD W311.01  ; RK_15 轮廓检测机构#1移载#2/3点测量程序触发
ANDNOT P_On
ORLD
ANDLD
AND W310.00  ; #1移载轮廓检测位有轮廓检测需求
ANDNOT W310.01  ; #2移载轮廓检测位有轮廓检测需求
ANDNOT W314.03  ; RK_15 轮廓检测机构#1移载#2轮廓测量选择（手动）
ANDNOT W314.04  ; RK_15 轮廓检测机构#1移载#3轮廓测量选择（手动）
ORLD
ANDLD
@MOV(021) &0 D4400  ; RK_15 轮廓检测机构程序切换设定
@BSET(071) &0 D4410 D4419  ; RK_15 轮廓检测机构程序切换字节数, RK_15 轮廓检测机构程序切换结束字
@MOV(021) #3032 D4400  ; RK_15 轮廓检测机构程序切换设定  // #1移载#2/3点测量程序
AND=(300) #3032 D4400  ; RK_15 轮廓检测机构程序切换设定
OUT W311.01  ; RK_15 轮廓检测机构#1移载#2/3点测量程序触发

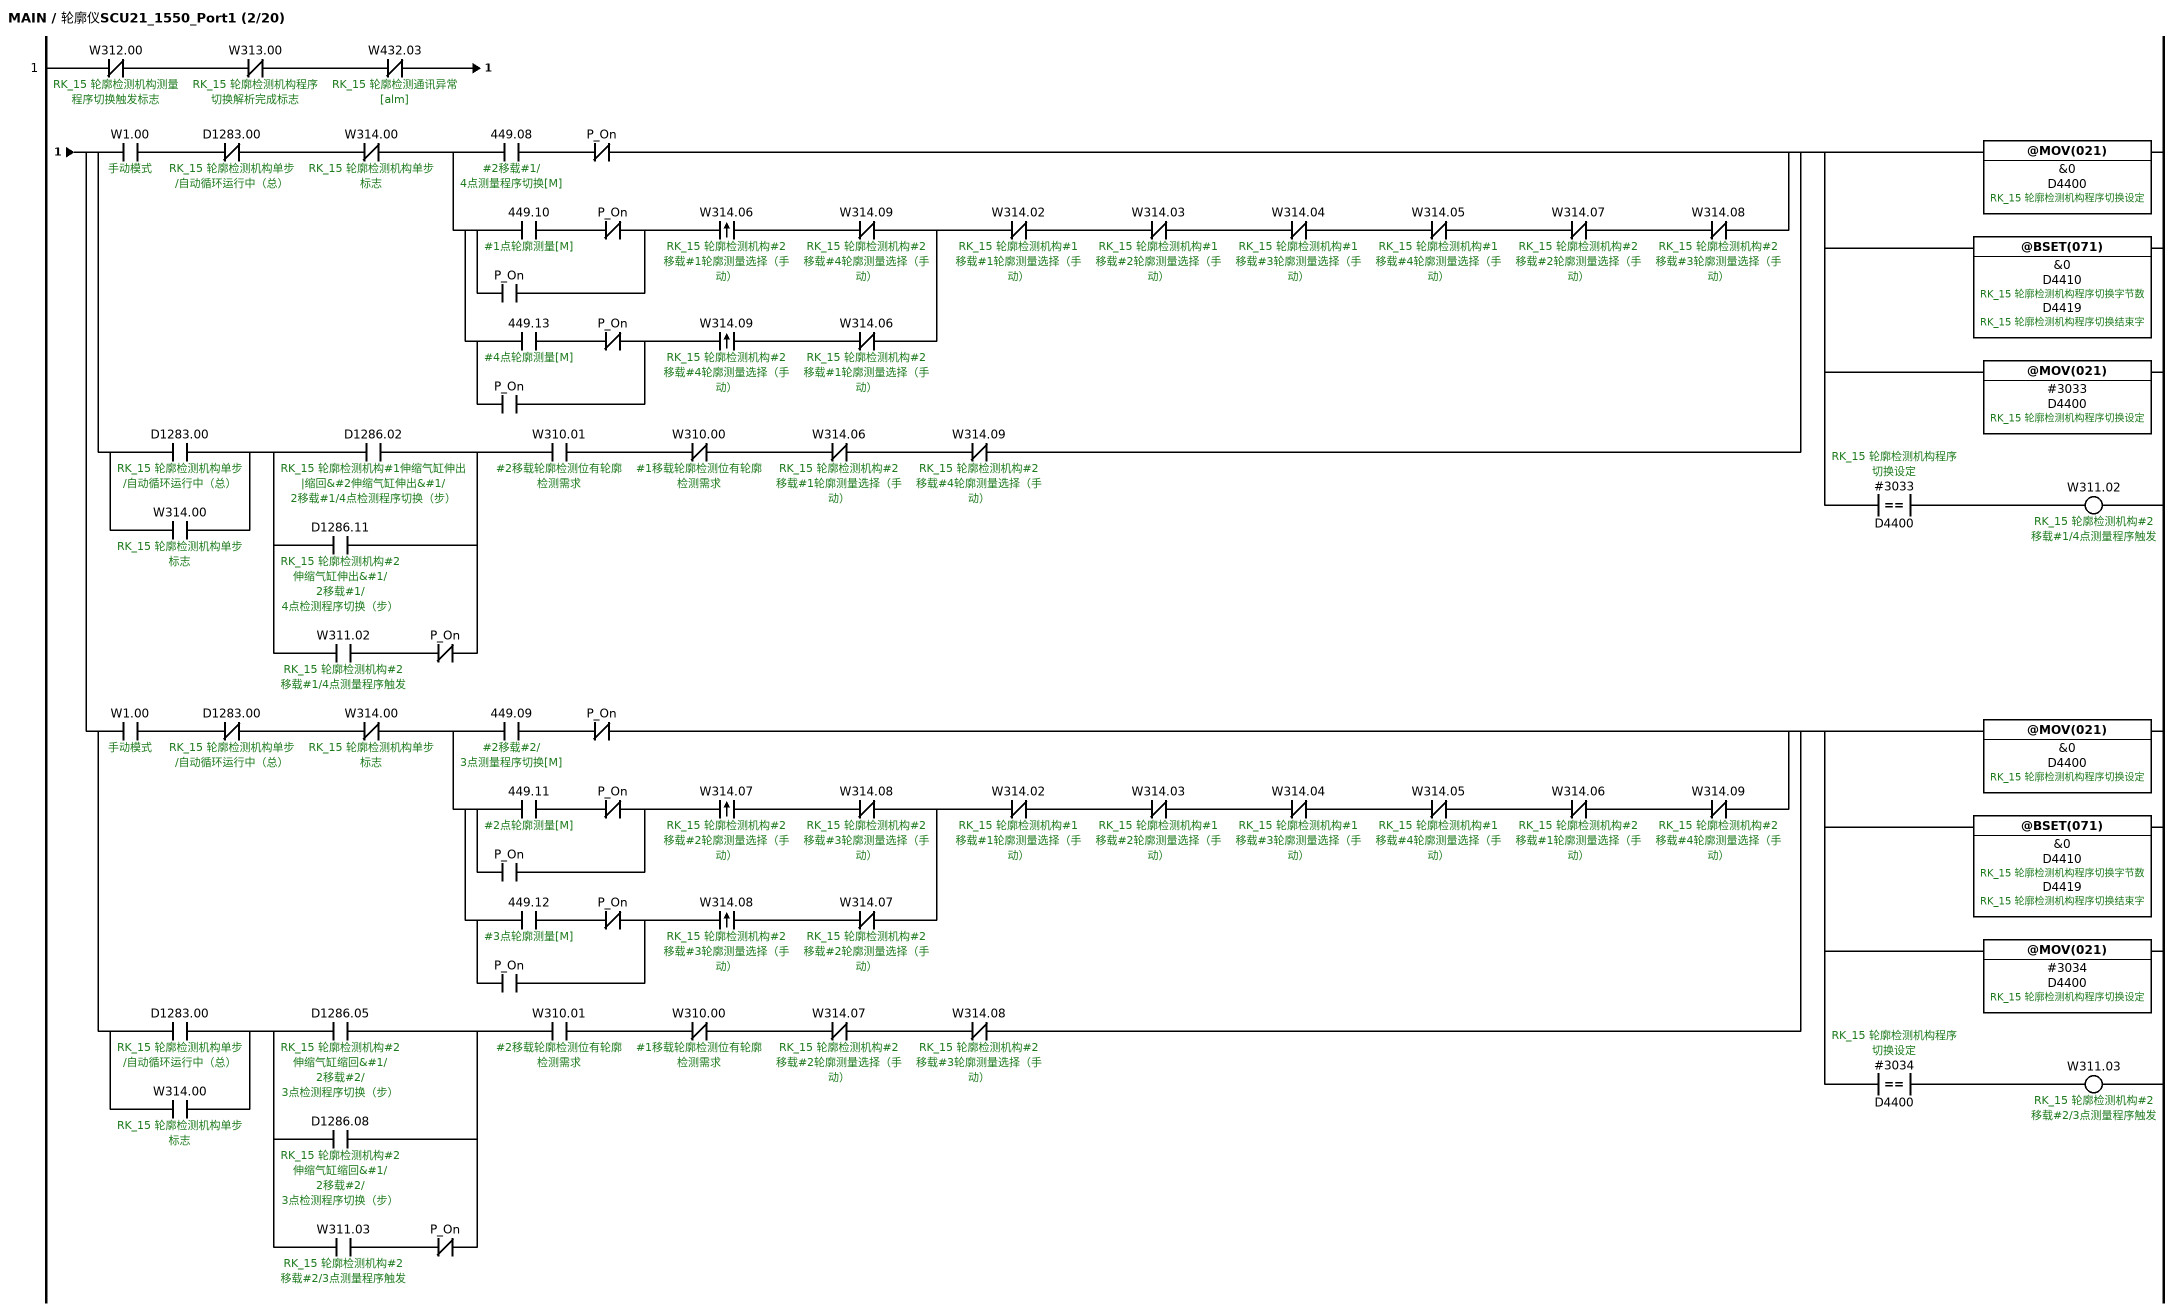
; rung 1
LDNOT W312.00  ; RK_15 轮廓检测机构测量程序切换触发标志
ANDNOT W313.00  ; RK_15 轮廓检测机构程序切换解析完成标志
ANDNOT W432.03  ; RK_15 轮廓检测通讯异常[alm]
OUT TR0
LD W1.00  ; 手动模式
ANDNOT D1283.00  ; RK_15 轮廓检测机构单步/自动循环运行中（总）
ANDNOT W314.00  ; RK_15 轮廓检测机构单步标志
LD 449.08  ; #2移载#1/4点测量程序切换[M]
ANDNOT P_On
LD 449.10  ; #1点轮廓测量[M]
ANDNOT P_On
OR P_On
@AND W314.06  ; RK_15 轮廓检测机构#2移载#1轮廓测量选择（手动）  // HMI按钮操作模式为“切换开关”
ANDNOT W314.09  ; RK_15 轮廓检测机构#2移载#4轮廓测量选择（手动）
LD 449.13  ; #4点轮廓测量[M]
ANDNOT P_On
OR P_On
@AND W314.09  ; RK_15 轮廓检测机构#2移载#4轮廓测量选择（手动）  // HMI按钮操作模式为“切换开关”
ANDNOT W314.06  ; RK_15 轮廓检测机构#2移载#1轮廓测量选择（手动）
ORLD
ANDNOT W314.02  ; RK_15 轮廓检测机构#1移载#1轮廓测量选择（手动）
ANDNOT W314.03  ; RK_15 轮廓检测机构#1移载#2轮廓测量选择（手动）
ANDNOT W314.04  ; RK_15 轮廓检测机构#1移载#3轮廓测量选择（手动）
ANDNOT W314.05  ; RK_15 轮廓检测机构#1移载#4轮廓测量选择（手动）
ANDNOT W314.07  ; RK_15 轮廓检测机构#2移载#2轮廓测量选择（手动）
ANDNOT W314.08  ; RK_15 轮廓检测机构#2移载#3轮廓测量选择（手动）
ORLD
ANDLD
LD D1283.00  ; RK_15 轮廓检测机构单步/自动循环运行中（总）
OR W314.00  ; RK_15 轮廓检测机构单步标志
LD D1286.02  ; RK_15 轮廓检测机构#1伸缩气缸伸出|缩回&#2伸缩气缸伸出&#1/2移载#1/4点检测程序切换（步）
OR D1286.11  ; RK_15 轮廓检测机构#2伸缩气缸伸出&#1/2移载#1/4点检测程序切换（步）
LD W311.02  ; RK_15 轮廓检测机构#2移载#1/4点测量程序触发
ANDNOT P_On
ORLD
ANDLD
AND W310.01  ; #2移载轮廓检测位有轮廓检测需求
ANDNOT W310.00  ; #1移载轮廓检测位有轮廓检测需求
ANDNOT W314.06  ; RK_15 轮廓检测机构#2移载#1轮廓测量选择（手动）
ANDNOT W314.09  ; RK_15 轮廓检测机构#2移载#4轮廓测量选择（手动）
ORLD
ANDLD
@MOV(021) &0 D4400  ; RK_15 轮廓检测机构程序切换设定
@BSET(071) &0 D4410 D4419  ; RK_15 轮廓检测机构程序切换字节数, RK_15 轮廓检测机构程序切换结束字
@MOV(021) #3033 D4400  ; RK_15 轮廓检测机构程序切换设定  // #2移载#1/4点测量程序
AND=(300) #3033 D4400  ; RK_15 轮廓检测机构程序切换设定
OUT W311.02  ; RK_15 轮廓检测机构#2移载#1/4点测量程序触发
LD TR0
LD W1.00  ; 手动模式
ANDNOT D1283.00  ; RK_15 轮廓检测机构单步/自动循环运行中（总）
ANDNOT W314.00  ; RK_15 轮廓检测机构单步标志
LD 449.09  ; #2移载#2/3点测量程序切换[M]
ANDNOT P_On
LD 449.11  ; #2点轮廓测量[M]
ANDNOT P_On
OR P_On
@AND W314.07  ; RK_15 轮廓检测机构#2移载#2轮廓测量选择（手动）  // HMI按钮操作模式为“切换开关”
ANDNOT W314.08  ; RK_15 轮廓检测机构#2移载#3轮廓测量选择（手动）
LD 449.12  ; #3点轮廓测量[M]
ANDNOT P_On
OR P_On
@AND W314.08  ; RK_15 轮廓检测机构#2移载#3轮廓测量选择（手动）  // HMI按钮操作模式为“切换开关”
ANDNOT W314.07  ; RK_15 轮廓检测机构#2移载#2轮廓测量选择（手动）
ORLD
ANDNOT W314.02  ; RK_15 轮廓检测机构#1移载#1轮廓测量选择（手动）
ANDNOT W314.03  ; RK_15 轮廓检测机构#1移载#2轮廓测量选择（手动）
ANDNOT W314.04  ; RK_15 轮廓检测机构#1移载#3轮廓测量选择（手动）
ANDNOT W314.05  ; RK_15 轮廓检测机构#1移载#4轮廓测量选择（手动）
ANDNOT W314.06  ; RK_15 轮廓检测机构#2移载#1轮廓测量选择（手动）
ANDNOT W314.09  ; RK_15 轮廓检测机构#2移载#4轮廓测量选择（手动）
ORLD
ANDLD
LD D1283.00  ; RK_15 轮廓检测机构单步/自动循环运行中（总）
OR W314.00  ; RK_15 轮廓检测机构单步标志
LD D1286.05  ; RK_15 轮廓检测机构#2伸缩气缸缩回&#1/2移载#2/3点检测程序切换（步）
OR D1286.08  ; RK_15 轮廓检测机构#2伸缩气缸缩回&#1/2移载#2/3点检测程序切换（步）
LD W311.03  ; RK_15 轮廓检测机构#2移载#2/3点测量程序触发
ANDNOT P_On
ORLD
ANDLD
AND W310.01  ; #2移载轮廓检测位有轮廓检测需求
ANDNOT W310.00  ; #1移载轮廓检测位有轮廓检测需求
ANDNOT W314.07  ; RK_15 轮廓检测机构#2移载#2轮廓测量选择（手动）
ANDNOT W314.08  ; RK_15 轮廓检测机构#2移载#3轮廓测量选择（手动）
ORLD
ANDLD
@MOV(021) &0 D4400  ; RK_15 轮廓检测机构程序切换设定
@BSET(071) &0 D4410 D4419  ; RK_15 轮廓检测机构程序切换字节数, RK_15 轮廓检测机构程序切换结束字
@MOV(021) #3034 D4400  ; RK_15 轮廓检测机构程序切换设定  // #2移载#2/3点测量程序
AND=(300) #3034 D4400  ; RK_15 轮廓检测机构程序切换设定
OUT W311.03  ; RK_15 轮廓检测机构#2移载#2/3点测量程序触发

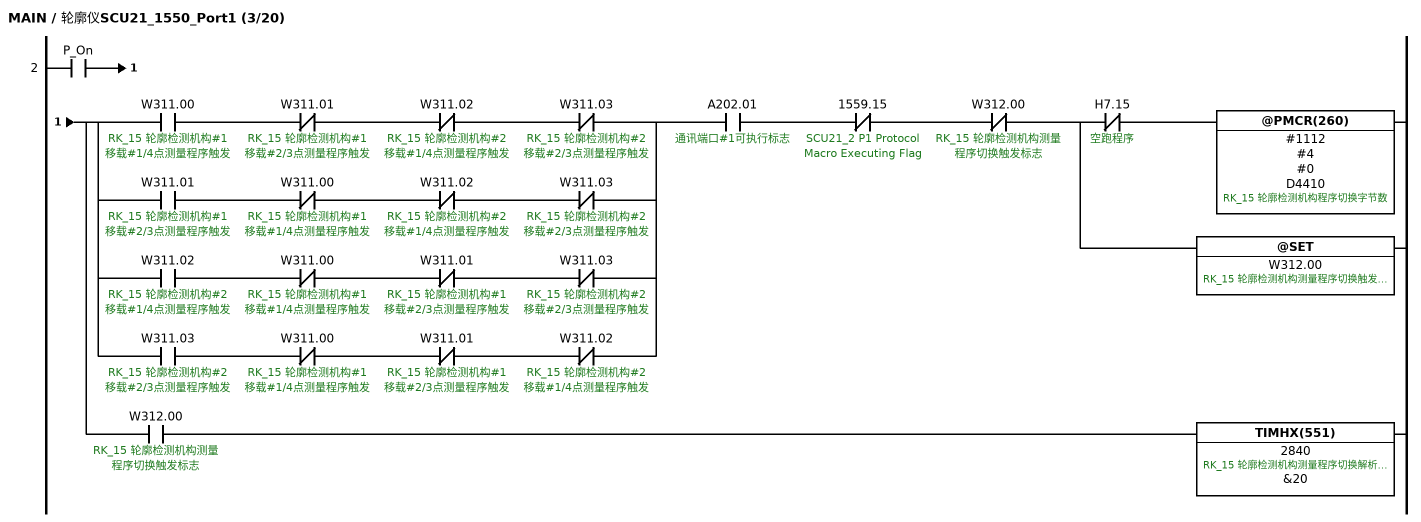
; rung 2
LD P_On
OUT TR0
LD W311.00  ; RK_15 轮廓检测机构#1移载#1/4点测量程序触发
ANDNOT W311.01  ; RK_15 轮廓检测机构#1移载#2/3点测量程序触发
ANDNOT W311.02  ; RK_15 轮廓检测机构#2移载#1/4点测量程序触发
ANDNOT W311.03  ; RK_15 轮廓检测机构#2移载#2/3点测量程序触发
LD W311.01  ; RK_15 轮廓检测机构#1移载#2/3点测量程序触发
ANDNOT W311.00  ; RK_15 轮廓检测机构#1移载#1/4点测量程序触发
ANDNOT W311.02  ; RK_15 轮廓检测机构#2移载#1/4点测量程序触发
ANDNOT W311.03  ; RK_15 轮廓检测机构#2移载#2/3点测量程序触发
ORLD
LD W311.02  ; RK_15 轮廓检测机构#2移载#1/4点测量程序触发
ANDNOT W311.00  ; RK_15 轮廓检测机构#1移载#1/4点测量程序触发
ANDNOT W311.01  ; RK_15 轮廓检测机构#1移载#2/3点测量程序触发
ANDNOT W311.03  ; RK_15 轮廓检测机构#2移载#2/3点测量程序触发
ORLD
LD W311.03  ; RK_15 轮廓检测机构#2移载#2/3点测量程序触发
ANDNOT W311.00  ; RK_15 轮廓检测机构#1移载#1/4点测量程序触发
ANDNOT W311.01  ; RK_15 轮廓检测机构#1移载#2/3点测量程序触发
ANDNOT W311.02  ; RK_15 轮廓检测机构#2移载#1/4点测量程序触发
ORLD
ANDLD
AND A202.01  ; 通讯端口#1可执行标志
ANDNOT 1559.15  ; SCU21_2 P1 Protocol Macro Executing Flag
ANDNOT W312.00  ; RK_15 轮廓检测机构测量程序切换触发标志
OUT TR1
ANDNOT H7.15  ; 空跑程序  // 20181013新增
@PMCR(260) #1112 #4 #0 D4410  ; RK_15 轮廓检测机构程序切换字节数
LD TR1
@SET W312.00  ; RK_15 轮廓检测机构测量程序切换触发标志
LD TR0
AND W312.00  ; RK_15 轮廓检测机构测量程序切换触发标志
TIMHX(551) 2840 &20  ; RK_15 轮廓检测机构测量程序切换解析延时

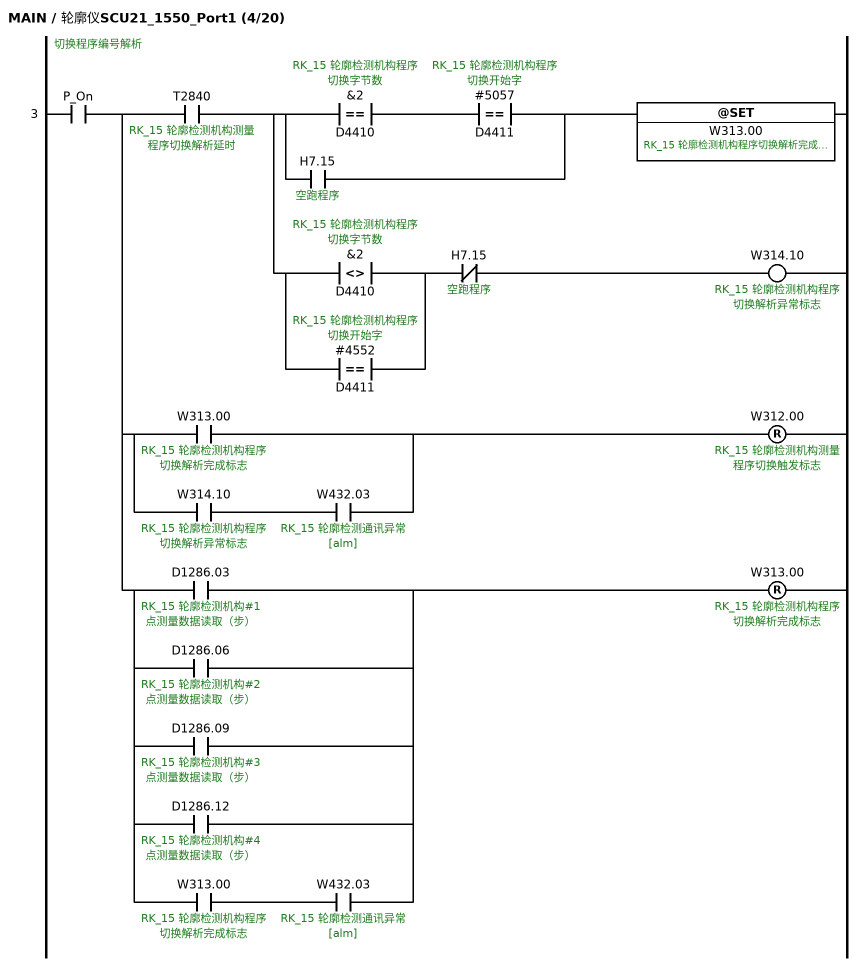
; rung 3: 切换程序编号解析
LD P_On
OUT TR0
AND T2840  ; RK_15 轮廓检测机构测量程序切换解析延时
OUT TR1
LD=(300) &2 D4410  ; RK_15 轮廓检测机构程序切换字节数
AND=(300) #5057 D4411  ; RK_15 轮廓检测机构程序切换开始字
OR H7.15  ; 空跑程序  // 20181013新增
ANDLD
@SET W313.00  ; RK_15 轮廓检测机构程序切换解析完成标志
LD TR1
LD<>(305) &2 D4410  ; RK_15 轮廓检测机构程序切换字节数
OR=(300) #4552 D4411  ; RK_15 轮廓检测机构程序切换开始字
ANDLD
ANDNOT H7.15  ; 空跑程序  // 20181013新增
OUT W314.10  ; RK_15 轮廓检测机构程序切换解析异常标志
LD TR0
LD W313.00  ; RK_15 轮廓检测机构程序切换解析完成标志
LD W314.10  ; RK_15 轮廓检测机构程序切换解析异常标志
AND W432.03  ; RK_15 轮廓检测通讯异常[alm]
ORLD
ANDLD
RSET W312.00  ; RK_15 轮廓检测机构测量程序切换触发标志
LD TR0
LD D1286.03  ; RK_15 轮廓检测机构#1点测量数据读取（步）
OR D1286.06  ; RK_15 轮廓检测机构#2点测量数据读取（步）
OR D1286.09  ; RK_15 轮廓检测机构#3点测量数据读取（步）
OR D1286.12  ; RK_15 轮廓检测机构#4点测量数据读取（步）
LD W313.00  ; RK_15 轮廓检测机构程序切换解析完成标志
AND W432.03  ; RK_15 轮廓检测通讯异常[alm]
ORLD
ANDLD
RSET W313.00  ; RK_15 轮廓检测机构程序切换解析完成标志

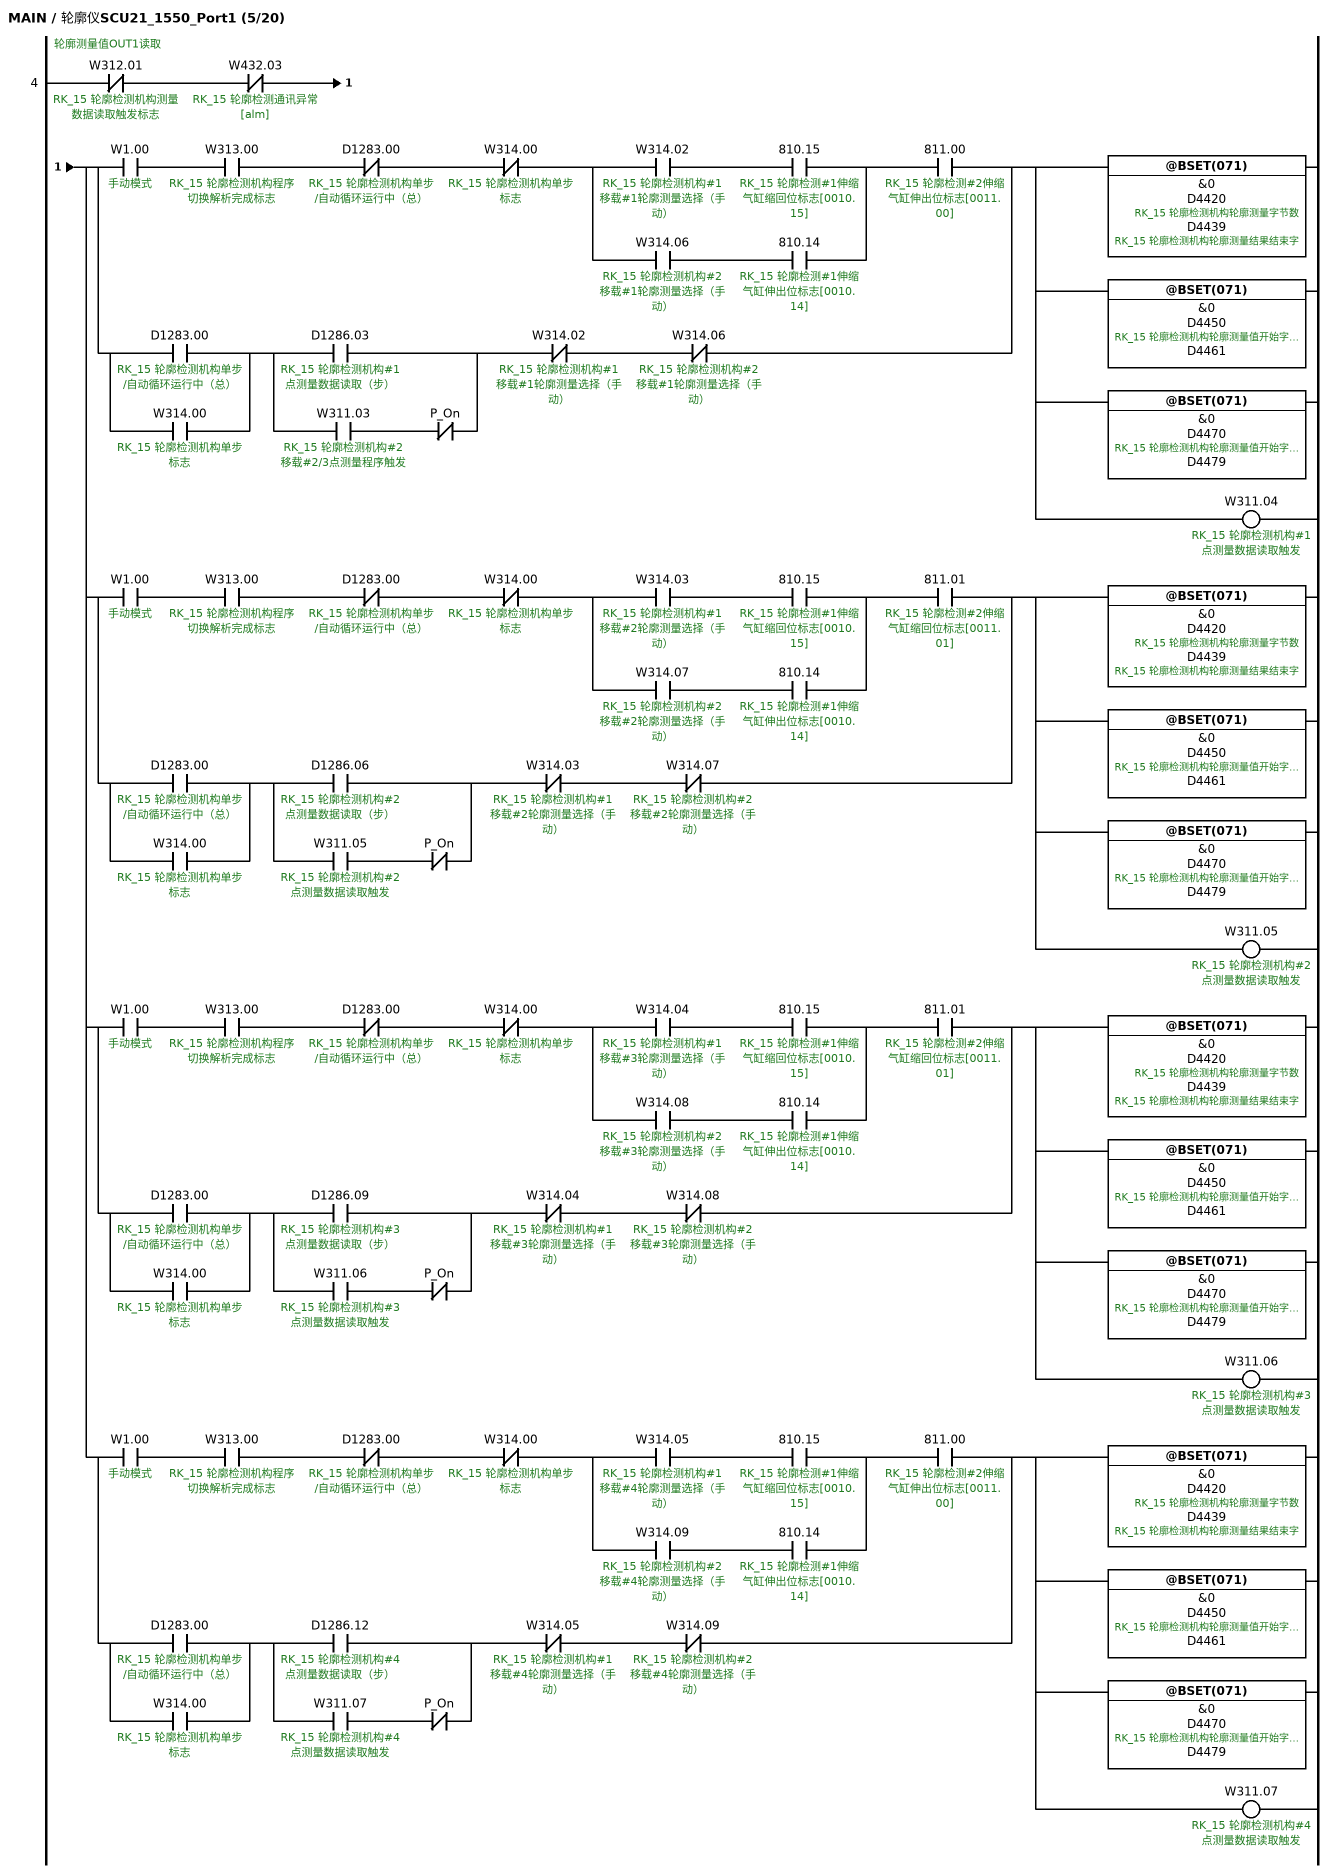
; rung 4: 轮廓测量值OUT1读取
LDNOT W312.01  ; RK_15 轮廓检测机构测量数据读取触发标志
ANDNOT W432.03  ; RK_15 轮廓检测通讯异常[alm]
OUT TR0
LD W1.00  ; 手动模式
AND W313.00  ; RK_15 轮廓检测机构程序切换解析完成标志
ANDNOT D1283.00  ; RK_15 轮廓检测机构单步/自动循环运行中（总）
ANDNOT W314.00  ; RK_15 轮廓检测机构单步标志
LD W314.02  ; RK_15 轮廓检测机构#1移载#1轮廓测量选择（手动）  // HMI按钮操作模式为“切换开关”
AND 810.15  ; RK_15 轮廓检测#1伸缩气缸缩回位标志[0010.15]
LD W314.06  ; RK_15 轮廓检测机构#2移载#1轮廓测量选择（手动）  // HMI按钮操作模式为“切换开关”
AND 810.14  ; RK_15 轮廓检测#1伸缩气缸伸出位标志[0010.14]
ORLD
ANDLD
AND 811.00  ; RK_15 轮廓检测#2伸缩气缸伸出位标志[0011.00]
LD D1283.00  ; RK_15 轮廓检测机构单步/自动循环运行中（总）
OR W314.00  ; RK_15 轮廓检测机构单步标志
LD D1286.03  ; RK_15 轮廓检测机构#1点测量数据读取（步）
LD W311.03  ; RK_15 轮廓检测机构#2移载#2/3点测量程序触发
ANDNOT P_On
ORLD
ANDLD
ANDNOT W314.02  ; RK_15 轮廓检测机构#1移载#1轮廓测量选择（手动）
ANDNOT W314.06  ; RK_15 轮廓检测机构#2移载#1轮廓测量选择（手动）
ORLD
ANDLD
@BSET(071) &0 D4420 D4439  ; RK_15 轮廓检测机构轮廓测量字节数, RK_15 轮廓检测机构轮廓测量结果结束字
@BSET(071) &0 D4450 D4461  ; RK_15 轮廓检测机构轮廓测量值开始字（String）
@BSET(071) &0 D4470 D4479  ; RK_15 轮廓检测机构轮廓测量值开始字（String）
OUT W311.04  ; RK_15 轮廓检测机构#1点测量数据读取触发
LD TR0
LD W1.00  ; 手动模式
AND W313.00  ; RK_15 轮廓检测机构程序切换解析完成标志
ANDNOT D1283.00  ; RK_15 轮廓检测机构单步/自动循环运行中（总）
ANDNOT W314.00  ; RK_15 轮廓检测机构单步标志
LD W314.03  ; RK_15 轮廓检测机构#1移载#2轮廓测量选择（手动）
AND 810.15  ; RK_15 轮廓检测#1伸缩气缸缩回位标志[0010.15]
LD W314.07  ; RK_15 轮廓检测机构#2移载#2轮廓测量选择（手动）
AND 810.14  ; RK_15 轮廓检测#1伸缩气缸伸出位标志[0010.14]
ORLD
ANDLD
AND 811.01  ; RK_15 轮廓检测#2伸缩气缸缩回位标志[0011.01]
LD D1283.00  ; RK_15 轮廓检测机构单步/自动循环运行中（总）
OR W314.00  ; RK_15 轮廓检测机构单步标志
LD D1286.06  ; RK_15 轮廓检测机构#2点测量数据读取（步）
LD W311.05  ; RK_15 轮廓检测机构#2点测量数据读取触发
ANDNOT P_On
ORLD
ANDLD
ANDNOT W314.03  ; RK_15 轮廓检测机构#1移载#2轮廓测量选择（手动）
ANDNOT W314.07  ; RK_15 轮廓检测机构#2移载#2轮廓测量选择（手动）
ORLD
ANDLD
@BSET(071) &0 D4420 D4439  ; RK_15 轮廓检测机构轮廓测量字节数, RK_15 轮廓检测机构轮廓测量结果结束字
@BSET(071) &0 D4450 D4461  ; RK_15 轮廓检测机构轮廓测量值开始字（String）
@BSET(071) &0 D4470 D4479  ; RK_15 轮廓检测机构轮廓测量值开始字（String）
OUT W311.05  ; RK_15 轮廓检测机构#2点测量数据读取触发
LD TR0
LD W1.00  ; 手动模式
AND W313.00  ; RK_15 轮廓检测机构程序切换解析完成标志
ANDNOT D1283.00  ; RK_15 轮廓检测机构单步/自动循环运行中（总）
ANDNOT W314.00  ; RK_15 轮廓检测机构单步标志
LD W314.04  ; RK_15 轮廓检测机构#1移载#3轮廓测量选择（手动）
AND 810.15  ; RK_15 轮廓检测#1伸缩气缸缩回位标志[0010.15]
LD W314.08  ; RK_15 轮廓检测机构#2移载#3轮廓测量选择（手动）
AND 810.14  ; RK_15 轮廓检测#1伸缩气缸伸出位标志[0010.14]
ORLD
ANDLD
AND 811.01  ; RK_15 轮廓检测#2伸缩气缸缩回位标志[0011.01]
LD D1283.00  ; RK_15 轮廓检测机构单步/自动循环运行中（总）
OR W314.00  ; RK_15 轮廓检测机构单步标志
LD D1286.09  ; RK_15 轮廓检测机构#3点测量数据读取（步）
LD W311.06  ; RK_15 轮廓检测机构#3点测量数据读取触发
ANDNOT P_On
ORLD
ANDLD
ANDNOT W314.04  ; RK_15 轮廓检测机构#1移载#3轮廓测量选择（手动）
ANDNOT W314.08  ; RK_15 轮廓检测机构#2移载#3轮廓测量选择（手动）
ORLD
ANDLD
@BSET(071) &0 D4420 D4439  ; RK_15 轮廓检测机构轮廓测量字节数, RK_15 轮廓检测机构轮廓测量结果结束字
@BSET(071) &0 D4450 D4461  ; RK_15 轮廓检测机构轮廓测量值开始字（String）
@BSET(071) &0 D4470 D4479  ; RK_15 轮廓检测机构轮廓测量值开始字（String）
OUT W311.06  ; RK_15 轮廓检测机构#3点测量数据读取触发
LD TR0
LD W1.00  ; 手动模式
AND W313.00  ; RK_15 轮廓检测机构程序切换解析完成标志
ANDNOT D1283.00  ; RK_15 轮廓检测机构单步/自动循环运行中（总）
ANDNOT W314.00  ; RK_15 轮廓检测机构单步标志
LD W314.05  ; RK_15 轮廓检测机构#1移载#4轮廓测量选择（手动）
AND 810.15  ; RK_15 轮廓检测#1伸缩气缸缩回位标志[0010.15]
LD W314.09  ; RK_15 轮廓检测机构#2移载#4轮廓测量选择（手动）
AND 810.14  ; RK_15 轮廓检测#1伸缩气缸伸出位标志[0010.14]
ORLD
ANDLD
AND 811.00  ; RK_15 轮廓检测#2伸缩气缸伸出位标志[0011.00]
LD D1283.00  ; RK_15 轮廓检测机构单步/自动循环运行中（总）
OR W314.00  ; RK_15 轮廓检测机构单步标志
LD D1286.12  ; RK_15 轮廓检测机构#4点测量数据读取（步）
LD W311.07  ; RK_15 轮廓检测机构#4点测量数据读取触发
ANDNOT P_On
ORLD
ANDLD
ANDNOT W314.05  ; RK_15 轮廓检测机构#1移载#4轮廓测量选择（手动）
ANDNOT W314.09  ; RK_15 轮廓检测机构#2移载#4轮廓测量选择（手动）
ORLD
ANDLD
@BSET(071) &0 D4420 D4439  ; RK_15 轮廓检测机构轮廓测量字节数, RK_15 轮廓检测机构轮廓测量结果结束字
@BSET(071) &0 D4450 D4461  ; RK_15 轮廓检测机构轮廓测量值开始字（String）
@BSET(071) &0 D4470 D4479  ; RK_15 轮廓检测机构轮廓测量值开始字（String）
OUT W311.07  ; RK_15 轮廓检测机构#4点测量数据读取触发

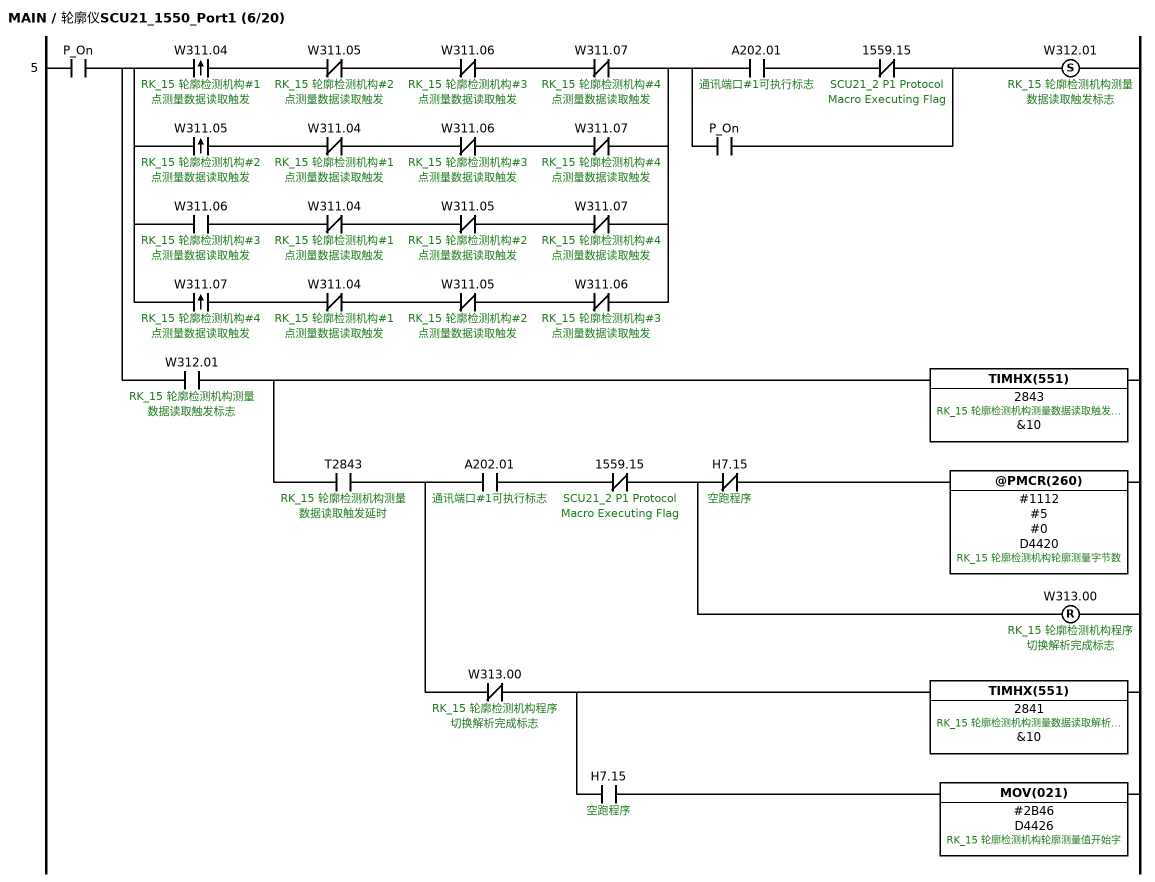
; rung 5
LD P_On
OUT TR0
@LD W311.04  ; RK_15 轮廓检测机构#1点测量数据读取触发
ANDNOT W311.05  ; RK_15 轮廓检测机构#2点测量数据读取触发
ANDNOT W311.06  ; RK_15 轮廓检测机构#3点测量数据读取触发
ANDNOT W311.07  ; RK_15 轮廓检测机构#4点测量数据读取触发
@LD W311.05  ; RK_15 轮廓检测机构#2点测量数据读取触发
ANDNOT W311.04  ; RK_15 轮廓检测机构#1点测量数据读取触发
ANDNOT W311.06  ; RK_15 轮廓检测机构#3点测量数据读取触发
ANDNOT W311.07  ; RK_15 轮廓检测机构#4点测量数据读取触发
ORLD
LD W311.06  ; RK_15 轮廓检测机构#3点测量数据读取触发
ANDNOT W311.04  ; RK_15 轮廓检测机构#1点测量数据读取触发
ANDNOT W311.05  ; RK_15 轮廓检测机构#2点测量数据读取触发
ANDNOT W311.07  ; RK_15 轮廓检测机构#4点测量数据读取触发
ORLD
@LD W311.07  ; RK_15 轮廓检测机构#4点测量数据读取触发
ANDNOT W311.04  ; RK_15 轮廓检测机构#1点测量数据读取触发
ANDNOT W311.05  ; RK_15 轮廓检测机构#2点测量数据读取触发
ANDNOT W311.06  ; RK_15 轮廓检测机构#3点测量数据读取触发
ORLD
ANDLD
LD A202.01  ; 通讯端口#1可执行标志
ANDNOT 1559.15  ; SCU21_2 P1 Protocol Macro Executing Flag
OR P_On
ANDLD
SET W312.01  ; RK_15 轮廓检测机构测量数据读取触发标志
LD TR0
AND W312.01  ; RK_15 轮廓检测机构测量数据读取触发标志
TIMHX(551) 2843 &10  ; RK_15 轮廓检测机构测量数据读取触发延时
AND T2843  ; RK_15 轮廓检测机构测量数据读取触发延时
OUT TR0
AND A202.01  ; 通讯端口#1可执行标志
ANDNOT 1559.15  ; SCU21_2 P1 Protocol Macro Executing Flag
OUT TR1
ANDNOT H7.15  ; 空跑程序  // 20181013新增
@PMCR(260) #1112 #5 #0 D4420  ; RK_15 轮廓检测机构轮廓测量字节数
LD TR1
RSET W313.00  ; RK_15 轮廓检测机构程序切换解析完成标志
LD TR0
ANDNOT W313.00  ; RK_15 轮廓检测机构程序切换解析完成标志
TIMHX(551) 2841 &10  ; RK_15 轮廓检测机构测量数据读取解析延时
AND H7.15  ; 空跑程序  // 20181013新增
MOV(021) #2B46 D4426  ; RK_15 轮廓检测机构轮廓测量值开始字

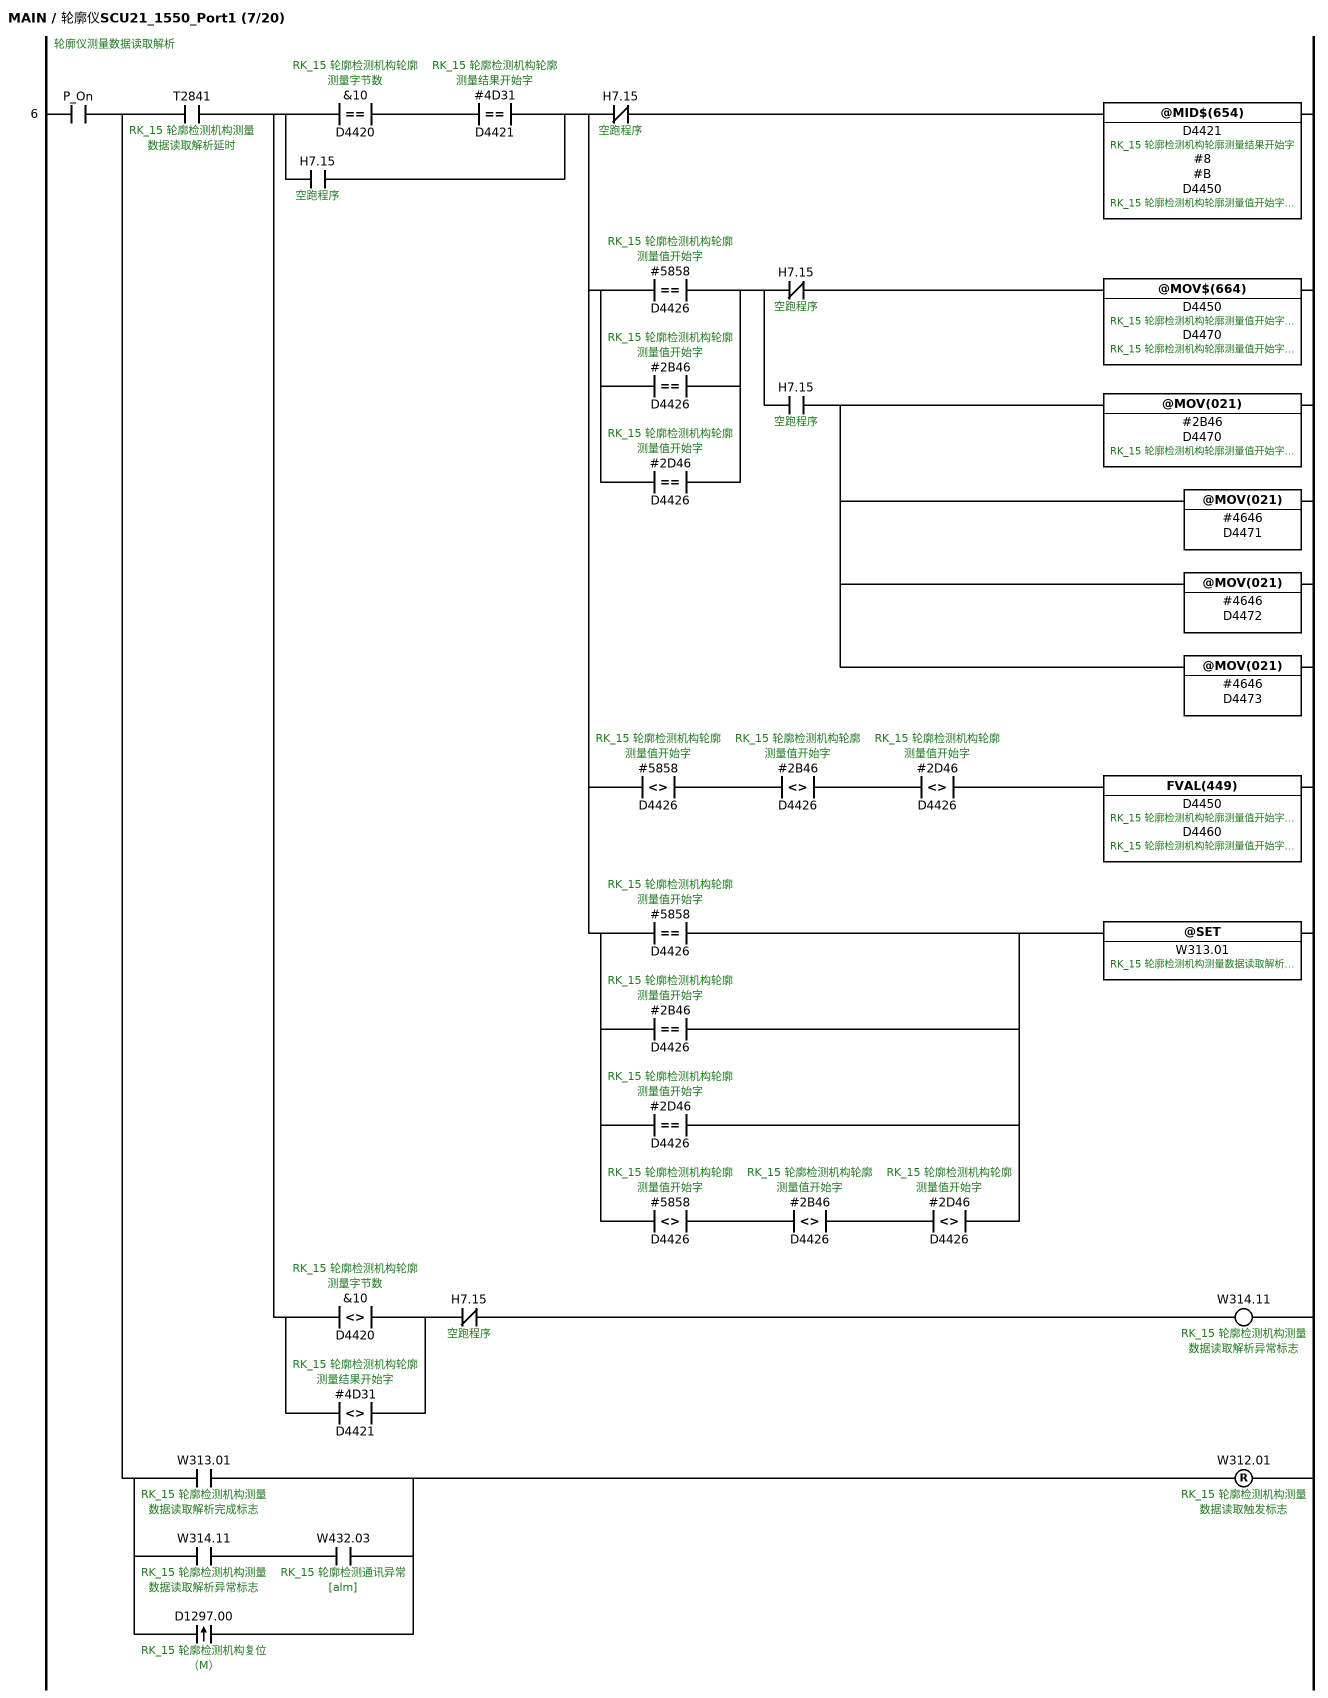
; rung 6: 轮廓仪测量数据读取解析
LD P_On
OUT TR0
AND T2841  ; RK_15 轮廓检测机构测量数据读取解析延时
OUT TR1
LD=(300) &10 D4420  ; RK_15 轮廓检测机构轮廓测量字节数
AND=(300) #4D31 D4421  ; RK_15 轮廓检测机构轮廓测量结果开始字
OR H7.15  ; 空跑程序  // 20181013新增
ANDLD
OUT TR2
ANDNOT H7.15  ; 空跑程序  // 20181013新增
@MID$(654) D4421 #8 #B D4450  ; RK_15 轮廓检测机构轮廓测量结果开始字, RK_15 轮廓检测机构轮廓测量值开始字（String）
LD TR2
LD=(300) #5858 D4426  ; RK_15 轮廓检测机构轮廓测量值开始字
OR=(300) #2B46 D4426  ; RK_15 轮廓检测机构轮廓测量值开始字
OR=(300) #2D46 D4426  ; RK_15 轮廓检测机构轮廓测量值开始字
ANDLD
OUT TR3
ANDNOT H7.15  ; 空跑程序  // 20181013新增
@MOV$(664) D4450 D4470  ; RK_15 轮廓检测机构轮廓测量值开始字（String）
LD TR3
AND H7.15  ; 空跑程序  // 20181013新增
@MOV(021) #2B46 D4470  ; RK_15 轮廓检测机构轮廓测量值开始字（String）
@MOV(021) #4646 D4471
@MOV(021) #4646 D4472
@MOV(021) #4646 D4473
LD TR2
AND<>(305) #5858 D4426  ; RK_15 轮廓检测机构轮廓测量值开始字
AND<>(305) #2B46 D4426  ; RK_15 轮廓检测机构轮廓测量值开始字
AND<>(305) #2D46 D4426  ; RK_15 轮廓检测机构轮廓测量值开始字
FVAL(449) D4450 D4460  ; RK_15 轮廓检测机构轮廓测量值开始字（String）, RK_15 轮廓检测机构轮廓测量值开始字（Float）
LD TR2
LD=(300) #5858 D4426  ; RK_15 轮廓检测机构轮廓测量值开始字
OR=(300) #2B46 D4426  ; RK_15 轮廓检测机构轮廓测量值开始字
OR=(300) #2D46 D4426  ; RK_15 轮廓检测机构轮廓测量值开始字
LD<>(305) #5858 D4426  ; RK_15 轮廓检测机构轮廓测量值开始字
AND<>(305) #2B46 D4426  ; RK_15 轮廓检测机构轮廓测量值开始字
AND<>(305) #2D46 D4426  ; RK_15 轮廓检测机构轮廓测量值开始字
ORLD
ANDLD
@SET W313.01  ; RK_15 轮廓检测机构测量数据读取解析完成标志
LD TR1
LD<>(305) &10 D4420  ; RK_15 轮廓检测机构轮廓测量字节数
OR<>(305) #4D31 D4421  ; RK_15 轮廓检测机构轮廓测量结果开始字
ANDLD
ANDNOT H7.15  ; 空跑程序  // 20181013新增
OUT W314.11  ; RK_15 轮廓检测机构测量数据读取解析异常标志
LD TR0
LD W313.01  ; RK_15 轮廓检测机构测量数据读取解析完成标志
LD W314.11  ; RK_15 轮廓检测机构测量数据读取解析异常标志
AND W432.03  ; RK_15 轮廓检测通讯异常[alm]
ORLD
@OR D1297.00  ; RK_15 轮廓检测机构复位（M）
ANDLD
RSET W312.01  ; RK_15 轮廓检测机构测量数据读取触发标志

